(* CODESYS project ScaraRobot2Hand

Project tree, tasks and I/O mapping:
  Just_Motion_Control_x86_64_Linux_SM_WV : Just Motion Control Cortex-Linux SM WV, Shenzhen Just Motion Control Electromechanics Co., version 3.5.19.50
    application Application
      libraries: CommFB, * (3S - Smart Software Solutions GmbH); JMC COMMON, 3.5.17.0 (JMC); ModbusFB, 4.3.0.0 (3S - Smart Software Solutions GmbH); Standard, 3.5.18.0 (System); SysFile, * (System); SysTimeCore, * (System); SysTimeRtc, * (System)
      task EtherCAT_Task (cyclic, interval 8 ms, priority 1) calls POU_MOTION, POU_JOG_ROBOT, POU_CONTROL_ROBOT, POU_MONITOR_ROBOT, POU_COORDINATE_, POU_HOMING, PRG_TrackingObjectSource_A, PRG_TrackingQueue_A, PRG_MultiToolTracking_A, PRG_TrackingObjectSource_B, PRG_TrackingQueue_B, PRG_MultiToolTracking_B
      task SoftMotion_PlanningTask_1 (freewheeling, priority 15) calls nothing
      task SoftMotion_PlanningTask (freewheeling, priority 15) calls nothing
      task Task_Communication (cyclic, interval 15 ms, priority 1) calls POU_MODBUS, PRG_VisionConfigInit, POU_CAM, PRG_VisionModbus, PRG_VisionManager
      task Task_Program (cyclic, interval 8 ms, priority 20) calls Monitor_Production, POU_Alarm, POU_TransFormOXYR, POU_Main, POU_HMI_CONTROL_ROBOT, POU_SAFETY_CHECK
      ENUM/
        Application/
          data type E_ApplicationID
          data type E_ApplicationManagerState
          data type E_ApplicationSimulationMode
        Conveyor Tracking/
          data type E_ConveyorState
          data type E_MultiTrackState
          data type E_ObjectSourceType
          data type E_TrackingObjectState
          data type E_TrackingSelectMode
          data type E_TrackingState
        data type E_AppCoordSystem
        data type E_ApplicationState
        data type E_MoveState
        data type E_ObjectSelectMode
        data type E_QueueResult
        data type E_SystemTestStage
        GlueBonding/
          data type E_GlueRunMode
          data type E_GlueState
          data type E_PathProcessState
          data type E_PathSegmentType
        Interpreter/
          data type E_CondLink
          data type E_CondOperator
          data type E_CondSource
          data type E_RobotCmd
        TOOL/
          data type E_ToolAction
          data type E_ToolCommandType
          data type E_ToolRuntimeState
          data type E_ToolType
        Vision/
          data type E_AlignState
          data type E_InspectionResult
          data type E_InspectionState
          data type E_PlaceMode
          data type E_VisionApplication
          data type E_VisionDataType
          data type E_VisionResultStatus
          data type E_VisionRobot
          data type E_VisionState
      FB_/
        Application/
        function block Blink_Bit [ST]
        ConveyorTrack/
          function block FB_CONVEYOR_TRACKING_MANAGER [ST]
          function block FB_CONVEYOR_TRACKING_MANAGER_B [ST]
          function block FB_MultiToolTrackingController_A [ST]
          function block FB_MultiToolTrackingController_B [ST]
          function block FB_SensorObjectSource [ST]
          function block FB_TrackingCoreInterface_A [ST]
          function block FB_TrackingCoreInterface_B [ST]
          function block FB_TrackingMotionQueueAdapter [ST]
          function block FB_TrackingMotionQueueAdapter_B [ST]
          function block FB_VisionObjectSource [ST]
          function block FB_VisionTrackingResultAdapter [ST]
        function block FB_CalibRunPoints [ST]
        function block FB_CONVERT_POS [ST]
        function block FB_FileManager [ST]: Load, Save
        function block FB_MotionQueuePop [ST]
        function block FB_MotionQueuePop_B [ST]
        function block FB_MotionQueuePush [ST]
        function block FB_MotionQueuePush_B [ST]
        function block FB_PALLETS [ST]
        function block FB_Real_TO_Word_ [ST]
        function block FB_Run_Point [ST]
        function block FB_RunMoveC [ST]
        function block FB_RunMoveL [ST]
        function block FB_RunMoveP [ST]
        function block FB_RunMoveP_1 [ST]
        function block FB_TorqueDiff [ST]
        function block FB_TriggerVS [ST]
        function block FB_word_TO_real_ [ST]
        function block FB_Write_Log [ST]: Write
        Modbus/
          function block FB_VisionModbusDriver [ST]
        TOOL/
          function block FB_SelectRobotTool [ST]
          function block FB_SelectRobotTool_B [ST]
          function block FB_ToolManager [ST]
          function block FB_ToolManager_B [ST]
          function block FB_ToolObjectScheduler [ST]
        Vision/
          function block FB_VisionAlign_1 [ST]
          function block FB_VisionAlign [ST]
          function block FB_VisionGetResult [ST]
          function block FB_VisionTrackingTrigger [ST]
          function block FB_VisionWaitResult [ST]
      FC_/
        function ApplyTransformOnePointDeg [ST]
        function CalcScaraTransformDeg [ST]
        Conveyor/
          function F_AngleDifferenceDeg [ST]
          function F_IsTrackingObjectSelectable [ST]
          function F_IsVisionTrackingDuplicate [ST]
          function F_VisionTrackingRawToMM [ST]
        Coordinate_TF/
          function F_MapAppCoordSystem [ST]
        function F_BuildMotionItem [ST]
        function F_BuildMotionItem_B [ST]
        function F_CheckPositionReached [ST]
        function F_GetFreeMoveSlot [ST]
        function F_GetFreeMoveSlot_B [ST]
        function F_IsMotionCmd [ST]
        function FC_CalcCalibPoint [ST]
        function FC_Deg_To_Rad [ST]
        function FC_NormalizeAngleDeg [ST]
        function FC_Rad_To_Deg [ST]
        Geometry/
          function F_AngleBetweenPoints [ST]
          function F_DegToRad [ST]
          function F_Distance2D [ST]
          function F_Distance3D [ST]
          function F_NormalizeAngleDeg [ST]
          function F_NormalizeVector2D [ST]
          function F_RadToDeg [ST]
          function F_RotateAroundCenter2D [ST]
          function F_RotatePos2D [ST]
          function F_VectorLength2D [ST]
        function MyATAN2 [ST]
        Path/
          function F_CalculateBlendRadius [ST]
          function F_CalculatePathLength [ST]
          function F_InterpolatePosLinear [ST]
          function F_IsDuplicatePathPoint [ST]
          function F_PathPointDistance [ST]
        RBA/
          function F_CalcReg_A [ST]
          function F_CalcVar_A [ST]
          function F_CompareDINT_A [ST]
          function F_EvalCondition_A [ST]
          function F_EvalCondRow_A [ST]
          function F_EvalCondRowFromEdit_A [ST]
          function F_FindElseOrEndIf_A [ST]
          function F_FindEndIf_A [ST]
          function F_FindEndWhile_A [ST]
          function F_FindWhileStart_A [ST]
          function F_GetCondValue_A [ST]
          function F_GetPointSMC_A [ST]
        RBB/
          function F_CalcReg_B [ST]
          function F_CalcVar_B [ST]
          function F_CompareDINT_B [ST]
          function F_EvalCondition_B [ST]
          function F_EvalCondRow_B [ST]
          function F_EvalCondRowFromEdit_B [ST]
          function F_FindElseOrEndIf_B [ST]
          function F_FindEndIf_B [ST]
          function F_FindEndWhile_B [ST]
          function F_FindWhileStart_B [ST]
          function F_GetCondValue_B [ST]
          function F_GetPointSMC_B [ST]
        Tool/
          function F_ConvertToolTCP [ST]
        TrackingQueue/
          function F_SelectTrackingObject [ST]
        Vision/
          function F_CalcTraySlotTarget [ST]
          function F_CheckAlignResult [ST]
          function F_CheckPosRange [ST]
          function F_CheckRangeReal [ST]
          function F_CheckVisionHeader [ST]
          function F_CheckVisionScore [ST]
          function F_CountInspectionFail [ST]
          function F_VisionDINTHighWord [ST]
          function F_VisionDINTLowWord [ST]
          function F_VisionRealToRawDINT [ST]
          function F_VisionUDINTHighWord [ST]
          function F_VisionUDINTLowWord [ST]
          function F_VisionWordsToDINT_LH [ST]
          function F_VisionWordsToUDINT_LH [ST]
      GLOBAL_/
        global variables GVL_2
        global variables GVL
      global variables GVL_1
      PRG_MACHINE/
        program Monitor_Production [ST]: Qty_Production, Tactime_Input, Tactime_MC1, Tactime_MC2, Tactime_output
        program POU_Alarm [ST]: Alarm_Project_4, Alarm_Robot
        program POU_CAM [ST]: ACT_CHECKCONNECT, ACT_Total, ACT_TRIGGER_TOP
        program POU_MODBUS [ST]: ACT_TCP_Sever
        program PRG_VisionConfigInit [ST]
        program PRG_VisionModbus [ST]
        program PRG_VisionTest [ST]
      PRG_ROBOT/
        program POU_CONTROL_ROBOT [ST]: ACT_LOGIC, ACT_POWER, ACT_Reset, ACT_SET_DYNAMICLIMITS
        program POU_COORDINATE_ [ST]: ACT_CFC, ACT_Conver_Pos, ACT_LOGIC
        program POU_HMI_CONTROL_ROBOT [ST]: ACT_ControlPanel, ACT_HMI_A_ConditionEditor, ACT_HMI_A_Vision_Tracking_Config, ACT_HMI_B_ConditionEditor, ACT_HMI_B_Vision_Tracking_Config, ACT_HMI_Recipe_Config, ACT_HMI_Recipe_Config_B, ACT_HMI_SensorSource_Config_B, ACT_HMI_SensorSource_Config, ACT_HMIToolConfigEditor_A, ACT_HMIToolConfigEditor_B, ACT_JOG_LOGIC, ACT_MANORAUTO, ACT_MENU, ACT_select_rb, ACT_View_Edit_Cmd, ACT_View_Edit_Cmd_B, ACT_View_Edit_Point_A, ACT_View_Edit_Point_B
        program POU_HOMING [ST]: ACT_ERROR, ACT_Home_Z, ACT_HOMING, ACT_SETLIMIT, ACT_STOP
        program POU_JOG_ROBOT [ST]: ACT_JOG, ACT_LOGIC_A, ACT_LOGIC_B, ACT_LOGIC_R
        program POU_Main [ST]: ACT_IN, ACT_Manual_MC, ACT_Out, ACT_SAVE_FILE, ACT_SelectProjectRun, ACT_StatusMode, TimeTable
        program POU_MONITOR_ROBOT [ST]: ACT_LOGIC, ACT_READ, ACT_Teaching
        program POU_MOTION [ST]: MOVC, MOVL, MOVP, ACT_GO_Pos_Auto, Main_Base_Program_RB_A, PRG_A_MotionManager, Main_Base_Program_RB_B, PRG_B_MotionManager, _Main_Process_Test, A_Test_Motion, B1_Test_Motion, _Main_Process_Test_VS, A_Test_Motion_VS, B1_Test_Motion_VS, _Main_Process_4, A0_Wait_4, A1_Pick_T1_4, A2_Place_T1_OK_4, A3_Place_T1_NG_4, A4_Pick_T2_4, A5_Place_T2_OK_4, A6_Place_T2_NG_4, A7_Barcode_T1_4, A8_Place_T2_NG_TS_4, B0_wait_4, B1_Pick_T1_4, B2_PLace_T1_4, B3_Barcode_4, B_Trigger_4, CNV_NG, Pro_MC1_4_, Pro_MC2_4_, ACT_GO_Pos_Manual, B_Auto_Calib_4, Robot_Calib_Vision, M_CACULATOR_Z, M_CHOOSE_POS, M_CHOOSE_POS_Calib, M_CHOOSE_POS_Man, M_CHOOSE_POS_VS, M_CHOOSE_POS_XY, M_CHOOSE_POS_Z_BF, M_initProcess, M_R_Mov, M_reset, ACT_Excute_Run
        program POU_SAFETY_CHECK [ST]: ACT_RB_A, ACT_RB_B
        program POU_TransFormOXYR [ST]
        program PRG_MultiToolTracking_A [ST]
        program PRG_MultiToolTracking_B [ST]
        program PRG_TestVisionAlign [ST]
        program PRG_TestVisionTriggerResult [ST]
        program PRG_TrackingObjectSource_A [ST]
        program PRG_TrackingObjectSource_B [ST]
        program PRG_TrackingQueue_A [ST]
        program PRG_TrackingQueue_B [ST]
        program PRG_VisionManager [ST]
        program PRG_VisionTrackingTest_A [ST]
      axis group SCARA_A: TRAFO.Kin_Scara2_Z, axes A0, A1, A2
      axis group SCARA_B: TRAFO.Kin_Scara2_Z, axes B0, B1, B2
      STRUCT_/
        Alarm/
          data type Alarm_Robot
        Application/
          data type ST_APPLICATION_COMMAND
          data type ST_APPLICATION_RESPONSE
        Array/
          data type Pallets_In
          data type Pallets_Out
        CAM/
          data type Calib_Cam
          data type Calib_Cam_Input_Model
          data type ModbusCam
          data type VS_Control
        COMMON/
          data type ST_ERROR_INFO
          data type ST_MODULE_REQUEST
          data type ST_MODULE_RESPONSE
          data type ST_MotionProfile
          data type ST_POS
          data type ST_RANGE_REAL
          data type ST_Transform2D
          data type ST_VECTOR_2D
        ConveyorTracking/
          data type ST_CONVEYOR_CONFIG
          data type ST_CONVEYOR_RUNTIME
          data type ST_CONVEYOR_STATUS
          data type ST_HMIToolConfigEditor
          data type ST_PCS_INFO
          data type ST_SensorObjectSourceConfig
          data type ST_TRACKING_CONFIG
          data type ST_TRACKING_IO_CONFIG
          data type ST_TRACKING_MOTION_CONFIG
          data type ST_TRACKING_MOTION_PHASE_CONFIG
          data type ST_TRACKING_OBJECT
          data type ST_TRACKING_QUEUE
          data type ST_TRACKING_RUNTIME
          data type ST_TRACKING_SIMULATION_CONFIG
          data type ST_TRACKING_WORKSPACE_CONFIG
          data type ST_TrackingObjectQueue
          data type ST_VISION_TRACK_OBJECT_ITEM
          data type ST_VISION_TRACK_OBJECT_RESULT
          data type ST_VisionTrackingDetection
          data type ST_VisionTrackingMultiResult
          data type ST_VisionTrackingSourceConfig
        Geometry/
          data type ST_CIRCLE_2D
          data type ST_LINE_2D
          data type ST_PATH_BLOCK
          data type ST_PATH_DATA
          data type ST_PATH_POINT
        Glue/
          data type ST_GLUE_CONFIG
          data type ST_GLUE_RUNTIME
        HMI/
          data type MainMC
          data type MODBUS
          data type Project
          data type TimeRun
        Modbus/
          data type ST_VISION_MODBUS_CONTROL
          data type ST_VISION_MODBUS_STATUS
        MOTOR/
          data type MOTOR_DATA
          data type MOTOR_IN
          data type MOTOR_OUT
        Project/
          data type Data_Point_Calib
          data type Data_Project_3
          data type Data_Project
          Project1/
          data type Project_2
          data type Project_3
          data type Project_3_VISION
          Project_4/
            data type Alarm_P_4
            data type Pro4_auto
            data type Pro4_Input
            data type Pro4_manual
            data type Pro4_Monitor
            data type Pro4_Process
            data type Pro4_RB_Pos
            data type Pro4_setting
            data type Pro4_Setting_Funtion
            data type Project4
        ROBOT/
          data type Model_Data_RB_ALL
          data type Model_Data_RB
          data type Move_Point
          data type Move_Type
          data type PCS_Data
          data type Pos_Coordsystem
          data type Project_And_Model
          data type RB_DATA
          data type RB_IN
          data type RB_IN_Man
          data type RB_OUT
          data type RB_Signal_Input
          data type RB_Speed_Point
          data type ST_Condition
          data type ST_ConditionLine
          data type ST_ConditionRow
          data type ST_ConditionTable
          data type ST_MotionParam
          data type ST_MotionQueueItem
          data type ST_RobotProgram
          data type ST_RobotStep
          data type ST_ScaraTransformDeg
          data type Torque_Axis
        TOOL/
          data type ST_MultiToolTrackingCommand
          data type ST_MultiToolTrackingRecipe
          data type ST_MultiToolTrackingStatus
          data type ST_ToolCommand
          data type ST_ToolConfig
          data type ST_ToolIOConfig
          data type ST_ToolStatus
        Vision/
          data type ST_ALIGN_CONFIG
          data type ST_ALIGN_RESULT
          data type ST_ALIGN_RUNTIME
          data type ST_AlignResult
          data type ST_ControlWord_VS
          data type ST_INSPECTION_CONFIG
          data type ST_INSPECTION_ITEM
          data type ST_INSPECTION_RESULT
          data type ST_INSPECTION_RUNTIME
          data type ST_InspectionItem
          data type ST_PathPoint
          data type ST_StatusWord_VS
          data type ST_TrayConfig
          data type ST_TrayRuntime
          data type ST_VISION_ALIGN_REQUEST
          data type ST_VISION_CHANNEL_STATUS
          data type ST_VISION_COMMAND
          data type ST_VISION_CONFIG
          data type ST_VISION_JOB_CONFIG
          data type ST_VISION_POS_RESULT
          data type ST_VISION_RESULT
          data type ST_VISION_RESULT_HEADER
          data type ST_VisionAlignRecipe
          data type ST_VisionAlignToolConfig
          data type ST_VisionAlignToolRuntime
          data type ST_VisionCommand
      Symbols
      trace Trace (task EtherCAT_Task): B1.fSetVelocity, B1.fActVelocity, B3.fSetVelocity, B3.fActVelocity, A0.diSetVelocity, A0.diActVelocity, A1.diSetVelocity, A1.diActVelocity, POU_CONTROL_ROBOT.J1_PosError, POU_CONTROL_ROBOT.J2_PosError, POU_CONTROL_ROBOT.J1_VelError, POU_CONTROL_ROBOT.J2_VelError, A0.fSetPosition, A0.fActPosition, A0.fActPosition, A0.fActPosition, A1.fActPosition, A1.fSetPosition, A1.fSetVelocity, A1.fActVelocity, GVL.RB_A_.CUR_X, GVL.RB_A_.CUR_Y, GVL.RB_A_.CUR_SP_X, GVL.RB_A_.CUR_SP_Y, SM_Drive_Logical.fActPosition
    EtherCAT_Master_SoftMotion : EtherCAT Master SoftMotion, CODESYS, version 4.6.0.0
        settings: MasterCycleTime = 8000; NetworkName = 'EtherCAT'; NetworkName = "EtherCAT"; SelectNetworkByName = False; SyncOffset = -20; SrcAddress1 = 3830; SrcAddress2 = 3107753849
      TA133 : TA133, Shenzhen Just Motion Control Electromechanics Co,.ltd, order no. TA133, version Revision=16#00010004
          settings: ModularDevice = True; EnableExpertSettings = True; MDP_InputOffsets = [0,736]; MDP_OutputOffsets = [0,984]; StationAlias = 1001; DeviceIdenticationADO = 18; DeviceIdenticationMode = 1; Sync.Length = 127; Sync.Length = 97; FMMU.Length = 127; FMMU.Length = 97; Number of RxPDOs of the Slave = 8; Number of TxPDOs of the Slave = 8; DC sync0 cycletime = 8000; DC enable = 1; DC sync0 enable = 1; DC sync0 shift time = 0; DC sync1 cycletime = 8000; DC sync1 enable = 0; DC sync1 shift time = 0; Number of SDO = 1; download slot cfg.Index = 16#F030; download slot cfg.Subindex = 16#00; download slot cfg.Size = 48; download slot cfg.AbortIfError = FALSE; download slot cfg.JumpToLine = FALSE; download slot cfg.Line = 0; download slot cfg.CompleteAccess = True; download slot cfg = [1,0,230,0,0,0]; RxTxPdo.NumberofExcludes = 0; RxTxPdo.NumberofEntries = 7; RxTxPdo.Index = 16#1700; RxTxPdo.Fixed = False; RxTxPdo.Mandatory = False; RxTxPdo.Virtual = False; RxTxPdo.Sm = 2; RxTxPdo.Su = 2; RxTxPdo.Name = 'Outputs'; RxTxPdo.DependOnSlot = False; RxTxPdo.DependOnSlotGroup = False;
            RxTxPdo.OverwrittenByModule = False; Controlword(axis 1).Index = 16#6040; Controlword(axis 1).SubIndex = 0; Controlword(axis 1).Size = 16; Controlword(axis 1).Offset = 0; Controlword(axis 1).DependOnSlot = False; Controlword(axis 1).DependOnSlotGroup = False; Modes of operation(axis 1).Index = 16#6060; Modes of operation(axis 1).SubIndex = 0; Modes of operation(axis 1).Size = 8; Modes of operation(axis 1).Offset = 0; Modes of operation(axis 1).DependOnSlot = False; Modes of operation(axis 1).DependOnSlotGroup = False; Target position(axis 1).Index = 16#607A; Target position(axis 1).SubIndex = 0; Target position(axis 1).Size = 32; Target position(axis 1).Offset = 0; Target position(axis 1).DependOnSlot = False; Target position(axis 1).DependOnSlotGroup = False; High-speed comparison 1(axis 1).Index = 16#6701; High-speed comparison 1(axis 1).SubIndex = 0; High-speed comparison 1(axis 1).Size = 32; High-speed comparison 1(axis 1).Offset = 0; High-speed comparison 1(axis 1).DependOnSlot = False; High-speed comparison 1(axis 1).DependOnSlotGroup = False; High-speed comparison 2(axis 1).Index = 16#6702; High-speed comparison 2(axis 1).SubIndex = 0; High-speed comparison 2(axis 1).Size = 32; High-speed comparison 2(axis 1).Offset = 0; High-speed comparison 2(axis 1).DependOnSlot = False; High-speed comparison 2(axis 1).DependOnSlotGroup = False; PWM Duty(axis 1).Index = 16#6707; PWM Duty(axis 1).SubIndex = 0; PWM Duty(axis 1).Size = 8; PWM Duty(axis 1).Offset = 0; PWM Duty(axis 1).DependOnSlot = False; PWM Duty(axis 1).DependOnSlotGroup = False; PWM Freq(axis 1).Index = 16#6708; PWM Freq(axis 1).SubIndex = 0; PWM Freq(axis 1).Size = 32;
            PWM Freq(axis 1).Offset = 0; PWM Freq(axis 1).DependOnSlot = False; PWM Freq(axis 1).DependOnSlotGroup = False; RxTxPdo.NumberofExcludes = 0; RxTxPdo.NumberofEntries = 7; RxTxPdo.Index = 16#1710; RxTxPdo.Fixed = False; RxTxPdo.Mandatory = False; RxTxPdo.Virtual = False; RxTxPdo.Sm = 2; RxTxPdo.Su = 2; RxTxPdo.Name = 'Outputs'; RxTxPdo.DependOnSlot = False; RxTxPdo.DependOnSlotGroup = False; RxTxPdo.OverwrittenByModule = False; Controlword(axis 2).Index = 16#6840; Controlword(axis 2).SubIndex = 0; Controlword(axis 2).Size = 16; Controlword(axis 2).Offset = 0; Controlword(axis 2).DependOnSlot = False; Controlword(axis 2).DependOnSlotGroup = False; Modes of operation(axis 2).Index = 16#6860; Modes of operation(axis 2).SubIndex = 0; Modes of operation(axis 2).Size = 8; Modes of operation(axis 2).Offset = 0; Modes of operation(axis 2).DependOnSlot = False; Modes of operation(axis 2).DependOnSlotGroup = False; Target position(axis 2).Index = 16#687A; Target position(axis 2).SubIndex = 0; Target position(axis 2).Size = 32; Target position(axis 2).Offset = 0; Target position(axis 2).DependOnSlot = False; Target position(axis 2).DependOnSlotGroup = False; High-speed comparison 1(axis 2).Index = 16#6F01; High-speed comparison 1(axis 2).SubIndex = 0; High-speed comparison 1(axis 2).Size = 32; High-speed comparison 1(axis 2).Offset = 0; High-speed comparison 1(axis 2).DependOnSlot = False; High-speed comparison 1(axis 2).DependOnSlotGroup = False; High-speed comparison 2(axis 2).Index = 16#6F02;
            High-speed comparison 2(axis 2).SubIndex = 0; High-speed comparison 2(axis 2).Size = 32; High-speed comparison 2(axis 2).Offset = 0; High-speed comparison 2(axis 2).DependOnSlot = False; High-speed comparison 2(axis 2).DependOnSlotGroup = False; PWM Duty(axis 2).Index = 16#6F07; PWM Duty(axis 2).SubIndex = 0; PWM Duty(axis 2).Size = 8; PWM Duty(axis 2).Offset = 0; PWM Duty(axis 2).DependOnSlot = False; PWM Duty(axis 2).DependOnSlotGroup = False; PWM Freq(axis 2).Index = 16#6F08; PWM Freq(axis 2).SubIndex = 0; PWM Freq(axis 2).Size = 32; PWM Freq(axis 2).Offset = 0; PWM Freq(axis 2).DependOnSlot = False; PWM Freq(axis 2).DependOnSlotGroup = False; RxTxPdo.NumberofExcludes = 0; RxTxPdo.NumberofEntries = 7; RxTxPdo.Index = 16#1720; RxTxPdo.Fixed = False; RxTxPdo.Mandatory = False; RxTxPdo.Virtual = False; RxTxPdo.Sm = 2; RxTxPdo.Su = 2; RxTxPdo.Name = 'Outputs'; RxTxPdo.DependOnSlot = False; RxTxPdo.DependOnSlotGroup = False; RxTxPdo.OverwrittenByModule = False; Controlword(axis 3).Index = 16#7040; Controlword(axis 3).SubIndex = 0; Controlword(axis 3).Size = 16; Controlword(axis 3).Offset = 0; Controlword(axis 3).DependOnSlot = False; Controlword(axis 3).DependOnSlotGroup = False; Modes of operation(axis 3).Index = 16#7060; Modes of operation(axis 3).SubIndex = 0; Modes of operation(axis 3).Size = 8; Modes of operation(axis 3).Offset = 0; Modes of operation(axis 3).DependOnSlot = False;
            Modes of operation(axis 3).DependOnSlotGroup = False; Target position(axis 3).Index = 16#707A; Target position(axis 3).SubIndex = 0; Target position(axis 3).Size = 32; Target position(axis 3).Offset = 0; Target position(axis 3).DependOnSlot = False; Target position(axis 3).DependOnSlotGroup = False; High-speed comparison 1(axis 3).Index = 16#7701; High-speed comparison 1(axis 3).SubIndex = 0; High-speed comparison 1(axis 3).Size = 32; High-speed comparison 1(axis 3).Offset = 0; High-speed comparison 1(axis 3).DependOnSlot = False; High-speed comparison 1(axis 3).DependOnSlotGroup = False; High-speed comparison 2(axis 3).Index = 16#7702; High-speed comparison 2(axis 3).SubIndex = 0; High-speed comparison 2(axis 3).Size = 32; High-speed comparison 2(axis 3).Offset = 0; High-speed comparison 2(axis 3).DependOnSlot = False; High-speed comparison 2(axis 3).DependOnSlotGroup = False; PWM Duty(axis 3).Index = 16#7707; PWM Duty(axis 3).SubIndex = 0; PWM Duty(axis 3).Size = 8; PWM Duty(axis 3).Offset = 0; PWM Duty(axis 3).DependOnSlot = False; PWM Duty(axis 3).DependOnSlotGroup = False; PWM Freq(axis 3).Index = 16#7708; PWM Freq(axis 3).SubIndex = 0; PWM Freq(axis 3).Size = 32; PWM Freq(axis 3).Offset = 0; PWM Freq(axis 3).DependOnSlot = False; PWM Freq(axis 3).DependOnSlotGroup = False; RxTxPdo.NumberofExcludes = 0; RxTxPdo.NumberofEntries = 7; RxTxPdo.Index = 16#1730; RxTxPdo.Fixed = False; RxTxPdo.Mandatory = False; RxTxPdo.Virtual = False; RxTxPdo.Sm = 2; RxTxPdo.Su = 2; RxTxPdo.Name = 'Outputs';
            RxTxPdo.DependOnSlot = False; RxTxPdo.DependOnSlotGroup = False; RxTxPdo.OverwrittenByModule = False; Controlword(axis 4).Index = 16#7840; Controlword(axis 4).SubIndex = 0; Controlword(axis 4).Size = 16; Controlword(axis 4).Offset = 0; Controlword(axis 4).DependOnSlot = False; Controlword(axis 4).DependOnSlotGroup = False; Modes of operation(axis 4).Index = 16#7860; Modes of operation(axis 4).SubIndex = 0; Modes of operation(axis 4).Size = 8; Modes of operation(axis 4).Offset = 0; Modes of operation(axis 4).DependOnSlot = False; Modes of operation(axis 4).DependOnSlotGroup = False; Target position(axis 4).Index = 16#787A; Target position(axis 4).SubIndex = 0; Target position(axis 4).Size = 32; Target position(axis 4).Offset = 0; Target position(axis 4).DependOnSlot = False; Target position(axis 4).DependOnSlotGroup = False; High-speed comparison 1(axis 4).Index = 16#7F01; High-speed comparison 1(axis 4).SubIndex = 0; High-speed comparison 1(axis 4).Size = 32; High-speed comparison 1(axis 4).Offset = 0; High-speed comparison 1(axis 4).DependOnSlot = False; High-speed comparison 1(axis 4).DependOnSlotGroup = False; High-speed comparison 2(axis 4).Index = 16#7F02; High-speed comparison 2(axis 4).SubIndex = 0; High-speed comparison 2(axis 4).Size = 32; High-speed comparison 2(axis 4).Offset = 0; High-speed comparison 2(axis 4).DependOnSlot = False; High-speed comparison 2(axis 4).DependOnSlotGroup = False; PWM Duty(axis 4).Index = 16#7F07; PWM Duty(axis 4).SubIndex = 0; PWM Duty(axis 4).Size = 8; PWM Duty(axis 4).Offset = 0; PWM Duty(axis 4).DependOnSlot = False; PWM Duty(axis 4).DependOnSlotGroup = False; PWM Freq(axis 4).Index = 16#7F08;
            PWM Freq(axis 4).SubIndex = 0; PWM Freq(axis 4).Size = 32; PWM Freq(axis 4).Offset = 0; PWM Freq(axis 4).DependOnSlot = False; PWM Freq(axis 4).DependOnSlotGroup = False; RxTxPdo.NumberofExcludes = 0; RxTxPdo.NumberofEntries = 7; RxTxPdo.Index = 16#1740; RxTxPdo.Fixed = False; RxTxPdo.Mandatory = False; RxTxPdo.Virtual = False; RxTxPdo.Sm = 2; RxTxPdo.Su = 2; RxTxPdo.Name = 'Outputs'; RxTxPdo.DependOnSlot = False; RxTxPdo.DependOnSlotGroup = False; RxTxPdo.OverwrittenByModule = False; Controlword(axis 5).Index = 16#8040; Controlword(axis 5).SubIndex = 0; Controlword(axis 5).Size = 16; Controlword(axis 5).Offset = 0; Controlword(axis 5).DependOnSlot = False; Controlword(axis 5).DependOnSlotGroup = False; Modes of operation(axis 5).Index = 16#8060; Modes of operation(axis 5).SubIndex = 0; Modes of operation(axis 5).Size = 8; Modes of operation(axis 5).Offset = 0; Modes of operation(axis 5).DependOnSlot = False; Modes of operation(axis 5).DependOnSlotGroup = False; Target position(axis 5).Index = 16#807A; Target position(axis 5).SubIndex = 0; Target position(axis 5).Size = 32; Target position(axis 5).Offset = 0; Target position(axis 5).DependOnSlot = False; Target position(axis 5).DependOnSlotGroup = False; High-speed comparison 1(axis 5).Index = 16#8701; High-speed comparison 1(axis 5).SubIndex = 0; High-speed comparison 1(axis 5).Size = 32; High-speed comparison 1(axis 5).Offset = 0; High-speed comparison 1(axis 5).DependOnSlot = False;
            High-speed comparison 1(axis 5).DependOnSlotGroup = False; High-speed comparison 2(axis 5).Index = 16#8702; High-speed comparison 2(axis 5).SubIndex = 0; High-speed comparison 2(axis 5).Size = 32; High-speed comparison 2(axis 5).Offset = 0; High-speed comparison 2(axis 5).DependOnSlot = False; High-speed comparison 2(axis 5).DependOnSlotGroup = False; PWM Duty(axis 5).Index = 16#8707; PWM Duty(axis 5).SubIndex = 0; PWM Duty(axis 5).Size = 8; PWM Duty(axis 5).Offset = 0; PWM Duty(axis 5).DependOnSlot = False; PWM Duty(axis 5).DependOnSlotGroup = False; PWM Freq(axis 5).Index = 16#8708; PWM Freq(axis 5).SubIndex = 0; PWM Freq(axis 5).Size = 32; PWM Freq(axis 5).Offset = 0; PWM Freq(axis 5).DependOnSlot = False; PWM Freq(axis 5).DependOnSlotGroup = False; RxTxPdo.NumberofExcludes = 0; RxTxPdo.NumberofEntries = 7; RxTxPdo.Index = 16#1750; RxTxPdo.Fixed = False; RxTxPdo.Mandatory = False; RxTxPdo.Virtual = False; RxTxPdo.Sm = 2; RxTxPdo.Su = 2; RxTxPdo.Name = 'Outputs'; RxTxPdo.DependOnSlot = False; RxTxPdo.DependOnSlotGroup = False; RxTxPdo.OverwrittenByModule = False; Controlword(axis 6).Index = 16#8840; Controlword(axis 6).SubIndex = 0; Controlword(axis 6).Size = 16; Controlword(axis 6).Offset = 0; Controlword(axis 6).DependOnSlot = False; Controlword(axis 6).DependOnSlotGroup = False; Modes of operation(axis 6).Index = 16#8860; Modes of operation(axis 6).SubIndex = 0; Modes of operation(axis 6).Size = 8;
            Modes of operation(axis 6).Offset = 0; Modes of operation(axis 6).DependOnSlot = False; Modes of operation(axis 6).DependOnSlotGroup = False; Target position(axis 6).Index = 16#887A; Target position(axis 6).SubIndex = 0; Target position(axis 6).Size = 32; Target position(axis 6).Offset = 0; Target position(axis 6).DependOnSlot = False; Target position(axis 6).DependOnSlotGroup = False; High-speed comparison 1(axis 6).Index = 16#8F01; High-speed comparison 1(axis 6).SubIndex = 0; High-speed comparison 1(axis 6).Size = 32; High-speed comparison 1(axis 6).Offset = 0; High-speed comparison 1(axis 6).DependOnSlot = False; High-speed comparison 1(axis 6).DependOnSlotGroup = False; High-speed comparison 2(axis 6).Index = 16#8F02; High-speed comparison 2(axis 6).SubIndex = 0; High-speed comparison 2(axis 6).Size = 32; High-speed comparison 2(axis 6).Offset = 0; High-speed comparison 2(axis 6).DependOnSlot = False; High-speed comparison 2(axis 6).DependOnSlotGroup = False; PWM Duty(axis 6).Index = 16#8F07; PWM Duty(axis 6).SubIndex = 0; PWM Duty(axis 6).Size = 8; PWM Duty(axis 6).Offset = 0; PWM Duty(axis 6).DependOnSlot = False; PWM Duty(axis 6).DependOnSlotGroup = False; PWM Freq(axis 6).Index = 16#8F08; PWM Freq(axis 6).SubIndex = 0; PWM Freq(axis 6).Size = 32; PWM Freq(axis 6).Offset = 0; PWM Freq(axis 6).DependOnSlot = False; PWM Freq(axis 6).DependOnSlotGroup = False; RxTxPdo.NumberofExcludes = 0; RxTxPdo.NumberofEntries = 3; RxTxPdo.Index = 16#1760; RxTxPdo.Fixed = False; RxTxPdo.Mandatory = False; RxTxPdo.Virtual = False; RxTxPdo.Sm = 2;
            RxTxPdo.Su = 2; RxTxPdo.Name = 'Outputs'; RxTxPdo.DependOnSlot = False; RxTxPdo.DependOnSlotGroup = False; RxTxPdo.OverwrittenByModule = False; High-speed comparison 1 switch.Index = 16#6703; High-speed comparison 1 switch.SubIndex = 0; High-speed comparison 1 switch.Size = 8; High-speed comparison 1 switch.Offset = 0; High-speed comparison 1 switch.DependOnSlot = False; High-speed comparison 1 switch.DependOnSlotGroup = False; High-speed comparison 2 switch.Index = 16#6704; High-speed comparison 2 switch.SubIndex = 0; High-speed comparison 2 switch.Size = 8; High-speed comparison 2 switch.Offset = 0; High-speed comparison 2 switch.DependOnSlot = False; High-speed comparison 2 switch.DependOnSlotGroup = False; PWM Output Enable.Index = 16#6709; PWM Output Enable.SubIndex = 0; PWM Output Enable.Size = 8; PWM Output Enable.Offset = 0; PWM Output Enable.DependOnSlot = False; PWM Output Enable.DependOnSlotGroup = False; RxTxPdo.NumberofExcludes = 0; RxTxPdo.NumberofEntries = 17; RxTxPdo.Index = 16#1600; RxTxPdo.Fixed = True; RxTxPdo.Mandatory = True; RxTxPdo.Virtual = False; RxTxPdo.Sm = 2; RxTxPdo.Su = 0; RxTxPdo.Name = 'Outputs process data mapping'; RxTxPdo.DependOnSlot = True; RxTxPdo.DependOnSlotGroup = False; RxTxPdo.OverwrittenByModule = True; AO0.Index = 16#7000; AO0.SubIndex = 1; AO0.Size = 16; AO0.Offset = 0; AO0.DependOnSlot = True;
            AO0.DependOnSlotGroup = False; Y0.Index = 16#7000; Y0.SubIndex = 2; Y0.Size = 1; Y0.Offset = 0; Y0.DependOnSlot = True; Y0.DependOnSlotGroup = False; Y1.Index = 16#7000; Y1.SubIndex = 3; Y1.Size = 1; Y1.Offset = 0; Y1.DependOnSlot = True; Y1.DependOnSlotGroup = False; Y2.Index = 16#7000; Y2.SubIndex = 4; Y2.Size = 1; Y2.Offset = 0; Y2.DependOnSlot = True; Y2.DependOnSlotGroup = False; Y3.Index = 16#7000; Y3.SubIndex = 5; Y3.Size = 1; Y3.Offset = 0; Y3.DependOnSlot = True; Y3.DependOnSlotGroup = False; Y4.Index = 16#7000; Y4.SubIndex = 6; Y4.Size = 1; Y4.Offset = 0; Y4.DependOnSlot = True; Y4.DependOnSlotGroup = False; Y5.Index = 16#7000; Y5.SubIndex = 7; Y5.Size = 1; Y5.Offset = 0; Y5.DependOnSlot = True; Y5.DependOnSlotGroup = False; Y6.Index = 16#7000; Y6.SubIndex = 8; Y6.Size = 1;
            Y6.Offset = 0; Y6.DependOnSlot = True; Y6.DependOnSlotGroup = False; Y7.Index = 16#7000; Y7.SubIndex = 9; Y7.Size = 1; Y7.Offset = 0; Y7.DependOnSlot = True; Y7.DependOnSlotGroup = False; Y8.Index = 16#7000; Y8.SubIndex = 10; Y8.Size = 1; Y8.Offset = 0; Y8.DependOnSlot = True; Y8.DependOnSlotGroup = False; Y9.Index = 16#7000; Y9.SubIndex = 11; Y9.Size = 1; Y9.Offset = 0; Y9.DependOnSlot = True; Y9.DependOnSlotGroup = False; Y10.Index = 16#7000; Y10.SubIndex = 12; Y10.Size = 1; Y10.Offset = 0; Y10.DependOnSlot = True; Y10.DependOnSlotGroup = False; Y11.Index = 16#7000; Y11.SubIndex = 13; Y11.Size = 1; Y11.Offset = 0; Y11.DependOnSlot = True; Y11.DependOnSlotGroup = False; Y12.Index = 16#7000; Y12.SubIndex = 14; Y12.Size = 1; Y12.Offset = 0; Y12.DependOnSlot = True; Y12.DependOnSlotGroup = False; Y13.Index = 16#7000;
            Y13.SubIndex = 15; Y13.Size = 1; Y13.Offset = 0; Y13.DependOnSlot = True; Y13.DependOnSlotGroup = False; Y14.Index = 16#7000; Y14.SubIndex = 16; Y14.Size = 1; Y14.Offset = 0; Y14.DependOnSlot = True; Y14.DependOnSlotGroup = False; Y15.Index = 16#7000; Y15.SubIndex = 17; Y15.Size = 1; Y15.Offset = 0; Y15.DependOnSlot = True; Y15.DependOnSlotGroup = False; RxTxPdo.NumberofExcludes = 0; RxTxPdo.NumberofEntries = 6; RxTxPdo.Index = 16#1B00; RxTxPdo.Fixed = False; RxTxPdo.Mandatory = False; RxTxPdo.Virtual = False; RxTxPdo.Sm = 3; RxTxPdo.Su = 3; RxTxPdo.Name = 'Inputs'; RxTxPdo.DependOnSlot = False; RxTxPdo.DependOnSlotGroup = False; RxTxPdo.OverwrittenByModule = False; Error Code(axis 1).Index = 16#603F; Error Code(axis 1).SubIndex = 0; Error Code(axis 1).Size = 16; Error Code(axis 1).Offset = 0; Error Code(axis 1).DependOnSlot = False; Error Code(axis 1).DependOnSlotGroup = False; Statusword(axis 1).Index = 16#6041; Statusword(axis 1).SubIndex = 0; Statusword(axis 1).Size = 16; Statusword(axis 1).Offset = 0; Statusword(axis 1).DependOnSlot = False;
            Statusword(axis 1).DependOnSlotGroup = False; Modes of operation display(axis 1).Index = 16#6061; Modes of operation display(axis 1).SubIndex = 0; Modes of operation display(axis 1).Size = 8; Modes of operation display(axis 1).Offset = 0; Modes of operation display(axis 1).DependOnSlot = False; Modes of operation display(axis 1).DependOnSlotGroup = False; Position actual value(axis 1).Index = 16#6064; Position actual value(axis 1).SubIndex = 0; Position actual value(axis 1).Size = 32; Position actual value(axis 1).Offset = 0; Position actual value(axis 1).DependOnSlot = False; Position actual value(axis 1).DependOnSlotGroup = False; Encoder Z phase(axis 1).Index = 16#6705; Encoder Z phase(axis 1).SubIndex = 0; Encoder Z phase(axis 1).Size = 32; Encoder Z phase(axis 1).Offset = 0; Encoder Z phase(axis 1).DependOnSlot = False; Encoder Z phase(axis 1).DependOnSlotGroup = False; PWM Error Code(axis 1).Index = 16#6711; PWM Error Code(axis 1).SubIndex = 0; PWM Error Code(axis 1).Size = 16; PWM Error Code(axis 1).Offset = 0; PWM Error Code(axis 1).DependOnSlot = False; PWM Error Code(axis 1).DependOnSlotGroup = False; RxTxPdo.NumberofExcludes = 0; RxTxPdo.NumberofEntries = 6; RxTxPdo.Index = 16#1B10; RxTxPdo.Fixed = False; RxTxPdo.Mandatory = False; RxTxPdo.Virtual = False; RxTxPdo.Sm = 3; RxTxPdo.Su = 3; RxTxPdo.Name = 'Inputs'; RxTxPdo.DependOnSlot = False; RxTxPdo.DependOnSlotGroup = False; RxTxPdo.OverwrittenByModule = False; Error Code(axis 2).Index = 16#683F; Error Code(axis 2).SubIndex = 0; Error Code(axis 2).Size = 16;
            Error Code(axis 2).Offset = 0; Error Code(axis 2).DependOnSlot = False; Error Code(axis 2).DependOnSlotGroup = False; Statusword(axis 2).Index = 16#6841; Statusword(axis 2).SubIndex = 0; Statusword(axis 2).Size = 16; Statusword(axis 2).Offset = 0; Statusword(axis 2).DependOnSlot = False; Statusword(axis 2).DependOnSlotGroup = False; Modes of operation display(axis 2).Index = 16#6861; Modes of operation display(axis 2).SubIndex = 0; Modes of operation display(axis 2).Size = 8; Modes of operation display(axis 2).Offset = 0; Modes of operation display(axis 2).DependOnSlot = False; Modes of operation display(axis 2).DependOnSlotGroup = False; Position actual value(axis 2).Index = 16#6864; Position actual value(axis 2).SubIndex = 0; Position actual value(axis 2).Size = 32; Position actual value(axis 2).Offset = 0; Position actual value(axis 2).DependOnSlot = False; Position actual value(axis 2).DependOnSlotGroup = False; Encoder Z phase(axis 2).Index = 16#6F05; Encoder Z phase(axis 2).SubIndex = 0; Encoder Z phase(axis 2).Size = 32; Encoder Z phase(axis 2).Offset = 0; Encoder Z phase(axis 2).DependOnSlot = False; Encoder Z phase(axis 2).DependOnSlotGroup = False; PWM Error Code(axis 2).Index = 16#6F11; PWM Error Code(axis 2).SubIndex = 0; PWM Error Code(axis 2).Size = 16; PWM Error Code(axis 2).Offset = 0; PWM Error Code(axis 2).DependOnSlot = False; PWM Error Code(axis 2).DependOnSlotGroup = False; RxTxPdo.NumberofExcludes = 0; RxTxPdo.NumberofEntries = 6; RxTxPdo.Index = 16#1B20; RxTxPdo.Fixed = False; RxTxPdo.Mandatory = False; RxTxPdo.Virtual = False; RxTxPdo.Sm = 3;
            RxTxPdo.Su = 3; RxTxPdo.Name = 'Inputs'; RxTxPdo.DependOnSlot = False; RxTxPdo.DependOnSlotGroup = False; RxTxPdo.OverwrittenByModule = False; Error Code(axis 3).Index = 16#703F; Error Code(axis 3).SubIndex = 0; Error Code(axis 3).Size = 16; Error Code(axis 3).Offset = 0; Error Code(axis 3).DependOnSlot = False; Error Code(axis 3).DependOnSlotGroup = False; Statusword(axis 3).Index = 16#7041; Statusword(axis 3).SubIndex = 0; Statusword(axis 3).Size = 16; Statusword(axis 3).Offset = 0; Statusword(axis 3).DependOnSlot = False; Statusword(axis 3).DependOnSlotGroup = False; Modes of operation display(axis 3).Index = 16#7061; Modes of operation display(axis 3).SubIndex = 0; Modes of operation display(axis 3).Size = 8; Modes of operation display(axis 3).Offset = 0; Modes of operation display(axis 3).DependOnSlot = False; Modes of operation display(axis 3).DependOnSlotGroup = False; Position actual value(axis 3).Index = 16#7064; Position actual value(axis 3).SubIndex = 0; Position actual value(axis 3).Size = 32; Position actual value(axis 3).Offset = 0; Position actual value(axis 3).DependOnSlot = False; Position actual value(axis 3).DependOnSlotGroup = False; Encoder Z phase(axis 3).Index = 16#7705; Encoder Z phase(axis 3).SubIndex = 0; Encoder Z phase(axis 3).Size = 32; Encoder Z phase(axis 3).Offset = 0; Encoder Z phase(axis 3).DependOnSlot = False; Encoder Z phase(axis 3).DependOnSlotGroup = False; PWM Error Code(axis 3).Index = 16#7711; PWM Error Code(axis 3).SubIndex = 0; PWM Error Code(axis 3).Size = 16; PWM Error Code(axis 3).Offset = 0; PWM Error Code(axis 3).DependOnSlot = False;
            PWM Error Code(axis 3).DependOnSlotGroup = False; RxTxPdo.NumberofExcludes = 0; RxTxPdo.NumberofEntries = 6; RxTxPdo.Index = 16#1B30; RxTxPdo.Fixed = False; RxTxPdo.Mandatory = False; RxTxPdo.Virtual = False; RxTxPdo.Sm = 3; RxTxPdo.Su = 3; RxTxPdo.Name = 'Inputs'; RxTxPdo.DependOnSlot = False; RxTxPdo.DependOnSlotGroup = False; RxTxPdo.OverwrittenByModule = False; Error Code(axis 4).Index = 16#783F; Error Code(axis 4).SubIndex = 0; Error Code(axis 4).Size = 16; Error Code(axis 4).Offset = 0; Error Code(axis 4).DependOnSlot = False; Error Code(axis 4).DependOnSlotGroup = False; Statusword(axis 4).Index = 16#7841; Statusword(axis 4).SubIndex = 0; Statusword(axis 4).Size = 16; Statusword(axis 4).Offset = 0; Statusword(axis 4).DependOnSlot = False; Statusword(axis 4).DependOnSlotGroup = False; Modes of operation display(axis 4).Index = 16#7861; Modes of operation display(axis 4).SubIndex = 0; Modes of operation display(axis 4).Size = 8; Modes of operation display(axis 4).Offset = 0; Modes of operation display(axis 4).DependOnSlot = False; Modes of operation display(axis 4).DependOnSlotGroup = False; Position actual value(axis 4).Index = 16#7864; Position actual value(axis 4).SubIndex = 0; Position actual value(axis 4).Size = 32; Position actual value(axis 4).Offset = 0; Position actual value(axis 4).DependOnSlot = False; Position actual value(axis 4).DependOnSlotGroup = False; Encoder Z phase(axis 4).Index = 16#7F05; Encoder Z phase(axis 4).SubIndex = 0; Encoder Z phase(axis 4).Size = 32;
            Encoder Z phase(axis 4).Offset = 0; Encoder Z phase(axis 4).DependOnSlot = False; Encoder Z phase(axis 4).DependOnSlotGroup = False; PWM Error Code(axis 4).Index = 16#7F11; PWM Error Code(axis 4).SubIndex = 0; PWM Error Code(axis 4).Size = 16; PWM Error Code(axis 4).Offset = 0; PWM Error Code(axis 4).DependOnSlot = False; PWM Error Code(axis 4).DependOnSlotGroup = False; RxTxPdo.NumberofExcludes = 0; RxTxPdo.NumberofEntries = 6; RxTxPdo.Index = 16#1B40; RxTxPdo.Fixed = False; RxTxPdo.Mandatory = False; RxTxPdo.Virtual = False; RxTxPdo.Sm = 3; RxTxPdo.Su = 3; RxTxPdo.Name = 'Inputs'; RxTxPdo.DependOnSlot = False; RxTxPdo.DependOnSlotGroup = False; RxTxPdo.OverwrittenByModule = False; Error Code(axis 5).Index = 16#803F; Error Code(axis 5).SubIndex = 0; Error Code(axis 5).Size = 16; Error Code(axis 5).Offset = 0; Error Code(axis 5).DependOnSlot = False; Error Code(axis 5).DependOnSlotGroup = False; Statusword(axis 5).Index = 16#8041; Statusword(axis 5).SubIndex = 0; Statusword(axis 5).Size = 16; Statusword(axis 5).Offset = 0; Statusword(axis 5).DependOnSlot = False; Statusword(axis 5).DependOnSlotGroup = False; Modes of operation display(axis 5).Index = 16#8061; Modes of operation display(axis 5).SubIndex = 0; Modes of operation display(axis 5).Size = 8; Modes of operation display(axis 5).Offset = 0; Modes of operation display(axis 5).DependOnSlot = False; Modes of operation display(axis 5).DependOnSlotGroup = False; Position actual value(axis 5).Index = 16#8064;
            Position actual value(axis 5).SubIndex = 0; Position actual value(axis 5).Size = 32; Position actual value(axis 5).Offset = 0; Position actual value(axis 5).DependOnSlot = False; Position actual value(axis 5).DependOnSlotGroup = False; Encoder Z phase(axis 5).Index = 16#8705; Encoder Z phase(axis 5).SubIndex = 0; Encoder Z phase(axis 5).Size = 32; Encoder Z phase(axis 5).Offset = 0; Encoder Z phase(axis 5).DependOnSlot = False; Encoder Z phase(axis 5).DependOnSlotGroup = False; PWM Error Code(axis 5).Index = 16#8711; PWM Error Code(axis 5).SubIndex = 0; PWM Error Code(axis 5).Size = 16; PWM Error Code(axis 5).Offset = 0; PWM Error Code(axis 5).DependOnSlot = False; PWM Error Code(axis 5).DependOnSlotGroup = False; RxTxPdo.NumberofExcludes = 0; RxTxPdo.NumberofEntries = 6; RxTxPdo.Index = 16#1B50; RxTxPdo.Fixed = False; RxTxPdo.Mandatory = False; RxTxPdo.Virtual = False; RxTxPdo.Sm = 3; RxTxPdo.Su = 3; RxTxPdo.Name = 'Inputs'; RxTxPdo.DependOnSlot = False; RxTxPdo.DependOnSlotGroup = False; RxTxPdo.OverwrittenByModule = False; Error Code(axis 6).Index = 16#883F; Error Code(axis 6).SubIndex = 0; Error Code(axis 6).Size = 16; Error Code(axis 6).Offset = 0; Error Code(axis 6).DependOnSlot = False; Error Code(axis 6).DependOnSlotGroup = False; Statusword(axis 6).Index = 16#8841; Statusword(axis 6).SubIndex = 0; Statusword(axis 6).Size = 16; Statusword(axis 6).Offset = 0; Statusword(axis 6).DependOnSlot = False;
            Statusword(axis 6).DependOnSlotGroup = False; Modes of operation display(axis 6).Index = 16#8861; Modes of operation display(axis 6).SubIndex = 0; Modes of operation display(axis 6).Size = 8; Modes of operation display(axis 6).Offset = 0; Modes of operation display(axis 6).DependOnSlot = False; Modes of operation display(axis 6).DependOnSlotGroup = False; Position actual value(axis 6).Index = 16#8864; Position actual value(axis 6).SubIndex = 0; Position actual value(axis 6).Size = 32; Position actual value(axis 6).Offset = 0; Position actual value(axis 6).DependOnSlot = False; Position actual value(axis 6).DependOnSlotGroup = False; Encoder Z phase(axis 6).Index = 16#8F05; Encoder Z phase(axis 6).SubIndex = 0; Encoder Z phase(axis 6).Size = 32; Encoder Z phase(axis 6).Offset = 0; Encoder Z phase(axis 6).DependOnSlot = False; Encoder Z phase(axis 6).DependOnSlotGroup = False; PWM Error Code(axis 6).Index = 16#8F11; PWM Error Code(axis 6).SubIndex = 0; PWM Error Code(axis 6).Size = 16; PWM Error Code(axis 6).Offset = 0; PWM Error Code(axis 6).DependOnSlot = False; PWM Error Code(axis 6).DependOnSlotGroup = False; RxTxPdo.NumberofExcludes = 0; RxTxPdo.NumberofEntries = 2; RxTxPdo.Index = 16#1B60; RxTxPdo.Fixed = False; RxTxPdo.Mandatory = False; RxTxPdo.Virtual = False; RxTxPdo.Sm = 3; RxTxPdo.Su = 3; RxTxPdo.Name = 'Inputs'; RxTxPdo.DependOnSlot = False; RxTxPdo.DependOnSlotGroup = False; RxTxPdo.OverwrittenByModule = False; High-speed comparison output status.Index = 16#6706; High-speed comparison output status.SubIndex = 0; High-speed comparison output status.Size = 8;
            High-speed comparison output status.Offset = 0; High-speed comparison output status.DependOnSlot = False; High-speed comparison output status.DependOnSlotGroup = False; PWM Output Enable Status.Index = 16#6710; PWM Output Enable Status.SubIndex = 0; PWM Output Enable Status.Size = 8; PWM Output Enable Status.Offset = 0; PWM Output Enable Status.DependOnSlot = False; PWM Output Enable Status.DependOnSlotGroup = False; RxTxPdo.NumberofExcludes = 0; RxTxPdo.NumberofEntries = 25; RxTxPdo.Index = 16#1A00; RxTxPdo.Fixed = True; RxTxPdo.Mandatory = True; RxTxPdo.Virtual = False; RxTxPdo.Sm = 3; RxTxPdo.Su = 0; RxTxPdo.Name = 'Inputs process data mapping'; RxTxPdo.DependOnSlot = True; RxTxPdo.DependOnSlotGroup = False; RxTxPdo.OverwrittenByModule = True; AI0.Index = 16#6000; AI0.SubIndex = 1; AI0.Size = 16; AI0.Offset = 0; AI0.DependOnSlot = True; AI0.DependOnSlotGroup = False; X0.Index = 16#6000; X0.SubIndex = 2; X0.Size = 1; X0.Offset = 0; X0.DependOnSlot = True; X0.DependOnSlotGroup = False; X1.Index = 16#6000; X1.SubIndex = 3; X1.Size = 1; X1.Offset = 0; X1.DependOnSlot = True; X1.DependOnSlotGroup = False; X2.Index = 16#6000;
            X2.SubIndex = 4; X2.Size = 1; X2.Offset = 0; X2.DependOnSlot = True; X2.DependOnSlotGroup = False; X3.Index = 16#6000; X3.SubIndex = 5; X3.Size = 1; X3.Offset = 0; X3.DependOnSlot = True; X3.DependOnSlotGroup = False; X4.Index = 16#6000; X4.SubIndex = 6; X4.Size = 1; X4.Offset = 0; X4.DependOnSlot = True; X4.DependOnSlotGroup = False; X5.Index = 16#6000; X5.SubIndex = 7; X5.Size = 1; X5.Offset = 0; X5.DependOnSlot = True; X5.DependOnSlotGroup = False; X6.Index = 16#6000; X6.SubIndex = 8; X6.Size = 1; X6.Offset = 0; X6.DependOnSlot = True; X6.DependOnSlotGroup = False; X7.Index = 16#6000; X7.SubIndex = 9; X7.Size = 1; X7.Offset = 0; X7.DependOnSlot = True; X7.DependOnSlotGroup = False; X8.Index = 16#6000; X8.SubIndex = 10; X8.Size = 1; X8.Offset = 0; X8.DependOnSlot = True;
            X8.DependOnSlotGroup = False; X9.Index = 16#6000; X9.SubIndex = 11; X9.Size = 1; X9.Offset = 0; X9.DependOnSlot = True; X9.DependOnSlotGroup = False; X10.Index = 16#6000; X10.SubIndex = 12; X10.Size = 1; X10.Offset = 0; X10.DependOnSlot = True; X10.DependOnSlotGroup = False; X11.Index = 16#6000; X11.SubIndex = 13; X11.Size = 1; X11.Offset = 0; X11.DependOnSlot = True; X11.DependOnSlotGroup = False; X12.Index = 16#6000; X12.SubIndex = 14; X12.Size = 1; X12.Offset = 0; X12.DependOnSlot = True; X12.DependOnSlotGroup = False; X13.Index = 16#6000; X13.SubIndex = 15; X13.Size = 1; X13.Offset = 0; X13.DependOnSlot = True; X13.DependOnSlotGroup = False; X14.Index = 16#6000; X14.SubIndex = 16; X14.Size = 1; X14.Offset = 0; X14.DependOnSlot = True; X14.DependOnSlotGroup = False; X15.Index = 16#6000; X15.SubIndex = 17; X15.Size = 1;
            X15.Offset = 0; X15.DependOnSlot = True; X15.DependOnSlotGroup = False; X16.Index = 16#6000; X16.SubIndex = 18; X16.Size = 1; X16.Offset = 0; X16.DependOnSlot = True; X16.DependOnSlotGroup = False; X17.Index = 16#6000; X17.SubIndex = 19; X17.Size = 1; X17.Offset = 0; X17.DependOnSlot = True; X17.DependOnSlotGroup = False; X18.Index = 16#6000; X18.SubIndex = 20; X18.Size = 1; X18.Offset = 0; X18.DependOnSlot = True; X18.DependOnSlotGroup = False; X19.Index = 16#6000; X19.SubIndex = 21; X19.Size = 1; X19.Offset = 0; X19.DependOnSlot = True; X19.DependOnSlotGroup = False; X20.Index = 16#6000; X20.SubIndex = 22; X20.Size = 1; X20.Offset = 0; X20.DependOnSlot = True; X20.DependOnSlotGroup = False; X21.Index = 16#6000; X21.SubIndex = 23; X21.Size = 1; X21.Offset = 0; X21.DependOnSlot = True; X21.DependOnSlotGroup = False; X22.Index = 16#6000;
            X22.SubIndex = 24; X22.Size = 1; X22.Offset = 0; X22.DependOnSlot = True; X22.DependOnSlotGroup = False; X23.Index = 16#6000; X23.SubIndex = 25; X23.Size = 1; X23.Offset = 0; X23.DependOnSlot = True; X23.DependOnSlotGroup = False; Controlword(axis 1).Name = 'Controlword(axis 1)'; Controlword(axis 1).DataType = 'UINT'; Controlword(axis 1).Default = ''; Controlword(axis 1).Comment = ''; Modes of operation(axis 1).Name = 'Modes of operation(axis 1)'; Modes of operation(axis 1).DataType = 'SINT'; Modes of operation(axis 1).Default = ''; Modes of operation(axis 1).Comment = ''; Target position(axis 1).Name = 'Target position(axis 1)'; Target position(axis 1).DataType = 'DINT'; Target position(axis 1).Default = ''; Target position(axis 1).Comment = ''; High-speed comparison 1(axis 1).Name = 'High-speed comparison 1(axis 1)'; High-speed comparison 1(axis 1).DataType = 'DINT'; High-speed comparison 1(axis 1).Default = ''; High-speed comparison 1(axis 1).Comment = ''; High-speed comparison 2(axis 1).Name = 'High-speed comparison 2(axis 1)'; High-speed comparison 2(axis 1).DataType = 'DINT'; High-speed comparison 2(axis 1).Default = ''; High-speed comparison 2(axis 1).Comment = ''; PWM Duty(axis 1).Name = 'PWM Duty(axis 1)'; PWM Duty(axis 1).DataType = 'USINT'; PWM Duty(axis 1).Default = ''; PWM Duty(axis 1).Comment = ''; PWM Freq(axis 1).Name = 'PWM Freq(axis 1)'; PWM Freq(axis 1).DataType = 'UDINT'; PWM Freq(axis 1).Default = ''; PWM Freq(axis 1).Comment = ''; Controlword(axis 2).Name = 'Controlword(axis 2)';
            Controlword(axis 2).DataType = 'UINT'; Controlword(axis 2).Default = ''; Controlword(axis 2).Comment = ''; Modes of operation(axis 2).Name = 'Modes of operation(axis 2)'; Modes of operation(axis 2).DataType = 'SINT'; Modes of operation(axis 2).Default = ''; Modes of operation(axis 2).Comment = ''; Target position(axis 2).Name = 'Target position(axis 2)'; Target position(axis 2).DataType = 'DINT'; Target position(axis 2).Default = ''; Target position(axis 2).Comment = ''; High-speed comparison 1(axis 2).Name = 'High-speed comparison 1(axis 2)'; High-speed comparison 1(axis 2).DataType = 'DINT'; High-speed comparison 1(axis 2).Default = ''; High-speed comparison 1(axis 2).Comment = ''; High-speed comparison 2(axis 2).Name = 'High-speed comparison 2(axis 2)'; High-speed comparison 2(axis 2).DataType = 'DINT'; High-speed comparison 2(axis 2).Default = ''; High-speed comparison 2(axis 2).Comment = ''; PWM Duty(axis 2).Name = 'PWM Duty(axis 2)'; PWM Duty(axis 2).DataType = 'USINT'; PWM Duty(axis 2).Default = ''; PWM Duty(axis 2).Comment = ''; PWM Freq(axis 2).Name = 'PWM Freq(axis 2)'; PWM Freq(axis 2).DataType = 'UDINT'; PWM Freq(axis 2).Default = ''; PWM Freq(axis 2).Comment = ''; Controlword(axis 3).Name = 'Controlword(axis 3)'; Controlword(axis 3).DataType = 'UINT'; Controlword(axis 3).Default = ''; Controlword(axis 3).Comment = ''; Modes of operation(axis 3).Name = 'Modes of operation(axis 3)'; Modes of operation(axis 3).DataType = 'SINT'; Modes of operation(axis 3).Default = ''; Modes of operation(axis 3).Comment = ''; Target position(axis 3).Name = 'Target position(axis 3)'; Target position(axis 3).DataType = 'DINT'; Target position(axis 3).Default = ''; Target position(axis 3).Comment = ''; High-speed comparison 1(axis 3).Name = 'High-speed comparison 1(axis 3)';
            High-speed comparison 1(axis 3).DataType = 'DINT'; High-speed comparison 1(axis 3).Default = ''; High-speed comparison 1(axis 3).Comment = ''; High-speed comparison 2(axis 3).Name = 'High-speed comparison 2(axis 3)'; High-speed comparison 2(axis 3).DataType = 'DINT'; High-speed comparison 2(axis 3).Default = ''; High-speed comparison 2(axis 3).Comment = ''; PWM Duty(axis 3).Name = 'PWM Duty(axis 3)'; PWM Duty(axis 3).DataType = 'USINT'; PWM Duty(axis 3).Default = ''; PWM Duty(axis 3).Comment = ''; PWM Freq(axis 3).Name = 'PWM Freq(axis 3)'; PWM Freq(axis 3).DataType = 'UDINT'; PWM Freq(axis 3).Default = ''; PWM Freq(axis 3).Comment = ''; Controlword(axis 4).Name = 'Controlword(axis 4)'; Controlword(axis 4).DataType = 'UINT'; Controlword(axis 4).Default = ''; Controlword(axis 4).Comment = ''; Modes of operation(axis 4).Name = 'Modes of operation(axis 4)'; Modes of operation(axis 4).DataType = 'SINT'; Modes of operation(axis 4).Default = ''; Modes of operation(axis 4).Comment = ''; Target position(axis 4).Name = 'Target position(axis 4)'; Target position(axis 4).DataType = 'DINT'; Target position(axis 4).Default = ''; Target position(axis 4).Comment = ''; High-speed comparison 1(axis 4).Name = 'High-speed comparison 1(axis 4)'; High-speed comparison 1(axis 4).DataType = 'DINT'; High-speed comparison 1(axis 4).Default = ''; High-speed comparison 1(axis 4).Comment = ''; High-speed comparison 2(axis 4).Name = 'High-speed comparison 2(axis 4)'; High-speed comparison 2(axis 4).DataType = 'DINT'; High-speed comparison 2(axis 4).Default = ''; High-speed comparison 2(axis 4).Comment = ''; PWM Duty(axis 4).Name = 'PWM Duty(axis 4)'; PWM Duty(axis 4).DataType = 'USINT'; PWM Duty(axis 4).Default = ''; PWM Duty(axis 4).Comment = ''; PWM Freq(axis 4).Name = 'PWM Freq(axis 4)';
            PWM Freq(axis 4).DataType = 'UDINT'; PWM Freq(axis 4).Default = ''; PWM Freq(axis 4).Comment = ''; Controlword(axis 5).Name = 'Controlword(axis 5)'; Controlword(axis 5).DataType = 'UINT'; Controlword(axis 5).Default = ''; Controlword(axis 5).Comment = ''; Modes of operation(axis 5).Name = 'Modes of operation(axis 5)'; Modes of operation(axis 5).DataType = 'SINT'; Modes of operation(axis 5).Default = ''; Modes of operation(axis 5).Comment = ''; Target position(axis 5).Name = 'Target position(axis 5)'; Target position(axis 5).DataType = 'DINT'; Target position(axis 5).Default = ''; Target position(axis 5).Comment = ''; High-speed comparison 1(axis 5).Name = 'High-speed comparison 1(axis 5)'; High-speed comparison 1(axis 5).DataType = 'DINT'; High-speed comparison 1(axis 5).Default = ''; High-speed comparison 1(axis 5).Comment = ''; High-speed comparison 2(axis 5).Name = 'High-speed comparison 2(axis 5)'; High-speed comparison 2(axis 5).DataType = 'DINT'; High-speed comparison 2(axis 5).Default = ''; High-speed comparison 2(axis 5).Comment = ''; PWM Duty(axis 5).Name = 'PWM Duty(axis 5)'; PWM Duty(axis 5).DataType = 'USINT'; PWM Duty(axis 5).Default = ''; PWM Duty(axis 5).Comment = ''; PWM Freq(axis 5).Name = 'PWM Freq(axis 5)'; PWM Freq(axis 5).DataType = 'UDINT'; PWM Freq(axis 5).Default = ''; PWM Freq(axis 5).Comment = ''; Controlword(axis 6).Name = 'Controlword(axis 6)'; Controlword(axis 6).DataType = 'UINT'; Controlword(axis 6).Default = ''; Controlword(axis 6).Comment = ''; Modes of operation(axis 6).Name = 'Modes of operation(axis 6)'; Modes of operation(axis 6).DataType = 'SINT'; Modes of operation(axis 6).Default = ''; Modes of operation(axis 6).Comment = ''; Target position(axis 6).Name = 'Target position(axis 6)';
            Target position(axis 6).DataType = 'DINT'; Target position(axis 6).Default = ''; Target position(axis 6).Comment = ''; High-speed comparison 1(axis 6).Name = 'High-speed comparison 1(axis 6)'; High-speed comparison 1(axis 6).DataType = 'DINT'; High-speed comparison 1(axis 6).Default = ''; High-speed comparison 1(axis 6).Comment = ''; High-speed comparison 2(axis 6).Name = 'High-speed comparison 2(axis 6)'; High-speed comparison 2(axis 6).DataType = 'DINT'; High-speed comparison 2(axis 6).Default = ''; High-speed comparison 2(axis 6).Comment = ''; PWM Duty(axis 6).Name = 'PWM Duty(axis 6)'; PWM Duty(axis 6).DataType = 'USINT'; PWM Duty(axis 6).Default = ''; PWM Duty(axis 6).Comment = ''; PWM Freq(axis 6).Name = 'PWM Freq(axis 6)'; PWM Freq(axis 6).DataType = 'UDINT'; PWM Freq(axis 6).Default = ''; PWM Freq(axis 6).Comment = ''; High-speed comparison 1 switch.Name = 'High-speed comparison 1 switch'; High-speed comparison 1 switch.DataType = 'USINT'; High-speed comparison 1 switch.Default = ''; High-speed comparison 1 switch.Comment = ''; High-speed comparison 2 switch.Name = 'High-speed comparison 2 switch'; High-speed comparison 2 switch.DataType = 'USINT'; High-speed comparison 2 switch.Default = ''; High-speed comparison 2 switch.Comment = ''; PWM Output Enable.Name = 'PWM Output Enable'; PWM Output Enable.DataType = 'USINT'; PWM Output Enable.Default = ''; PWM Output Enable.Comment = ''; AO0.Name = 'AO0'; AO0.DataType = 'UINT'; AO0.Default = ''; AO0.Comment = ''; Y0.Name = 'Y0'; Y0.DataType = 'BOOL'; Y0.Default = ''; Y0.Comment = ''; Y1.Name = 'Y1';
            Y1.DataType = 'BOOL'; Y1.Default = ''; Y1.Comment = ''; Y2.Name = 'Y2'; Y2.DataType = 'BOOL'; Y2.Default = ''; Y2.Comment = ''; Y3.Name = 'Y3'; Y3.DataType = 'BOOL'; Y3.Default = ''; Y3.Comment = ''; Y4.Name = 'Y4'; Y4.DataType = 'BOOL'; Y4.Default = ''; Y4.Comment = ''; Y5.Name = 'Y5'; Y5.DataType = 'BOOL'; Y5.Default = ''; Y5.Comment = ''; Y6.Name = 'Y6'; Y6.DataType = 'BOOL'; Y6.Default = ''; Y6.Comment = ''; Y7.Name = 'Y7'; Y7.DataType = 'BOOL'; Y7.Default = ''; Y7.Comment = ''; Y8.Name = 'Y8'; Y8.DataType = 'BOOL'; Y8.Default = ''; Y8.Comment = ''; Y9.Name = 'Y9'; Y9.DataType = 'BOOL'; Y9.Default = ''; Y9.Comment = ''; Y10.Name = 'Y10'; Y10.DataType = 'BOOL'; Y10.Default = ''; Y10.Comment = ''; Y11.Name = 'Y11';
            Y11.DataType = 'BOOL'; Y11.Default = ''; Y11.Comment = ''; Y12.Name = 'Y12'; Y12.DataType = 'BOOL'; Y12.Default = ''; Y12.Comment = ''; Y13.Name = 'Y13'; Y13.DataType = 'BOOL'; Y13.Default = ''; Y13.Comment = ''; Y14.Name = 'Y14'; Y14.DataType = 'BOOL'; Y14.Default = ''; Y14.Comment = ''; Y15.Name = 'Y15'; Y15.DataType = 'BOOL'; Y15.Default = ''; Y15.Comment = ''; Error Code(axis 1).Name = 'Error Code(axis 1)'; Error Code(axis 1).DataType = 'UINT'; Error Code(axis 1).Default = ''; Error Code(axis 1).Comment = ''; Statusword(axis 1).Name = 'Statusword(axis 1)'; Statusword(axis 1).DataType = 'UINT'; Statusword(axis 1).Default = ''; Statusword(axis 1).Comment = ''; Modes of operation display(axis 1).Name = 'Modes of operation display(axis 1)'; Modes of operation display(axis 1).DataType = 'SINT'; Modes of operation display(axis 1).Default = ''; Modes of operation display(axis 1).Comment = ''; Position actual value(axis 1).Name = 'Position actual value(axis 1)'; Position actual value(axis 1).DataType = 'DINT'; Position actual value(axis 1).Default = ''; Position actual value(axis 1).Comment = ''; Encoder Z phase(axis 1).Name = 'Encoder Z phase(axis 1)'; Encoder Z phase(axis 1).DataType = 'DINT'; Encoder Z phase(axis 1).Default = ''; Encoder Z phase(axis 1).Comment = ''; PWM Error Code(axis 1).Name = 'PWM Error Code(axis 1)';
            PWM Error Code(axis 1).DataType = 'UINT'; PWM Error Code(axis 1).Default = ''; PWM Error Code(axis 1).Comment = ''; Error Code(axis 2).Name = 'Error Code(axis 2)'; Error Code(axis 2).DataType = 'UINT'; Error Code(axis 2).Default = ''; Error Code(axis 2).Comment = ''; Statusword(axis 2).Name = 'Statusword(axis 2)'; Statusword(axis 2).DataType = 'UINT'; Statusword(axis 2).Default = ''; Statusword(axis 2).Comment = ''; Modes of operation display(axis 2).Name = 'Modes of operation display(axis 2)'; Modes of operation display(axis 2).DataType = 'SINT'; Modes of operation display(axis 2).Default = ''; Modes of operation display(axis 2).Comment = ''; Position actual value(axis 2).Name = 'Position actual value(axis 2)'; Position actual value(axis 2).DataType = 'DINT'; Position actual value(axis 2).Default = ''; Position actual value(axis 2).Comment = ''; Encoder Z phase(axis 2).Name = 'Encoder Z phase(axis 2)'; Encoder Z phase(axis 2).DataType = 'DINT'; Encoder Z phase(axis 2).Default = ''; Encoder Z phase(axis 2).Comment = ''; PWM Error Code(axis 2).Name = 'PWM Error Code(axis 2)'; PWM Error Code(axis 2).DataType = 'UINT'; PWM Error Code(axis 2).Default = ''; PWM Error Code(axis 2).Comment = ''; Error Code(axis 3).Name = 'Error Code(axis 3)'; Error Code(axis 3).DataType = 'UINT'; Error Code(axis 3).Default = ''; Error Code(axis 3).Comment = ''; Statusword(axis 3).Name = 'Statusword(axis 3)'; Statusword(axis 3).DataType = 'UINT'; Statusword(axis 3).Default = ''; Statusword(axis 3).Comment = ''; Modes of operation display(axis 3).Name = 'Modes of operation display(axis 3)'; Modes of operation display(axis 3).DataType = 'SINT'; Modes of operation display(axis 3).Default = ''; Modes of operation display(axis 3).Comment = ''; Position actual value(axis 3).Name = 'Position actual value(axis 3)';
            Position actual value(axis 3).DataType = 'DINT'; Position actual value(axis 3).Default = ''; Position actual value(axis 3).Comment = ''; Encoder Z phase(axis 3).Name = 'Encoder Z phase(axis 3)'; Encoder Z phase(axis 3).DataType = 'DINT'; Encoder Z phase(axis 3).Default = ''; Encoder Z phase(axis 3).Comment = ''; PWM Error Code(axis 3).Name = 'PWM Error Code(axis 3)'; PWM Error Code(axis 3).DataType = 'UINT'; PWM Error Code(axis 3).Default = ''; PWM Error Code(axis 3).Comment = ''; Error Code(axis 4).Name = 'Error Code(axis 4)'; Error Code(axis 4).DataType = 'UINT'; Error Code(axis 4).Default = ''; Error Code(axis 4).Comment = ''; Statusword(axis 4).Name = 'Statusword(axis 4)'; Statusword(axis 4).DataType = 'UINT'; Statusword(axis 4).Default = ''; Statusword(axis 4).Comment = ''; Modes of operation display(axis 4).Name = 'Modes of operation display(axis 4)'; Modes of operation display(axis 4).DataType = 'SINT'; Modes of operation display(axis 4).Default = ''; Modes of operation display(axis 4).Comment = ''; Position actual value(axis 4).Name = 'Position actual value(axis 4)'; Position actual value(axis 4).DataType = 'DINT'; Position actual value(axis 4).Default = ''; Position actual value(axis 4).Comment = ''; Encoder Z phase(axis 4).Name = 'Encoder Z phase(axis 4)'; Encoder Z phase(axis 4).DataType = 'DINT'; Encoder Z phase(axis 4).Default = ''; Encoder Z phase(axis 4).Comment = ''; PWM Error Code(axis 4).Name = 'PWM Error Code(axis 4)'; PWM Error Code(axis 4).DataType = 'UINT'; PWM Error Code(axis 4).Default = ''; PWM Error Code(axis 4).Comment = ''; Error Code(axis 5).Name = 'Error Code(axis 5)'; Error Code(axis 5).DataType = 'UINT'; Error Code(axis 5).Default = ''; Error Code(axis 5).Comment = ''; Statusword(axis 5).Name = 'Statusword(axis 5)';
            Statusword(axis 5).DataType = 'UINT'; Statusword(axis 5).Default = ''; Statusword(axis 5).Comment = ''; Modes of operation display(axis 5).Name = 'Modes of operation display(axis 5)'; Modes of operation display(axis 5).DataType = 'SINT'; Modes of operation display(axis 5).Default = ''; Modes of operation display(axis 5).Comment = ''; Position actual value(axis 5).Name = 'Position actual value(axis 5)'; Position actual value(axis 5).DataType = 'DINT'; Position actual value(axis 5).Default = ''; Position actual value(axis 5).Comment = ''; Encoder Z phase(axis 5).Name = 'Encoder Z phase(axis 5)'; Encoder Z phase(axis 5).DataType = 'DINT'; Encoder Z phase(axis 5).Default = ''; Encoder Z phase(axis 5).Comment = ''; PWM Error Code(axis 5).Name = 'PWM Error Code(axis 5)'; PWM Error Code(axis 5).DataType = 'UINT'; PWM Error Code(axis 5).Default = ''; PWM Error Code(axis 5).Comment = ''; Error Code(axis 6).Name = 'Error Code(axis 6)'; Error Code(axis 6).DataType = 'UINT'; Error Code(axis 6).Default = ''; Error Code(axis 6).Comment = ''; Statusword(axis 6).Name = 'Statusword(axis 6)'; Statusword(axis 6).DataType = 'UINT'; Statusword(axis 6).Default = ''; Statusword(axis 6).Comment = ''; Modes of operation display(axis 6).Name = 'Modes of operation display(axis 6)'; Modes of operation display(axis 6).DataType = 'SINT'; Modes of operation display(axis 6).Default = ''; Modes of operation display(axis 6).Comment = ''; Position actual value(axis 6).Name = 'Position actual value(axis 6)'; Position actual value(axis 6).DataType = 'DINT'; Position actual value(axis 6).Default = ''; Position actual value(axis 6).Comment = ''; Encoder Z phase(axis 6).Name = 'Encoder Z phase(axis 6)'; Encoder Z phase(axis 6).DataType = 'DINT'; Encoder Z phase(axis 6).Default = ''; Encoder Z phase(axis 6).Comment = ''; PWM Error Code(axis 6).Name = 'PWM Error Code(axis 6)';
            PWM Error Code(axis 6).DataType = 'UINT'; PWM Error Code(axis 6).Default = ''; PWM Error Code(axis 6).Comment = ''; High-speed comparison output status.Name = 'High-speed comparison output status'; High-speed comparison output status.DataType = 'USINT'; High-speed comparison output status.Default = ''; High-speed comparison output status.Comment = ''; PWM Output Enable Status.Name = 'PWM Output Enable Status'; PWM Output Enable Status.DataType = 'USINT'; PWM Output Enable Status.Default = ''; PWM Output Enable Status.Comment = ''; AI0.Name = 'AI0'; AI0.DataType = 'UINT'; AI0.Default = ''; AI0.Comment = ''; X0.Name = 'X0'; X0.DataType = 'BOOL'; X0.Default = ''; X0.Comment = ''; X1.Name = 'X1'; X1.DataType = 'BOOL'; X1.Default = ''; X1.Comment = ''; X2.Name = 'X2'; X2.DataType = 'BOOL'; X2.Default = ''; X2.Comment = ''; X3.Name = 'X3'; X3.DataType = 'BOOL'; X3.Default = ''; X3.Comment = ''; X4.Name = 'X4'; X4.DataType = 'BOOL'; X4.Default = ''; X4.Comment = ''; X5.Name = 'X5'; X5.DataType = 'BOOL'; X5.Default = ''; X5.Comment = ''; X6.Name = 'X6';
            X6.DataType = 'BOOL'; X6.Default = ''; X6.Comment = ''; X7.Name = 'X7'; X7.DataType = 'BOOL'; X7.Default = ''; X7.Comment = ''; X8.Name = 'X8'; X8.DataType = 'BOOL'; X8.Default = ''; X8.Comment = ''; X9.Name = 'X9'; X9.DataType = 'BOOL'; X9.Default = ''; X9.Comment = ''; X10.Name = 'X10'; X10.DataType = 'BOOL'; X10.Default = ''; X10.Comment = ''; X11.Name = 'X11'; X11.DataType = 'BOOL'; X11.Default = ''; X11.Comment = ''; X12.Name = 'X12'; X12.DataType = 'BOOL'; X12.Default = ''; X12.Comment = ''; X13.Name = 'X13'; X13.DataType = 'BOOL'; X13.Default = ''; X13.Comment = ''; X14.Name = 'X14'; X14.DataType = 'BOOL'; X14.Default = ''; X14.Comment = ''; X15.Name = 'X15'; X15.DataType = 'BOOL'; X15.Default = ''; X15.Comment = ''; X16.Name = 'X16';
            X16.DataType = 'BOOL'; X16.Default = ''; X16.Comment = ''; X17.Name = 'X17'; X17.DataType = 'BOOL'; X17.Default = ''; X17.Comment = ''; X18.Name = 'X18'; X18.DataType = 'BOOL'; X18.Default = ''; X18.Comment = ''; X19.Name = 'X19'; X19.DataType = 'BOOL'; X19.Default = ''; X19.Comment = ''; X20.Name = 'X20'; X20.DataType = 'BOOL'; X20.Default = ''; X20.Comment = ''; X21.Name = 'X21'; X21.DataType = 'BOOL'; X21.Default = ''; X21.Comment = ''; X22.Name = 'X22'; X22.DataType = 'BOOL'; X22.Default = ''; X22.Comment = ''; X23.Name = 'X23'; X23.DataType = 'BOOL'; X23.Default = ''; X23.Comment = ''
          unmapped channels: Controlword(axis 1), Modes of operation(axis 1), Target position(axis 1), High-speed comparison 1(axis 1), High-speed comparison 2(axis 1), PWM Duty(axis 1), PWM Freq(axis 1), Controlword(axis 2), Modes of operation(axis 2), Target position(axis 2), High-speed comparison 1(axis 2), High-speed comparison 2(axis 2), PWM Duty(axis 2), PWM Freq(axis 2), Controlword(axis 3), Modes of operation(axis 3), Target position(axis 3), High-speed comparison 1(axis 3), High-speed comparison 2(axis 3), PWM Duty(axis 3), PWM Freq(axis 3), Controlword(axis 4), Modes of operation(axis 4), Target position(axis 4), High-speed comparison 1(axis 4), High-speed comparison 2(axis 4), PWM Duty(axis 4), PWM Freq(axis 4), Controlword(axis 5), Modes of operation(axis 5), Target position(axis 5), High-speed comparison 1(axis 5), High-speed comparison 2(axis 5), PWM Duty(axis 5), PWM Freq(axis 5), Controlword(axis 6), Modes of operation(axis 6), Target position(axis 6), High-speed comparison 1(axis 6), High-speed comparison 2(axis 6),
            PWM Duty(axis 6), PWM Freq(axis 6), High-speed comparison 1 switch, High-speed comparison 2 switch, PWM Output Enable, Error Code(axis 1), Statusword(axis 1), Modes of operation display(axis 1), Position actual value(axis 1), Encoder Z phase(axis 1), PWM Error Code(axis 1), Error Code(axis 2), Statusword(axis 2), Modes of operation display(axis 2), Position actual value(axis 2), Encoder Z phase(axis 2), PWM Error Code(axis 2), Error Code(axis 3), Statusword(axis 3), Modes of operation display(axis 3), Position actual value(axis 3), Encoder Z phase(axis 3), PWM Error Code(axis 3), Error Code(axis 4), Statusword(axis 4), Modes of operation display(axis 4), Position actual value(axis 4), Encoder Z phase(axis 4), PWM Error Code(axis 4), Error Code(axis 5), Statusword(axis 5), Modes of operation display(axis 5), Position actual value(axis 5), Encoder Z phase(axis 5), PWM Error Code(axis 5), Error Code(axis 6), Statusword(axis 6), Modes of operation display(axis 6), Position actual value(axis 6), Encoder Z phase(axis 6),
            PWM Error Code(axis 6), High-speed comparison output status, PWM Output Enable Status
        AXIS_1 : SM_Drive_EtherCAT_JMC, 3S - Smart Software Solutions GmbH, order no. 0, version 4.6.1.0
            settings: wDriveID = 16; AdrOffset_8010 = 304; BitOffset_8010 = 0; BitLength_8010 = 16; Address_8010 = '%QW152'; Type_8010 = 'UINT'; AddressPointer_8010 = ADR(%QW152); AdrOffset_8020 = 308; BitOffset_8020 = 0; BitLength_8020 = 32; Address_8020 = '%QD77'; Type_8020 = 'DINT'; AddressPointer_8020 = ADR(%QD77); AdrOffset_8030 = 4294967295; BitOffset_8030 = 0; BitLength_8030 = 0; Address_8030 = ''; Type_8030 = ''; AddressPointer_8030 = 0; AdrOffset_8040 = 4294967295; BitOffset_8040 = 0; BitLength_8040 = 0; Address_8040 = ''; Type_8040 = ''; AddressPointer_8040 = 0; AdrOffset_8050 = 306; BitOffset_8050 = 0; BitLength_8050 = 8; Address_8050 = '%QB306'; Type_8050 = 'SINT'; AddressPointer_8050 = ADR(%QB306); AdrOffset_8060 = 4294967295; BitOffset_8060 = 0; BitLength_8060 = 0; Address_8060 = ''; Type_8060 = ''; AddressPointer_8060 = 0; AdrOffset_8070 = 4294967295; BitOffset_8070 = 0; BitLength_8070 = 0;
              Address_8070 = ''; Type_8070 = ''; AddressPointer_8070 = 0; AdrOffset_8080 = 4294967295; BitOffset_8080 = 0; BitLength_8080 = 0; Address_8080 = ''; Type_8080 = ''; AddressPointer_8080 = 0; AdrOffset_8090 = 4294967295; BitOffset_8090 = 0; BitLength_8090 = 0; Address_8090 = ''; Type_8090 = ''; AddressPointer_8090 = 0; AdrOffset_8510 = 2; BitOffset_8510 = 0; BitLength_8510 = 16; Address_8510 = '%IW1'; Type_8510 = 'UINT'; AddressPointer_8510 = ADR(%IW1); AdrOffset_8520 = 8; BitOffset_8520 = 0; BitLength_8520 = 32; Address_8520 = '%ID2'; Type_8520 = 'DINT'; AddressPointer_8520 = ADR(%ID2); AdrOffset_8530 = 4294967295; BitOffset_8530 = 0; BitLength_8530 = 0; Address_8530 = ''; Type_8530 = ''; AddressPointer_8530 = 0; AdrOffset_8540 = 4294967295; BitOffset_8540 = 0; BitLength_8540 = 0; Address_8540 = ''; Type_8540 = ''; AddressPointer_8540 = 0; AdrOffset_8550 = 4;
              BitOffset_8550 = 0; BitLength_8550 = 8; Address_8550 = '%IB4'; Type_8550 = 'SINT'; AddressPointer_8550 = ADR(%IB4); AdrOffset_8560 = 4294967295; BitOffset_8560 = 0; BitLength_8560 = 0; Address_8560 = ''; Type_8560 = ''; AddressPointer_8560 = 0; AdrOffset_8570 = 4294967295; BitOffset_8570 = 0; BitLength_8570 = 0; Address_8570 = ''; Type_8570 = ''; AddressPointer_8570 = 0; AdrOffset_8580 = 4294967295; BitOffset_8580 = 0; BitLength_8580 = 0; Address_8580 = ''; Type_8580 = ''; AddressPointer_8580 = 0; AdrOffset_8590 = 4294967295; BitOffset_8590 = 0; BitLength_8590 = 0; Address_8590 = ''; Type_8590 = ''; AddressPointer_8590 = 0; AdrOffset_8600 = 4294967295; BitOffset_8600 = 0; BitLength_8600 = 0; Address_8600 = ''; Type_8600 = ''; AddressPointer_8600 = 0; AdrOffset_8600 = 4294967295; BitOffset_8600 = 0; BitLength_8600 = 0; Address_8610 = ''; Type_8610 = '';
              AddressPointer_8610 = 0; AdrOffset_8620 = 4294967295; BitOffset_8620 = 0; BitLength_8620 = 0; Address_8620 = ''; Type_8620 = ''; AddressPointer_8620 = 0
        AXIS_2 : SM_Drive_EtherCAT_JMC, 3S - Smart Software Solutions GmbH, order no. 0, version 4.6.1.0
            settings: wDriveID = 17; AdrOffset_8010 = 328; BitOffset_8010 = 0; BitLength_8010 = 16; Address_8010 = '%QW164'; Type_8010 = 'UINT'; AddressPointer_8010 = ADR(%QW164); AdrOffset_8020 = 332; BitOffset_8020 = 0; BitLength_8020 = 32; Address_8020 = '%QD83'; Type_8020 = 'DINT'; AddressPointer_8020 = ADR(%QD83); AdrOffset_8030 = 4294967295; BitOffset_8030 = 0; BitLength_8030 = 0; Address_8030 = ''; Type_8030 = ''; AddressPointer_8030 = 0; AdrOffset_8040 = 4294967295; BitOffset_8040 = 0; BitLength_8040 = 0; Address_8040 = ''; Type_8040 = ''; AddressPointer_8040 = 0; AdrOffset_8050 = 330; BitOffset_8050 = 0; BitLength_8050 = 8; Address_8050 = '%QB330'; Type_8050 = 'SINT'; AddressPointer_8050 = ADR(%QB330); AdrOffset_8060 = 4294967295; BitOffset_8060 = 0; BitLength_8060 = 0; Address_8060 = ''; Type_8060 = ''; AddressPointer_8060 = 0; AdrOffset_8070 = 4294967295; BitOffset_8070 = 0; BitLength_8070 = 0;
              Address_8070 = ''; Type_8070 = ''; AddressPointer_8070 = 0; AdrOffset_8080 = 4294967295; BitOffset_8080 = 0; BitLength_8080 = 0; Address_8080 = ''; Type_8080 = ''; AddressPointer_8080 = 0; AdrOffset_8090 = 4294967295; BitOffset_8090 = 0; BitLength_8090 = 0; Address_8090 = ''; Type_8090 = ''; AddressPointer_8090 = 0; AdrOffset_8510 = 20; BitOffset_8510 = 0; BitLength_8510 = 16; Address_8510 = '%IW10'; Type_8510 = 'UINT'; AddressPointer_8510 = ADR(%IW10); AdrOffset_8520 = 24; BitOffset_8520 = 0; BitLength_8520 = 32; Address_8520 = '%ID6'; Type_8520 = 'DINT'; AddressPointer_8520 = ADR(%ID6); AdrOffset_8530 = 4294967295; BitOffset_8530 = 0; BitLength_8530 = 0; Address_8530 = ''; Type_8530 = ''; AddressPointer_8530 = 0; AdrOffset_8540 = 4294967295; BitOffset_8540 = 0; BitLength_8540 = 0; Address_8540 = ''; Type_8540 = ''; AddressPointer_8540 = 0; AdrOffset_8550 = 22;
              BitOffset_8550 = 0; BitLength_8550 = 8; Address_8550 = '%IB22'; Type_8550 = 'SINT'; AddressPointer_8550 = ADR(%IB22); AdrOffset_8560 = 4294967295; BitOffset_8560 = 0; BitLength_8560 = 0; Address_8560 = ''; Type_8560 = ''; AddressPointer_8560 = 0; AdrOffset_8570 = 4294967295; BitOffset_8570 = 0; BitLength_8570 = 0; Address_8570 = ''; Type_8570 = ''; AddressPointer_8570 = 0; AdrOffset_8580 = 4294967295; BitOffset_8580 = 0; BitLength_8580 = 0; Address_8580 = ''; Type_8580 = ''; AddressPointer_8580 = 0; AdrOffset_8590 = 4294967295; BitOffset_8590 = 0; BitLength_8590 = 0; Address_8590 = ''; Type_8590 = ''; AddressPointer_8590 = 0; AdrOffset_8600 = 4294967295; BitOffset_8600 = 0; BitLength_8600 = 0; Address_8600 = ''; Type_8600 = ''; AddressPointer_8600 = 0; AdrOffset_8600 = 4294967295; BitOffset_8600 = 0; BitLength_8600 = 0; Address_8610 = ''; Type_8610 = '';
              AddressPointer_8610 = 0; AdrOffset_8620 = 4294967295; BitOffset_8620 = 0; BitLength_8620 = 0; Address_8620 = ''; Type_8620 = ''; AddressPointer_8620 = 0
        AXIS_3 : SM_Drive_EtherCAT_JMC, 3S - Smart Software Solutions GmbH, order no. 0, version 4.6.1.0
            settings: wDriveID = 18; AdrOffset_8010 = 352; BitOffset_8010 = 0; BitLength_8010 = 16; Address_8010 = '%QW176'; Type_8010 = 'UINT'; AddressPointer_8010 = ADR(%QW176); AdrOffset_8020 = 356; BitOffset_8020 = 0; BitLength_8020 = 32; Address_8020 = '%QD89'; Type_8020 = 'DINT'; AddressPointer_8020 = ADR(%QD89); AdrOffset_8030 = 4294967295; BitOffset_8030 = 0; BitLength_8030 = 0; Address_8030 = ''; Type_8030 = ''; AddressPointer_8030 = 0; AdrOffset_8040 = 4294967295; BitOffset_8040 = 0; BitLength_8040 = 0; Address_8040 = ''; Type_8040 = ''; AddressPointer_8040 = 0; AdrOffset_8050 = 354; BitOffset_8050 = 0; BitLength_8050 = 8; Address_8050 = '%QB354'; Type_8050 = 'SINT'; AddressPointer_8050 = ADR(%QB354); AdrOffset_8060 = 4294967295; BitOffset_8060 = 0; BitLength_8060 = 0; Address_8060 = ''; Type_8060 = ''; AddressPointer_8060 = 0; AdrOffset_8070 = 4294967295; BitOffset_8070 = 0; BitLength_8070 = 0;
              Address_8070 = ''; Type_8070 = ''; AddressPointer_8070 = 0; AdrOffset_8080 = 4294967295; BitOffset_8080 = 0; BitLength_8080 = 0; Address_8080 = ''; Type_8080 = ''; AddressPointer_8080 = 0; AdrOffset_8090 = 4294967295; BitOffset_8090 = 0; BitLength_8090 = 0; Address_8090 = ''; Type_8090 = ''; AddressPointer_8090 = 0; AdrOffset_8510 = 36; BitOffset_8510 = 0; BitLength_8510 = 16; Address_8510 = '%IW18'; Type_8510 = 'UINT'; AddressPointer_8510 = ADR(%IW18); AdrOffset_8520 = 40; BitOffset_8520 = 0; BitLength_8520 = 32; Address_8520 = '%ID10'; Type_8520 = 'DINT'; AddressPointer_8520 = ADR(%ID10); AdrOffset_8530 = 4294967295; BitOffset_8530 = 0; BitLength_8530 = 0; Address_8530 = ''; Type_8530 = ''; AddressPointer_8530 = 0; AdrOffset_8540 = 4294967295; BitOffset_8540 = 0; BitLength_8540 = 0; Address_8540 = ''; Type_8540 = ''; AddressPointer_8540 = 0; AdrOffset_8550 = 38;
              BitOffset_8550 = 0; BitLength_8550 = 8; Address_8550 = '%IB38'; Type_8550 = 'SINT'; AddressPointer_8550 = ADR(%IB38); AdrOffset_8560 = 4294967295; BitOffset_8560 = 0; BitLength_8560 = 0; Address_8560 = ''; Type_8560 = ''; AddressPointer_8560 = 0; AdrOffset_8570 = 4294967295; BitOffset_8570 = 0; BitLength_8570 = 0; Address_8570 = ''; Type_8570 = ''; AddressPointer_8570 = 0; AdrOffset_8580 = 4294967295; BitOffset_8580 = 0; BitLength_8580 = 0; Address_8580 = ''; Type_8580 = ''; AddressPointer_8580 = 0; AdrOffset_8590 = 4294967295; BitOffset_8590 = 0; BitLength_8590 = 0; Address_8590 = ''; Type_8590 = ''; AddressPointer_8590 = 0; AdrOffset_8600 = 4294967295; BitOffset_8600 = 0; BitLength_8600 = 0; Address_8600 = ''; Type_8600 = ''; AddressPointer_8600 = 0; AdrOffset_8600 = 4294967295; BitOffset_8600 = 0; BitLength_8600 = 0; Address_8610 = ''; Type_8610 = '';
              AddressPointer_8610 = 0; AdrOffset_8620 = 4294967295; BitOffset_8620 = 0; BitLength_8620 = 0; Address_8620 = ''; Type_8620 = ''; AddressPointer_8620 = 0
        AXIS_4 : SM_Drive_EtherCAT_JMC, 3S - Smart Software Solutions GmbH, order no. 0, version 4.6.1.0
            settings: wDriveID = 19; AdrOffset_8010 = 376; BitOffset_8010 = 0; BitLength_8010 = 16; Address_8010 = '%QW188'; Type_8010 = 'UINT'; AddressPointer_8010 = ADR(%QW188); AdrOffset_8020 = 380; BitOffset_8020 = 0; BitLength_8020 = 32; Address_8020 = '%QD95'; Type_8020 = 'DINT'; AddressPointer_8020 = ADR(%QD95); AdrOffset_8030 = 4294967295; BitOffset_8030 = 0; BitLength_8030 = 0; Address_8030 = ''; Type_8030 = ''; AddressPointer_8030 = 0; AdrOffset_8040 = 4294967295; BitOffset_8040 = 0; BitLength_8040 = 0; Address_8040 = ''; Type_8040 = ''; AddressPointer_8040 = 0; AdrOffset_8050 = 378; BitOffset_8050 = 0; BitLength_8050 = 8; Address_8050 = '%QB378'; Type_8050 = 'SINT'; AddressPointer_8050 = ADR(%QB378); AdrOffset_8060 = 4294967295; BitOffset_8060 = 0; BitLength_8060 = 0; Address_8060 = ''; Type_8060 = ''; AddressPointer_8060 = 0; AdrOffset_8070 = 4294967295; BitOffset_8070 = 0; BitLength_8070 = 0;
              Address_8070 = ''; Type_8070 = ''; AddressPointer_8070 = 0; AdrOffset_8080 = 4294967295; BitOffset_8080 = 0; BitLength_8080 = 0; Address_8080 = ''; Type_8080 = ''; AddressPointer_8080 = 0; AdrOffset_8090 = 4294967295; BitOffset_8090 = 0; BitLength_8090 = 0; Address_8090 = ''; Type_8090 = ''; AddressPointer_8090 = 0; AdrOffset_8510 = 52; BitOffset_8510 = 0; BitLength_8510 = 16; Address_8510 = '%IW26'; Type_8510 = 'UINT'; AddressPointer_8510 = ADR(%IW26); AdrOffset_8520 = 56; BitOffset_8520 = 0; BitLength_8520 = 32; Address_8520 = '%ID14'; Type_8520 = 'DINT'; AddressPointer_8520 = ADR(%ID14); AdrOffset_8530 = 4294967295; BitOffset_8530 = 0; BitLength_8530 = 0; Address_8530 = ''; Type_8530 = ''; AddressPointer_8530 = 0; AdrOffset_8540 = 4294967295; BitOffset_8540 = 0; BitLength_8540 = 0; Address_8540 = ''; Type_8540 = ''; AddressPointer_8540 = 0; AdrOffset_8550 = 54;
              BitOffset_8550 = 0; BitLength_8550 = 8; Address_8550 = '%IB54'; Type_8550 = 'SINT'; AddressPointer_8550 = ADR(%IB54); AdrOffset_8560 = 4294967295; BitOffset_8560 = 0; BitLength_8560 = 0; Address_8560 = ''; Type_8560 = ''; AddressPointer_8560 = 0; AdrOffset_8570 = 4294967295; BitOffset_8570 = 0; BitLength_8570 = 0; Address_8570 = ''; Type_8570 = ''; AddressPointer_8570 = 0; AdrOffset_8580 = 4294967295; BitOffset_8580 = 0; BitLength_8580 = 0; Address_8580 = ''; Type_8580 = ''; AddressPointer_8580 = 0; AdrOffset_8590 = 4294967295; BitOffset_8590 = 0; BitLength_8590 = 0; Address_8590 = ''; Type_8590 = ''; AddressPointer_8590 = 0; AdrOffset_8600 = 4294967295; BitOffset_8600 = 0; BitLength_8600 = 0; Address_8600 = ''; Type_8600 = ''; AddressPointer_8600 = 0; AdrOffset_8600 = 4294967295; BitOffset_8600 = 0; BitLength_8600 = 0; Address_8610 = ''; Type_8610 = '';
              AddressPointer_8610 = 0; AdrOffset_8620 = 4294967295; BitOffset_8620 = 0; BitLength_8620 = 0; Address_8620 = ''; Type_8620 = ''; AddressPointer_8620 = 0
        AXIS_5 : SM_Drive_EtherCAT_JMC, 3S - Smart Software Solutions GmbH, order no. 0, version 4.6.1.0
            settings: wDriveID = 20; AdrOffset_8010 = 400; BitOffset_8010 = 0; BitLength_8010 = 16; Address_8010 = '%QW200'; Type_8010 = 'UINT'; AddressPointer_8010 = ADR(%QW200); AdrOffset_8020 = 404; BitOffset_8020 = 0; BitLength_8020 = 32; Address_8020 = '%QD101'; Type_8020 = 'DINT'; AddressPointer_8020 = ADR(%QD101); AdrOffset_8030 = 4294967295; BitOffset_8030 = 0; BitLength_8030 = 0; Address_8030 = ''; Type_8030 = ''; AddressPointer_8030 = 0; AdrOffset_8040 = 4294967295; BitOffset_8040 = 0; BitLength_8040 = 0; Address_8040 = ''; Type_8040 = ''; AddressPointer_8040 = 0; AdrOffset_8050 = 402; BitOffset_8050 = 0; BitLength_8050 = 8; Address_8050 = '%QB402'; Type_8050 = 'SINT'; AddressPointer_8050 = ADR(%QB402); AdrOffset_8060 = 4294967295; BitOffset_8060 = 0; BitLength_8060 = 0; Address_8060 = ''; Type_8060 = ''; AddressPointer_8060 = 0; AdrOffset_8070 = 4294967295; BitOffset_8070 = 0; BitLength_8070 = 0;
              Address_8070 = ''; Type_8070 = ''; AddressPointer_8070 = 0; AdrOffset_8080 = 4294967295; BitOffset_8080 = 0; BitLength_8080 = 0; Address_8080 = ''; Type_8080 = ''; AddressPointer_8080 = 0; AdrOffset_8090 = 4294967295; BitOffset_8090 = 0; BitLength_8090 = 0; Address_8090 = ''; Type_8090 = ''; AddressPointer_8090 = 0; AdrOffset_8510 = 68; BitOffset_8510 = 0; BitLength_8510 = 16; Address_8510 = '%IW34'; Type_8510 = 'UINT'; AddressPointer_8510 = ADR(%IW34); AdrOffset_8520 = 72; BitOffset_8520 = 0; BitLength_8520 = 32; Address_8520 = '%ID18'; Type_8520 = 'DINT'; AddressPointer_8520 = ADR(%ID18); AdrOffset_8530 = 4294967295; BitOffset_8530 = 0; BitLength_8530 = 0; Address_8530 = ''; Type_8530 = ''; AddressPointer_8530 = 0; AdrOffset_8540 = 4294967295; BitOffset_8540 = 0; BitLength_8540 = 0; Address_8540 = ''; Type_8540 = ''; AddressPointer_8540 = 0; AdrOffset_8550 = 70;
              BitOffset_8550 = 0; BitLength_8550 = 8; Address_8550 = '%IB70'; Type_8550 = 'SINT'; AddressPointer_8550 = ADR(%IB70); AdrOffset_8560 = 4294967295; BitOffset_8560 = 0; BitLength_8560 = 0; Address_8560 = ''; Type_8560 = ''; AddressPointer_8560 = 0; AdrOffset_8570 = 4294967295; BitOffset_8570 = 0; BitLength_8570 = 0; Address_8570 = ''; Type_8570 = ''; AddressPointer_8570 = 0; AdrOffset_8580 = 4294967295; BitOffset_8580 = 0; BitLength_8580 = 0; Address_8580 = ''; Type_8580 = ''; AddressPointer_8580 = 0; AdrOffset_8590 = 4294967295; BitOffset_8590 = 0; BitLength_8590 = 0; Address_8590 = ''; Type_8590 = ''; AddressPointer_8590 = 0; AdrOffset_8600 = 4294967295; BitOffset_8600 = 0; BitLength_8600 = 0; Address_8600 = ''; Type_8600 = ''; AddressPointer_8600 = 0; AdrOffset_8600 = 4294967295; BitOffset_8600 = 0; BitLength_8600 = 0; Address_8610 = ''; Type_8610 = '';
              AddressPointer_8610 = 0; AdrOffset_8620 = 4294967295; BitOffset_8620 = 0; BitLength_8620 = 0; Address_8620 = ''; Type_8620 = ''; AddressPointer_8620 = 0
        AXIS_6 : SM_Drive_EtherCAT_JMC, 3S - Smart Software Solutions GmbH, order no. 0, version 4.6.1.0
            settings: wDriveID = 21; dwRatioTechUnitsDenom = 800; eRampType = 3; ScalingIncs = 800; AdrOffset_8010 = 424; BitOffset_8010 = 0; BitLength_8010 = 16; Address_8010 = '%QW212'; Type_8010 = 'UINT'; AddressPointer_8010 = ADR(%QW212); AdrOffset_8020 = 428; BitOffset_8020 = 0; BitLength_8020 = 32; Address_8020 = '%QD107'; Type_8020 = 'DINT'; AddressPointer_8020 = ADR(%QD107); AdrOffset_8030 = 4294967295; BitOffset_8030 = 0; BitLength_8030 = 0; Address_8030 = ''; Type_8030 = ''; AddressPointer_8030 = 0; AdrOffset_8040 = 4294967295; BitOffset_8040 = 0; BitLength_8040 = 0; Address_8040 = ''; Type_8040 = ''; AddressPointer_8040 = 0; AdrOffset_8050 = 426; BitOffset_8050 = 0; BitLength_8050 = 8; Address_8050 = '%QB426'; Type_8050 = 'SINT'; AddressPointer_8050 = ADR(%QB426); AdrOffset_8060 = 4294967295; BitOffset_8060 = 0; BitLength_8060 = 0; Address_8060 = ''; Type_8060 = ''; AddressPointer_8060 = 0;
              AdrOffset_8070 = 4294967295; BitOffset_8070 = 0; BitLength_8070 = 0; Address_8070 = ''; Type_8070 = ''; AddressPointer_8070 = 0; AdrOffset_8080 = 4294967295; BitOffset_8080 = 0; BitLength_8080 = 0; Address_8080 = ''; Type_8080 = ''; AddressPointer_8080 = 0; AdrOffset_8090 = 4294967295; BitOffset_8090 = 0; BitLength_8090 = 0; Address_8090 = ''; Type_8090 = ''; AddressPointer_8090 = 0; AdrOffset_8510 = 84; BitOffset_8510 = 0; BitLength_8510 = 16; Address_8510 = '%IW42'; Type_8510 = 'UINT'; AddressPointer_8510 = ADR(%IW42); AdrOffset_8520 = 88; BitOffset_8520 = 0; BitLength_8520 = 32; Address_8520 = '%ID22'; Type_8520 = 'DINT'; AddressPointer_8520 = ADR(%ID22); AdrOffset_8530 = 4294967295; BitOffset_8530 = 0; BitLength_8530 = 0; Address_8530 = ''; Type_8530 = ''; AddressPointer_8530 = 0; AdrOffset_8540 = 4294967295; BitOffset_8540 = 0; BitLength_8540 = 0; Address_8540 = '';
              Type_8540 = ''; AddressPointer_8540 = 0; AdrOffset_8550 = 86; BitOffset_8550 = 0; BitLength_8550 = 8; Address_8550 = '%IB86'; Type_8550 = 'SINT'; AddressPointer_8550 = ADR(%IB86); AdrOffset_8560 = 4294967295; BitOffset_8560 = 0; BitLength_8560 = 0; Address_8560 = ''; Type_8560 = ''; AddressPointer_8560 = 0; AdrOffset_8570 = 4294967295; BitOffset_8570 = 0; BitLength_8570 = 0; Address_8570 = ''; Type_8570 = ''; AddressPointer_8570 = 0; AdrOffset_8580 = 4294967295; BitOffset_8580 = 0; BitLength_8580 = 0; Address_8580 = ''; Type_8580 = ''; AddressPointer_8580 = 0; AdrOffset_8590 = 4294967295; BitOffset_8590 = 0; BitLength_8590 = 0; Address_8590 = ''; Type_8590 = ''; AddressPointer_8590 = 0; AdrOffset_8600 = 4294967295; BitOffset_8600 = 0; BitLength_8600 = 0; Address_8600 = ''; Type_8600 = ''; AddressPointer_8600 = 0; AdrOffset_8600 = 4294967295; BitOffset_8600 = 0;
              BitLength_8600 = 0; Address_8610 = ''; Type_8610 = ''; AddressPointer_8610 = 0; AdrOffset_8620 = 4294967295; BitOffset_8620 = 0; BitLength_8620 = 0; Address_8620 = ''; Type_8620 = ''; AddressPointer_8620 = 0
        local : local, Shenzhen Just Motion Control Electromechanics Co,.ltd, order no. local, version 0
            settings: Number of Outputs = 17; Number of Inputs = 25; Number of Infos about Outputs = 17; Number of Infos about Inputs = 25; RxTxPdo.Virtual = False; RxTxPdo.DependOnSlot = True; RxTxPdo.DependOnSlotGroup = False; RxTxPdo.OverwrittenByModule = True; AO0.Offset = 0; AO0.DependOnSlot = True; AO0.DependOnSlotGroup = False; Y0.Offset = 0; Y0.DependOnSlot = True; Y0.DependOnSlotGroup = False; Y1.Offset = 0; Y1.DependOnSlot = True; Y1.DependOnSlotGroup = False; Y2.Offset = 0; Y2.DependOnSlot = True; Y2.DependOnSlotGroup = False; Y3.Offset = 0; Y3.DependOnSlot = True; Y3.DependOnSlotGroup = False; Y4.Offset = 0; Y4.DependOnSlot = True; Y4.DependOnSlotGroup = False; Y5.Offset = 0; Y5.DependOnSlot = True; Y5.DependOnSlotGroup = False; Y6.Offset = 0; Y6.DependOnSlot = True; Y6.DependOnSlotGroup = False; Y7.Offset = 0; Y7.DependOnSlot = True; Y7.DependOnSlotGroup = False; Y8.Offset = 0; Y8.DependOnSlot = True; Y8.DependOnSlotGroup = False; Y9.Offset = 0; Y9.DependOnSlot = True;
              Y9.DependOnSlotGroup = False; Y10.Offset = 0; Y10.DependOnSlot = True; Y10.DependOnSlotGroup = False; Y11.Offset = 0; Y11.DependOnSlot = True; Y11.DependOnSlotGroup = False; Y12.Offset = 0; Y12.DependOnSlot = True; Y12.DependOnSlotGroup = False; Y13.Offset = 0; Y13.DependOnSlot = True; Y13.DependOnSlotGroup = False; Y14.Offset = 0; Y14.DependOnSlot = True; Y14.DependOnSlotGroup = False; Y15.Offset = 0; Y15.DependOnSlot = True; Y15.DependOnSlotGroup = False; RxTxPdo.Virtual = False; RxTxPdo.DependOnSlot = True; RxTxPdo.DependOnSlotGroup = False; RxTxPdo.OverwrittenByModule = True; AI0.Offset = 0; AI0.DependOnSlot = True; AI0.DependOnSlotGroup = False; X0.Offset = 0; X0.DependOnSlot = True; X0.DependOnSlotGroup = False; X1.Offset = 0; X1.DependOnSlot = True; X1.DependOnSlotGroup = False; X2.Offset = 0; X2.DependOnSlot = True; X2.DependOnSlotGroup = False; X3.Offset = 0; X3.DependOnSlot = True; X3.DependOnSlotGroup = False; X4.Offset = 0; X4.DependOnSlot = True;
              X4.DependOnSlotGroup = False; X5.Offset = 0; X5.DependOnSlot = True; X5.DependOnSlotGroup = False; X6.Offset = 0; X6.DependOnSlot = True; X6.DependOnSlotGroup = False; X7.Offset = 0; X7.DependOnSlot = True; X7.DependOnSlotGroup = False; X8.Offset = 0; X8.DependOnSlot = True; X8.DependOnSlotGroup = False; X9.Offset = 0; X9.DependOnSlot = True; X9.DependOnSlotGroup = False; X10.Offset = 0; X10.DependOnSlot = True; X10.DependOnSlotGroup = False; X11.Offset = 0; X11.DependOnSlot = True; X11.DependOnSlotGroup = False; X12.Offset = 0; X12.DependOnSlot = True; X12.DependOnSlotGroup = False; X13.Offset = 0; X13.DependOnSlot = True; X13.DependOnSlotGroup = False; X14.Offset = 0; X14.DependOnSlot = True; X14.DependOnSlotGroup = False; X15.Offset = 0; X15.DependOnSlot = True; X15.DependOnSlotGroup = False; X16.Offset = 0; X16.DependOnSlot = True; X16.DependOnSlotGroup = False; X17.Offset = 0; X17.DependOnSlot = True; X17.DependOnSlotGroup = False;
              X18.Offset = 0; X18.DependOnSlot = True; X18.DependOnSlotGroup = False; X19.Offset = 0; X19.DependOnSlot = True; X19.DependOnSlotGroup = False; X20.Offset = 0; X20.DependOnSlot = True; X20.DependOnSlotGroup = False; X21.Offset = 0; X21.DependOnSlot = True; X21.DependOnSlotGroup = False; X22.Offset = 0; X22.DependOnSlot = True; X22.DependOnSlotGroup = False; X23.Offset = 0; X23.DependOnSlot = True; X23.DependOnSlotGroup = False; AO0.Default = ''; Y0.Default = ''; Y1.Default = ''; Y2.Default = ''; Y3.Default = ''; Y4.Default = ''; Y5.Default = ''; Y6.Default = ''; Y7.Default = ''; Y8.Default = ''; Y9.Default = ''; Y10.Default = ''; Y11.Default = ''; Y12.Default = ''; Y13.Default = ''; Y14.Default = ''; Y15.Default = ''; AI0.Default = ''; X0.Default = ''; X1.Default = ''; X2.Default = ''; X3.Default = '';
              X4.Default = ''; X5.Default = ''; X6.Default = ''; X7.Default = ''; X8.Default = ''; X9.Default = ''; X10.Default = ''; X11.Default = ''; X12.Default = ''; X13.Default = ''; X14.Default = ''; X15.Default = ''; X16.Default = ''; X17.Default = ''; X18.Default = ''; X19.Default = ''; X20.Default = ''; X21.Default = ''; X22.Default = ''; X23.Default = ''
            output Application.GVL.Y[0] : BIT  // Y0
            output Application.GVL.Y[1] : BIT  // Y1
            output Application.GVL.Y[2] : BIT  // Y2
            output Application.GVL.Y[3] : BIT  // Y3
            output Application.GVL.Y[4] : BIT  // Y4
            output Application.GVL.Y[5] : BIT  // Y5
            output Application.GVL.Y[6] : BIT  // Y6
            output Application.GVL.Y[7] : BIT  // Y7
            output Application.GVL.Y[8] : BIT  // Y8
            output Application.GVL.Y[9] : BIT  // Y9
            output Application.GVL.Y[10] : BIT  // Y10
            output Application.GVL.Y[11] : BIT  // Y11
            output Application.GVL.Y[12] : BIT  // Y12
            output Application.GVL.Y[13] : BIT  // Y13
            output Application.GVL.Y[14] : BIT  // Y14
            output Application.GVL.Y[15] : BIT  // Y15
            input  Application.GVL.X[0] : BIT  // X0
            input  Application.GVL.X[1] : BIT  // X1
            input  Application.GVL.X[2] : BIT  // X2
            input  Application.GVL.X[3] : BIT  // X3
            input  Application.GVL.X[4] : BIT  // X4
            input  Application.GVL.X[5] : BIT  // X5
            input  Application.GVL.X[6] : BIT  // X6
            input  Application.GVL.X[7] : BIT  // X7
            input  Application.GVL.X[8] : BIT  // X8
            input  Application.GVL.X[9] : BIT  // X9
            input  Application.GVL.X[10] : BIT  // X10
            input  Application.GVL.X[11] : BIT  // X11
            input  Application.GVL.X[12] : BIT  // X12
            input  Application.GVL.X[13] : BIT  // X13
            input  Application.GVL.X[14] : BIT  // X14
            input  Application.GVL.X[15] : BIT  // X15
            input  Application.GVL.X[16] : BIT  // X16
            input  Application.GVL.X[17] : BIT  // X17
            input  Application.GVL.X[18] : BIT  // X18
            input  Application.GVL.X[19] : BIT  // X19
            input  Application.GVL.X[20] : BIT  // X20
            input  Application.GVL.X[21] : BIT  // X21
            input  Application.GVL.X[22] : BIT  // X22
            input  Application.GVL.X[23] : BIT  // X23
            unmapped channels: AO0, AI0
      XINJE_DS5C1_CoE_Drive_Rev4_0_A0 : XINJE-DS5C1 EtherCAT(CoE) Drive Rev4.0 v3.7.70, Xinje Electronics, Inc., order no. XINJE-DS5C1 CoE Drive Rev4.0, version Revision=16#20201207
          settings: EnableExpertSettings = True; StationAlias = 1002; Optional = False; DeviceIdenticationADO = 18; DeviceIdenticationMode = 1; DC sync0 cycletime = 8000; DC enable = 1; DC sync0 enable = 1; DC sync0 shift time = 0; DC sync1 cycletime = 8000; DC sync1 enable = 0; DC sync1 factor = 'x 1'; DC sync1 shift time = 0; Number of SDO = 4; Interpolation time period.Value = 8; Homing method.Index = 16#6098; Homing method.Subindex = 16#00; Homing method.Value = 35; Homing method.Size = 8; Homing method.AbortIfError = FALSE; Homing method.JumpToLine = FALSE; Homing method.Line = 0; Homing method.CompleteAccess = False; Interpolation time index.Index = 16#60C2; Interpolation time index.Subindex = 16#02; Interpolation time index.Value = 253; Interpolation time index.Size = 8; Interpolation time index.AbortIfError = FALSE; Interpolation time index.JumpToLine = FALSE; Interpolation time index.Line = 0; Interpolation time index.CompleteAccess = False
          unmapped channels: Control Word, TargetPosition, TargetVelocity, TargetTorque, ModeOfOperation, Status Word, ActualPosition, Velocity actual value, ActualTorque, ModeOfOperationDisplay
        A0 : SM_Drive_GenericDSP402, 3S - Smart Software Solutions GmbH, order no. 0, version 4.6.1.0
            settings: wDriveID = 3; dwRatioTechUnitsDenom = 327680; iRatioTechUnitsNum = -9; eRampType = 2; fSWMaxVelocity = 225; fSWMaxAcceleration = 500; fSWMaxDeceleration = 500; fSWMaxJerk = 500; ScalingIncs = 131072; ScalingMotorTurns2 = 100; ScalingUnits = 360; InvertDirection = TRUE; IsLinearMotor = FALSE; AdrOffset_8010 = 456; BitOffset_8010 = 0; BitLength_8010 = 16; Address_8010 = '%QW228'; Type_8010 = 'UINT'; AddressPointer_8010 = ADR(%QW228); AdrOffset_8020 = 460; BitOffset_8020 = 0; BitLength_8020 = 32; Address_8020 = '%QD115'; Type_8020 = 'DINT'; AddressPointer_8020 = ADR(%QD115); AdrOffset_8030 = 464; BitOffset_8030 = 0; BitLength_8030 = 32; Address_8030 = '%QD116'; Type_8030 = 'DINT'; AddressPointer_8030 = ADR(%QD116); AdrOffset_8040 = 468; BitOffset_8040 = 0; BitLength_8040 = 16; Address_8040 = '%QW234'; Type_8040 = 'INT'; AddressPointer_8040 = ADR(%QW234); AdrOffset_8050 = 470; BitOffset_8050 = 0; BitLength_8050 = 8;
              Address_8050 = '%QB470'; Type_8050 = 'SINT'; AddressPointer_8050 = ADR(%QB470); AdrOffset_8060 = 4294967295; BitOffset_8060 = 0; BitLength_8060 = 0; Address_8060 = ''; Type_8060 = ''; AddressPointer_8060 = 0; AdrOffset_8070 = 4294967295; BitOffset_8070 = 0; BitLength_8070 = 0; Address_8070 = ''; Type_8070 = ''; AddressPointer_8070 = 0; AdrOffset_8080 = 4294967295; BitOffset_8080 = 0; BitLength_8080 = 0; Address_8080 = ''; Type_8080 = ''; AddressPointer_8080 = 0; AdrOffset_8090 = 4294967295; BitOffset_8090 = 0; BitLength_8090 = 0; Address_8090 = ''; Type_8090 = ''; AddressPointer_8090 = 0; AdrOffset_8510 = 108; BitOffset_8510 = 0; BitLength_8510 = 16; Address_8510 = '%IW54'; Type_8510 = 'UINT'; AddressPointer_8510 = ADR(%IW54); AdrOffset_8520 = 112; BitOffset_8520 = 0; BitLength_8520 = 32; Address_8520 = '%ID28'; Type_8520 = 'DINT'; AddressPointer_8520 = ADR(%ID28); AdrOffset_8530 = 116;
              BitOffset_8530 = 0; BitLength_8530 = 32; Address_8530 = '%ID29'; Type_8530 = 'DINT'; AddressPointer_8530 = ADR(%ID29); AdrOffset_8540 = 120; BitOffset_8540 = 0; BitLength_8540 = 16; Address_8540 = '%IW60'; Type_8540 = 'INT'; AddressPointer_8540 = ADR(%IW60); AdrOffset_8550 = 122; BitOffset_8550 = 0; BitLength_8550 = 8; Address_8550 = '%IB122'; Type_8550 = 'SINT'; AddressPointer_8550 = ADR(%IB122); AdrOffset_8560 = 4294967295; BitOffset_8560 = 0; BitLength_8560 = 0; Address_8560 = ''; Type_8560 = ''; AddressPointer_8560 = 0; AdrOffset_8570 = 4294967295; BitOffset_8570 = 0; BitLength_8570 = 0; Address_8570 = ''; Type_8570 = ''; AddressPointer_8570 = 0; AdrOffset_8580 = 4294967295; BitOffset_8580 = 0; BitLength_8580 = 0; Address_8580 = ''; Type_8580 = ''; AddressPointer_8580 = 0; AdrOffset_8590 = 4294967295; BitOffset_8590 = 0; BitLength_8590 = 0; Address_8590 = ''; Type_8590 = '';
              AddressPointer_8590 = 0; AdrOffset_8600 = 4294967295; BitOffset_8600 = 0; BitLength_8600 = 0; Address_8600 = ''; Type_8600 = ''; AddressPointer_8600 = 0; AdrOffset_8600 = 4294967295; BitOffset_8600 = 0; BitLength_8600 = 0; Address_8610 = ''; Type_8610 = ''; AddressPointer_8610 = 0; AdrOffset_8620 = 4294967295; BitOffset_8620 = 0; BitLength_8620 = 0; Address_8620 = ''; Type_8620 = ''; AddressPointer_8620 = 0
      XINJE_DS5C1_CoE_Drive_Rev4_0_A1 : XINJE-DS5C1 EtherCAT(CoE) Drive Rev4.0 v3.7.70, Xinje Electronics, Inc., order no. XINJE-DS5C1 CoE Drive Rev4.0, version Revision=16#20201207
          settings: EnableExpertSettings = True; StationAlias = 1003; DeviceIdenticationADO = 18; DeviceIdenticationMode = 1; DC sync0 cycletime = 8000; DC sync1 cycletime = 8000; Number of SDO = 4; Homing method.Index = 16#6098; Homing method.Subindex = 16#00; Homing method.Value = 35; Homing method.Size = 8; Homing method.AbortIfError = FALSE; Homing method.JumpToLine = FALSE; Homing method.Line = 0; Homing method.CompleteAccess = False; Op mode.Index = 16#6060; Op mode.Subindex = 16#00; Op mode.Value = 8; Op mode.Size = 8; Op mode.AbortIfError = FALSE; Op mode.JumpToLine = FALSE; Op mode.Line = 0; Op mode.CompleteAccess = False; Interpolation time period.Index = 16#60C2; Interpolation time period.Subindex = 16#01; Interpolation time period.Value = 8; Interpolation time period.Size = 8; Interpolation time period.AbortIfError = FALSE; Interpolation time period.JumpToLine = FALSE; Interpolation time period.Line = 0; Interpolation time period.CompleteAccess = False; Interpolation time index.Index = 16#60C2; Interpolation time index.Subindex = 16#02; Interpolation time index.Value = 253; Interpolation time index.Size = 8; Interpolation time index.AbortIfError = FALSE; Interpolation time index.JumpToLine = FALSE; Interpolation time index.Line = 0; Interpolation time index.CompleteAccess = False
          unmapped channels: Control Word, TargetPosition, TargetVelocity, TargetTorque, ModeOfOperation, Status Word, ActualPosition, Velocity actual value, ActualTorque, ModeOfOperationDisplay
        A1 : SM_Drive_GenericDSP402, 3S - Smart Software Solutions GmbH, order no. 0, version 4.6.1.0
            settings: wDriveID = 4; dwRatioTechUnitsDenom = 327680; iRatioTechUnitsNum = -9; eRampType = 2; fSWMaxVelocity = 140; fSWMaxAcceleration = 400; fSWMaxDeceleration = 400; fSWMaxJerk = 400; ScalingIncs = 131072; ScalingMotorTurns2 = 100; ScalingUnits = 360; InvertDirection = TRUE; AdrOffset_8010 = 472; BitOffset_8010 = 0; BitLength_8010 = 16; Address_8010 = '%QW236'; Type_8010 = 'UINT'; AddressPointer_8010 = ADR(%QW236); AdrOffset_8020 = 476; BitOffset_8020 = 0; BitLength_8020 = 32; Address_8020 = '%QD119'; Type_8020 = 'DINT'; AddressPointer_8020 = ADR(%QD119); AdrOffset_8030 = 480; BitOffset_8030 = 0; BitLength_8030 = 32; Address_8030 = '%QD120'; Type_8030 = 'DINT'; AddressPointer_8030 = ADR(%QD120); AdrOffset_8040 = 484; BitOffset_8040 = 0; BitLength_8040 = 16; Address_8040 = '%QW242'; Type_8040 = 'INT'; AddressPointer_8040 = ADR(%QW242); AdrOffset_8050 = 486; BitOffset_8050 = 0; BitLength_8050 = 8; Address_8050 = '%QB486';
              Type_8050 = 'SINT'; AddressPointer_8050 = ADR(%QB486); AdrOffset_8060 = 4294967295; BitOffset_8060 = 0; BitLength_8060 = 0; Address_8060 = ''; Type_8060 = ''; AddressPointer_8060 = 0; AdrOffset_8070 = 4294967295; BitOffset_8070 = 0; BitLength_8070 = 0; Address_8070 = ''; Type_8070 = ''; AddressPointer_8070 = 0; AdrOffset_8080 = 4294967295; BitOffset_8080 = 0; BitLength_8080 = 0; Address_8080 = ''; Type_8080 = ''; AddressPointer_8080 = 0; AdrOffset_8090 = 4294967295; BitOffset_8090 = 0; BitLength_8090 = 0; Address_8090 = ''; Type_8090 = ''; AddressPointer_8090 = 0; AdrOffset_8510 = 124; BitOffset_8510 = 0; BitLength_8510 = 16; Address_8510 = '%IW62'; Type_8510 = 'UINT'; AddressPointer_8510 = ADR(%IW62); AdrOffset_8520 = 128; BitOffset_8520 = 0; BitLength_8520 = 32; Address_8520 = '%ID32'; Type_8520 = 'DINT'; AddressPointer_8520 = ADR(%ID32); AdrOffset_8530 = 132; BitOffset_8530 = 0;
              BitLength_8530 = 32; Address_8530 = '%ID33'; Type_8530 = 'DINT'; AddressPointer_8530 = ADR(%ID33); AdrOffset_8540 = 136; BitOffset_8540 = 0; BitLength_8540 = 16; Address_8540 = '%IW68'; Type_8540 = 'INT'; AddressPointer_8540 = ADR(%IW68); AdrOffset_8550 = 138; BitOffset_8550 = 0; BitLength_8550 = 8; Address_8550 = '%IB138'; Type_8550 = 'SINT'; AddressPointer_8550 = ADR(%IB138); AdrOffset_8560 = 4294967295; BitOffset_8560 = 0; BitLength_8560 = 0; Address_8560 = ''; Type_8560 = ''; AddressPointer_8560 = 0; AdrOffset_8570 = 4294967295; BitOffset_8570 = 0; BitLength_8570 = 0; Address_8570 = ''; Type_8570 = ''; AddressPointer_8570 = 0; AdrOffset_8580 = 4294967295; BitOffset_8580 = 0; BitLength_8580 = 0; Address_8580 = ''; Type_8580 = ''; AddressPointer_8580 = 0; AdrOffset_8590 = 4294967295; BitOffset_8590 = 0; BitLength_8590 = 0; Address_8590 = ''; Type_8590 = ''; AddressPointer_8590 = 0;
              AdrOffset_8600 = 4294967295; BitOffset_8600 = 0; BitLength_8600 = 0; Address_8600 = ''; Type_8600 = ''; AddressPointer_8600 = 0; AdrOffset_8600 = 4294967295; BitOffset_8600 = 0; BitLength_8600 = 0; Address_8610 = ''; Type_8610 = ''; AddressPointer_8610 = 0; AdrOffset_8620 = 4294967295; BitOffset_8620 = 0; BitLength_8620 = 0; Address_8620 = ''; Type_8620 = ''; AddressPointer_8620 = 0
      XINJE_DS5C1_CoE_Drive_Rev4_0_A2 : XINJE-DS5C1 EtherCAT(CoE) Drive Rev4.0 v3.7.70, Xinje Electronics, Inc., order no. XINJE-DS5C1 CoE Drive Rev4.0, version Revision=16#20201207
          settings: EnableExpertSettings = True; StationAlias = 1004; DeviceIdenticationADO = 18; DeviceIdenticationMode = 1; DC sync0 cycletime = 8000; DC sync1 cycletime = 8000; Number of SDO = 4; Homing method.Index = 16#6098; Homing method.Subindex = 16#00; Homing method.Value = 35; Homing method.Size = 8; Homing method.AbortIfError = FALSE; Homing method.JumpToLine = FALSE; Homing method.Line = 0; Homing method.CompleteAccess = False; Op mode.Index = 16#6060; Op mode.Subindex = 16#00; Op mode.Value = 8; Op mode.Size = 8; Op mode.AbortIfError = FALSE; Op mode.JumpToLine = FALSE; Op mode.Line = 0; Op mode.CompleteAccess = False; Interpolation time period.Index = 16#60C2; Interpolation time period.Subindex = 16#01; Interpolation time period.Value = 8; Interpolation time period.Size = 8; Interpolation time period.AbortIfError = FALSE; Interpolation time period.JumpToLine = FALSE; Interpolation time period.Line = 0; Interpolation time period.CompleteAccess = False; Interpolation time index.Index = 16#60C2; Interpolation time index.Subindex = 16#02; Interpolation time index.Value = 253; Interpolation time index.Size = 8; Interpolation time index.AbortIfError = FALSE; Interpolation time index.JumpToLine = FALSE; Interpolation time index.Line = 0; Interpolation time index.CompleteAccess = False
          unmapped channels: Control Word, TargetPosition, TargetVelocity, TargetTorque, ModeOfOperation, Status Word, ActualPosition, Velocity actual value, ActualTorque, ModeOfOperationDisplay
        A2 : SM_Drive_GenericDSP402, 3S - Smart Software Solutions GmbH, order no. 0, version 4.6.1.0
            settings: wDriveID = 5; dwRatioTechUnitsDenom = 32768; iRatioTechUnitsNum = 5; eRampType = 2; fSWMaxVelocity = 500; fSWMaxAcceleration = 2000; fSWMaxDeceleration = 2000; ScalingIncs = 131072; ScalingUnits = 20; AdrOffset_8010 = 488; BitOffset_8010 = 0; BitLength_8010 = 16; Address_8010 = '%QW244'; Type_8010 = 'UINT'; AddressPointer_8010 = ADR(%QW244); AdrOffset_8020 = 492; BitOffset_8020 = 0; BitLength_8020 = 32; Address_8020 = '%QD123'; Type_8020 = 'DINT'; AddressPointer_8020 = ADR(%QD123); AdrOffset_8030 = 496; BitOffset_8030 = 0; BitLength_8030 = 32; Address_8030 = '%QD124'; Type_8030 = 'DINT'; AddressPointer_8030 = ADR(%QD124); AdrOffset_8040 = 500; BitOffset_8040 = 0; BitLength_8040 = 16; Address_8040 = '%QW250'; Type_8040 = 'INT'; AddressPointer_8040 = ADR(%QW250); AdrOffset_8050 = 502; BitOffset_8050 = 0; BitLength_8050 = 8; Address_8050 = '%QB502'; Type_8050 = 'SINT'; AddressPointer_8050 = ADR(%QB502); AdrOffset_8060 = 4294967295;
              BitOffset_8060 = 0; BitLength_8060 = 0; Address_8060 = ''; Type_8060 = ''; AddressPointer_8060 = 0; AdrOffset_8070 = 4294967295; BitOffset_8070 = 0; BitLength_8070 = 0; Address_8070 = ''; Type_8070 = ''; AddressPointer_8070 = 0; AdrOffset_8080 = 4294967295; BitOffset_8080 = 0; BitLength_8080 = 0; Address_8080 = ''; Type_8080 = ''; AddressPointer_8080 = 0; AdrOffset_8090 = 4294967295; BitOffset_8090 = 0; BitLength_8090 = 0; Address_8090 = ''; Type_8090 = ''; AddressPointer_8090 = 0; AdrOffset_8510 = 140; BitOffset_8510 = 0; BitLength_8510 = 16; Address_8510 = '%IW70'; Type_8510 = 'UINT'; AddressPointer_8510 = ADR(%IW70); AdrOffset_8520 = 144; BitOffset_8520 = 0; BitLength_8520 = 32; Address_8520 = '%ID36'; Type_8520 = 'DINT'; AddressPointer_8520 = ADR(%ID36); AdrOffset_8530 = 148; BitOffset_8530 = 0; BitLength_8530 = 32; Address_8530 = '%ID37'; Type_8530 = 'DINT';
              AddressPointer_8530 = ADR(%ID37); AdrOffset_8540 = 152; BitOffset_8540 = 0; BitLength_8540 = 16; Address_8540 = '%IW76'; Type_8540 = 'INT'; AddressPointer_8540 = ADR(%IW76); AdrOffset_8550 = 154; BitOffset_8550 = 0; BitLength_8550 = 8; Address_8550 = '%IB154'; Type_8550 = 'SINT'; AddressPointer_8550 = ADR(%IB154); AdrOffset_8560 = 4294967295; BitOffset_8560 = 0; BitLength_8560 = 0; Address_8560 = ''; Type_8560 = ''; AddressPointer_8560 = 0; AdrOffset_8570 = 4294967295; BitOffset_8570 = 0; BitLength_8570 = 0; Address_8570 = ''; Type_8570 = ''; AddressPointer_8570 = 0; AdrOffset_8580 = 4294967295; BitOffset_8580 = 0; BitLength_8580 = 0; Address_8580 = ''; Type_8580 = ''; AddressPointer_8580 = 0; AdrOffset_8590 = 4294967295; BitOffset_8590 = 0; BitLength_8590 = 0; Address_8590 = ''; Type_8590 = ''; AddressPointer_8590 = 0; AdrOffset_8600 = 4294967295; BitOffset_8600 = 0; BitLength_8600 = 0;
              Address_8600 = ''; Type_8600 = ''; AddressPointer_8600 = 0; AdrOffset_8600 = 4294967295; BitOffset_8600 = 0; BitLength_8600 = 0; Address_8610 = ''; Type_8610 = ''; AddressPointer_8610 = 0; AdrOffset_8620 = 4294967295; BitOffset_8620 = 0; BitLength_8620 = 0; Address_8620 = ''; Type_8620 = ''; AddressPointer_8620 = 0
      XINJE_DS5C1_CoE_Drive_Rev4_0_A3 : XINJE-DS5C1 EtherCAT(CoE) Drive Rev4.0 v3.7.70, Xinje Electronics, Inc., order no. XINJE-DS5C1 CoE Drive Rev4.0, version Revision=16#20201207
          settings: EnableExpertSettings = True; StationAlias = 1005; DeviceIdenticationADO = 18; DeviceIdenticationMode = 1; DC sync0 cycletime = 8000; DC sync1 cycletime = 8000; Number of SDO = 4; Homing method.Index = 16#6098; Homing method.Subindex = 16#00; Homing method.Value = 35; Homing method.Size = 8; Homing method.AbortIfError = FALSE; Homing method.JumpToLine = FALSE; Homing method.Line = 0; Homing method.CompleteAccess = False; Op mode.Index = 16#6060; Op mode.Subindex = 16#00; Op mode.Value = 8; Op mode.Size = 8; Op mode.AbortIfError = FALSE; Op mode.JumpToLine = FALSE; Op mode.Line = 0; Op mode.CompleteAccess = False; Interpolation time period.Index = 16#60C2; Interpolation time period.Subindex = 16#01; Interpolation time period.Value = 8; Interpolation time period.Size = 8; Interpolation time period.AbortIfError = FALSE; Interpolation time period.JumpToLine = FALSE; Interpolation time period.Line = 0; Interpolation time period.CompleteAccess = False; Interpolation time index.Index = 16#60C2; Interpolation time index.Subindex = 16#02; Interpolation time index.Value = 253; Interpolation time index.Size = 8; Interpolation time index.AbortIfError = FALSE; Interpolation time index.JumpToLine = FALSE; Interpolation time index.Line = 0; Interpolation time index.CompleteAccess = False
          unmapped channels: Control Word, TargetPosition, TargetVelocity, TargetTorque, ModeOfOperation, Status Word, ActualPosition, Velocity actual value, ActualTorque, ModeOfOperationDisplay
        A3 : SM_Drive_GenericDSP402, 3S - Smart Software Solutions GmbH, order no. 0, version 4.6.1.0
            settings: wDriveID = 6; dwRatioTechUnitsDenom = 65536; iRatioTechUnitsNum = 45; eRampType = 2; fSWMaxVelocity = 2000; fSWMaxAcceleration = 4000; fSWMaxDeceleration = 4000; fSWMaxJerk = 4000; ScalingIncs = 131072; ScalingMotorTurns2 = 4; ScalingUnits = 360; AdrOffset_8010 = 504; BitOffset_8010 = 0; BitLength_8010 = 16; Address_8010 = '%QW252'; Type_8010 = 'UINT'; AddressPointer_8010 = ADR(%QW252); AdrOffset_8020 = 508; BitOffset_8020 = 0; BitLength_8020 = 32; Address_8020 = '%QD127'; Type_8020 = 'DINT'; AddressPointer_8020 = ADR(%QD127); AdrOffset_8030 = 512; BitOffset_8030 = 0; BitLength_8030 = 32; Address_8030 = '%QD128'; Type_8030 = 'DINT'; AddressPointer_8030 = ADR(%QD128); AdrOffset_8040 = 516; BitOffset_8040 = 0; BitLength_8040 = 16; Address_8040 = '%QW258'; Type_8040 = 'INT'; AddressPointer_8040 = ADR(%QW258); AdrOffset_8050 = 518; BitOffset_8050 = 0; BitLength_8050 = 8; Address_8050 = '%QB518'; Type_8050 = 'SINT';
              AddressPointer_8050 = ADR(%QB518); AdrOffset_8060 = 4294967295; BitOffset_8060 = 0; BitLength_8060 = 0; Address_8060 = ''; Type_8060 = ''; AddressPointer_8060 = 0; AdrOffset_8070 = 4294967295; BitOffset_8070 = 0; BitLength_8070 = 0; Address_8070 = ''; Type_8070 = ''; AddressPointer_8070 = 0; AdrOffset_8080 = 4294967295; BitOffset_8080 = 0; BitLength_8080 = 0; Address_8080 = ''; Type_8080 = ''; AddressPointer_8080 = 0; AdrOffset_8090 = 4294967295; BitOffset_8090 = 0; BitLength_8090 = 0; Address_8090 = ''; Type_8090 = ''; AddressPointer_8090 = 0; AdrOffset_8510 = 156; BitOffset_8510 = 0; BitLength_8510 = 16; Address_8510 = '%IW78'; Type_8510 = 'UINT'; AddressPointer_8510 = ADR(%IW78); AdrOffset_8520 = 160; BitOffset_8520 = 0; BitLength_8520 = 32; Address_8520 = '%ID40'; Type_8520 = 'DINT'; AddressPointer_8520 = ADR(%ID40); AdrOffset_8530 = 164; BitOffset_8530 = 0; BitLength_8530 = 32;
              Address_8530 = '%ID41'; Type_8530 = 'DINT'; AddressPointer_8530 = ADR(%ID41); AdrOffset_8540 = 168; BitOffset_8540 = 0; BitLength_8540 = 16; Address_8540 = '%IW84'; Type_8540 = 'INT'; AddressPointer_8540 = ADR(%IW84); AdrOffset_8550 = 170; BitOffset_8550 = 0; BitLength_8550 = 8; Address_8550 = '%IB170'; Type_8550 = 'SINT'; AddressPointer_8550 = ADR(%IB170); AdrOffset_8560 = 4294967295; BitOffset_8560 = 0; BitLength_8560 = 0; Address_8560 = ''; Type_8560 = ''; AddressPointer_8560 = 0; AdrOffset_8570 = 4294967295; BitOffset_8570 = 0; BitLength_8570 = 0; Address_8570 = ''; Type_8570 = ''; AddressPointer_8570 = 0; AdrOffset_8580 = 4294967295; BitOffset_8580 = 0; BitLength_8580 = 0; Address_8580 = ''; Type_8580 = ''; AddressPointer_8580 = 0; AdrOffset_8590 = 4294967295; BitOffset_8590 = 0; BitLength_8590 = 0; Address_8590 = ''; Type_8590 = ''; AddressPointer_8590 = 0; AdrOffset_8600 = 4294967295;
              BitOffset_8600 = 0; BitLength_8600 = 0; Address_8600 = ''; Type_8600 = ''; AddressPointer_8600 = 0; AdrOffset_8600 = 4294967295; BitOffset_8600 = 0; BitLength_8600 = 0; Address_8610 = ''; Type_8610 = ''; AddressPointer_8610 = 0; AdrOffset_8620 = 4294967295; BitOffset_8620 = 0; BitLength_8620 = 0; Address_8620 = ''; Type_8620 = ''; AddressPointer_8620 = 0; Automatic Mapping = FALSE
      XINJE_DS5C1_CoE_Drive_Rev4_0_B0 : XINJE-DS5C1 EtherCAT(CoE) Drive Rev4.0 v3.7.70, Xinje Electronics, Inc., order no. XINJE-DS5C1 CoE Drive Rev4.0, version Revision=16#20201207
          settings: EnableExpertSettings = True; StationAlias = 1006; DeviceIdenticationADO = 18; DeviceIdenticationMode = 1; DC sync0 cycletime = 8000; DC sync1 cycletime = 8000; Number of SDO = 4; Homing method.Index = 16#6098; Homing method.Subindex = 16#00; Homing method.Value = 35; Homing method.Size = 8; Homing method.AbortIfError = FALSE; Homing method.JumpToLine = FALSE; Homing method.Line = 0; Homing method.CompleteAccess = False; Op mode.Index = 16#6060; Op mode.Subindex = 16#00; Op mode.Value = 8; Op mode.Size = 8; Op mode.AbortIfError = FALSE; Op mode.JumpToLine = FALSE; Op mode.Line = 0; Op mode.CompleteAccess = False; Interpolation time period.Index = 16#60C2; Interpolation time period.Subindex = 16#01; Interpolation time period.Value = 8; Interpolation time period.Size = 8; Interpolation time period.AbortIfError = FALSE; Interpolation time period.JumpToLine = FALSE; Interpolation time period.Line = 0; Interpolation time period.CompleteAccess = False; Interpolation time index.Index = 16#60C2; Interpolation time index.Subindex = 16#02; Interpolation time index.Value = 253; Interpolation time index.Size = 8; Interpolation time index.AbortIfError = FALSE; Interpolation time index.JumpToLine = FALSE; Interpolation time index.Line = 0; Interpolation time index.CompleteAccess = False
          unmapped channels: Control Word, TargetPosition, TargetVelocity, TargetTorque, ModeOfOperation, Status Word, ActualPosition, Velocity actual value, ActualTorque, ModeOfOperationDisplay
        B0 : SM_Drive_GenericDSP402, 3S - Smart Software Solutions GmbH, order no. 0, version 4.6.1.0
            settings: wDriveID = 7; dwRatioTechUnitsDenom = 327680; iRatioTechUnitsNum = -9; eRampType = 2; fSWMaxVelocity = 225; fSWMaxAcceleration = 500; fSWMaxDeceleration = 500; fSWMaxJerk = 500; ScalingIncs = 131072; ScalingMotorTurns2 = 100; ScalingUnits = 360; InvertDirection = TRUE; AdrOffset_8010 = 520; BitOffset_8010 = 0; BitLength_8010 = 16; Address_8010 = '%QW260'; Type_8010 = 'UINT'; AddressPointer_8010 = ADR(%QW260); AdrOffset_8020 = 524; BitOffset_8020 = 0; BitLength_8020 = 32; Address_8020 = '%QD131'; Type_8020 = 'DINT'; AddressPointer_8020 = ADR(%QD131); AdrOffset_8030 = 528; BitOffset_8030 = 0; BitLength_8030 = 32; Address_8030 = '%QD132'; Type_8030 = 'DINT'; AddressPointer_8030 = ADR(%QD132); AdrOffset_8040 = 532; BitOffset_8040 = 0; BitLength_8040 = 16; Address_8040 = '%QW266'; Type_8040 = 'INT'; AddressPointer_8040 = ADR(%QW266); AdrOffset_8050 = 534; BitOffset_8050 = 0; BitLength_8050 = 8; Address_8050 = '%QB534';
              Type_8050 = 'SINT'; AddressPointer_8050 = ADR(%QB534); AdrOffset_8060 = 4294967295; BitOffset_8060 = 0; BitLength_8060 = 0; Address_8060 = ''; Type_8060 = ''; AddressPointer_8060 = 0; AdrOffset_8070 = 4294967295; BitOffset_8070 = 0; BitLength_8070 = 0; Address_8070 = ''; Type_8070 = ''; AddressPointer_8070 = 0; AdrOffset_8080 = 4294967295; BitOffset_8080 = 0; BitLength_8080 = 0; Address_8080 = ''; Type_8080 = ''; AddressPointer_8080 = 0; AdrOffset_8090 = 4294967295; BitOffset_8090 = 0; BitLength_8090 = 0; Address_8090 = ''; Type_8090 = ''; AddressPointer_8090 = 0; AdrOffset_8510 = 172; BitOffset_8510 = 0; BitLength_8510 = 16; Address_8510 = '%IW86'; Type_8510 = 'UINT'; AddressPointer_8510 = ADR(%IW86); AdrOffset_8520 = 176; BitOffset_8520 = 0; BitLength_8520 = 32; Address_8520 = '%ID44'; Type_8520 = 'DINT'; AddressPointer_8520 = ADR(%ID44); AdrOffset_8530 = 180; BitOffset_8530 = 0;
              BitLength_8530 = 32; Address_8530 = '%ID45'; Type_8530 = 'DINT'; AddressPointer_8530 = ADR(%ID45); AdrOffset_8540 = 184; BitOffset_8540 = 0; BitLength_8540 = 16; Address_8540 = '%IW92'; Type_8540 = 'INT'; AddressPointer_8540 = ADR(%IW92); AdrOffset_8550 = 186; BitOffset_8550 = 0; BitLength_8550 = 8; Address_8550 = '%IB186'; Type_8550 = 'SINT'; AddressPointer_8550 = ADR(%IB186); AdrOffset_8560 = 4294967295; BitOffset_8560 = 0; BitLength_8560 = 0; Address_8560 = ''; Type_8560 = ''; AddressPointer_8560 = 0; AdrOffset_8570 = 4294967295; BitOffset_8570 = 0; BitLength_8570 = 0; Address_8570 = ''; Type_8570 = ''; AddressPointer_8570 = 0; AdrOffset_8580 = 4294967295; BitOffset_8580 = 0; BitLength_8580 = 0; Address_8580 = ''; Type_8580 = ''; AddressPointer_8580 = 0; AdrOffset_8590 = 4294967295; BitOffset_8590 = 0; BitLength_8590 = 0; Address_8590 = ''; Type_8590 = ''; AddressPointer_8590 = 0;
              AdrOffset_8600 = 4294967295; BitOffset_8600 = 0; BitLength_8600 = 0; Address_8600 = ''; Type_8600 = ''; AddressPointer_8600 = 0; AdrOffset_8600 = 4294967295; BitOffset_8600 = 0; BitLength_8600 = 0; Address_8610 = ''; Type_8610 = ''; AddressPointer_8610 = 0; AdrOffset_8620 = 4294967295; BitOffset_8620 = 0; BitLength_8620 = 0; Address_8620 = ''; Type_8620 = ''; AddressPointer_8620 = 0
      XINJE_DS5C1_CoE_Drive_Rev4_0_B1 : XINJE-DS5C1 EtherCAT(CoE) Drive Rev4.0 v3.7.70, Xinje Electronics, Inc., order no. XINJE-DS5C1 CoE Drive Rev4.0, version Revision=16#20201207
          settings: EnableExpertSettings = True; StationAlias = 1007; DeviceIdenticationADO = 18; DeviceIdenticationMode = 1; DC sync0 cycletime = 8000; DC sync1 cycletime = 8000; Number of SDO = 4; Homing method.Index = 16#6098; Homing method.Subindex = 16#00; Homing method.Value = 35; Homing method.Size = 8; Homing method.AbortIfError = FALSE; Homing method.JumpToLine = FALSE; Homing method.Line = 0; Homing method.CompleteAccess = False; Op mode.Index = 16#6060; Op mode.Subindex = 16#00; Op mode.Value = 8; Op mode.Size = 8; Op mode.AbortIfError = FALSE; Op mode.JumpToLine = FALSE; Op mode.Line = 0; Op mode.CompleteAccess = False; Interpolation time period.Index = 16#60C2; Interpolation time period.Subindex = 16#01; Interpolation time period.Value = 8; Interpolation time period.Size = 8; Interpolation time period.AbortIfError = FALSE; Interpolation time period.JumpToLine = FALSE; Interpolation time period.Line = 0; Interpolation time period.CompleteAccess = False; Interpolation time index.Index = 16#60C2; Interpolation time index.Subindex = 16#02; Interpolation time index.Value = 253; Interpolation time index.Size = 8; Interpolation time index.AbortIfError = FALSE; Interpolation time index.JumpToLine = FALSE; Interpolation time index.Line = 0; Interpolation time index.CompleteAccess = False
          unmapped channels: Control Word, TargetPosition, TargetVelocity, TargetTorque, ModeOfOperation, Status Word, ActualPosition, Velocity actual value, ActualTorque, ModeOfOperationDisplay
        B1 : SM_Drive_GenericDSP402, 3S - Smart Software Solutions GmbH, order no. 0, version 4.6.1.0
            settings: wDriveID = 8; dwRatioTechUnitsDenom = 327680; iRatioTechUnitsNum = 9; eRampType = 2; fSWMaxVelocity = 140; fSWMaxAcceleration = 400; fSWMaxDeceleration = 400; fSWMaxJerk = 400; ScalingIncs = 131072; ScalingMotorTurns2 = 100; ScalingUnits = 360; AdrOffset_8010 = 536; BitOffset_8010 = 0; BitLength_8010 = 16; Address_8010 = '%QW268'; Type_8010 = 'UINT'; AddressPointer_8010 = ADR(%QW268); AdrOffset_8020 = 540; BitOffset_8020 = 0; BitLength_8020 = 32; Address_8020 = '%QD135'; Type_8020 = 'DINT'; AddressPointer_8020 = ADR(%QD135); AdrOffset_8030 = 544; BitOffset_8030 = 0; BitLength_8030 = 32; Address_8030 = '%QD136'; Type_8030 = 'DINT'; AddressPointer_8030 = ADR(%QD136); AdrOffset_8040 = 548; BitOffset_8040 = 0; BitLength_8040 = 16; Address_8040 = '%QW274'; Type_8040 = 'INT'; AddressPointer_8040 = ADR(%QW274); AdrOffset_8050 = 550; BitOffset_8050 = 0; BitLength_8050 = 8; Address_8050 = '%QB550'; Type_8050 = 'SINT';
              AddressPointer_8050 = ADR(%QB550); AdrOffset_8060 = 4294967295; BitOffset_8060 = 0; BitLength_8060 = 0; Address_8060 = ''; Type_8060 = ''; AddressPointer_8060 = 0; AdrOffset_8070 = 4294967295; BitOffset_8070 = 0; BitLength_8070 = 0; Address_8070 = ''; Type_8070 = ''; AddressPointer_8070 = 0; AdrOffset_8080 = 4294967295; BitOffset_8080 = 0; BitLength_8080 = 0; Address_8080 = ''; Type_8080 = ''; AddressPointer_8080 = 0; AdrOffset_8090 = 4294967295; BitOffset_8090 = 0; BitLength_8090 = 0; Address_8090 = ''; Type_8090 = ''; AddressPointer_8090 = 0; AdrOffset_8510 = 188; BitOffset_8510 = 0; BitLength_8510 = 16; Address_8510 = '%IW94'; Type_8510 = 'UINT'; AddressPointer_8510 = ADR(%IW94); AdrOffset_8520 = 192; BitOffset_8520 = 0; BitLength_8520 = 32; Address_8520 = '%ID48'; Type_8520 = 'DINT'; AddressPointer_8520 = ADR(%ID48); AdrOffset_8530 = 196; BitOffset_8530 = 0; BitLength_8530 = 32;
              Address_8530 = '%ID49'; Type_8530 = 'DINT'; AddressPointer_8530 = ADR(%ID49); AdrOffset_8540 = 200; BitOffset_8540 = 0; BitLength_8540 = 16; Address_8540 = '%IW100'; Type_8540 = 'INT'; AddressPointer_8540 = ADR(%IW100); AdrOffset_8550 = 202; BitOffset_8550 = 0; BitLength_8550 = 8; Address_8550 = '%IB202'; Type_8550 = 'SINT'; AddressPointer_8550 = ADR(%IB202); AdrOffset_8560 = 4294967295; BitOffset_8560 = 0; BitLength_8560 = 0; Address_8560 = ''; Type_8560 = ''; AddressPointer_8560 = 0; AdrOffset_8570 = 4294967295; BitOffset_8570 = 0; BitLength_8570 = 0; Address_8570 = ''; Type_8570 = ''; AddressPointer_8570 = 0; AdrOffset_8580 = 4294967295; BitOffset_8580 = 0; BitLength_8580 = 0; Address_8580 = ''; Type_8580 = ''; AddressPointer_8580 = 0; AdrOffset_8590 = 4294967295; BitOffset_8590 = 0; BitLength_8590 = 0; Address_8590 = ''; Type_8590 = ''; AddressPointer_8590 = 0; AdrOffset_8600 = 4294967295;
              BitOffset_8600 = 0; BitLength_8600 = 0; Address_8600 = ''; Type_8600 = ''; AddressPointer_8600 = 0; AdrOffset_8600 = 4294967295; BitOffset_8600 = 0; BitLength_8600 = 0; Address_8610 = ''; Type_8610 = ''; AddressPointer_8610 = 0; AdrOffset_8620 = 4294967295; BitOffset_8620 = 0; BitLength_8620 = 0; Address_8620 = ''; Type_8620 = ''; AddressPointer_8620 = 0
      XINJE_DS5C1_CoE_Drive_Rev4_0_B2 : XINJE-DS5C1 EtherCAT(CoE) Drive Rev4.0 v3.7.70, Xinje Electronics, Inc., order no. XINJE-DS5C1 CoE Drive Rev4.0, version Revision=16#20201207
          settings: EnableExpertSettings = True; StationAlias = 1008; DeviceIdenticationADO = 18; DeviceIdenticationMode = 1; DC sync0 cycletime = 8000; DC sync1 cycletime = 8000; Number of SDO = 4; Homing method.Index = 16#6098; Homing method.Subindex = 16#00; Homing method.Value = 35; Homing method.Size = 8; Homing method.AbortIfError = FALSE; Homing method.JumpToLine = FALSE; Homing method.Line = 0; Homing method.CompleteAccess = False; Op mode.Index = 16#6060; Op mode.Subindex = 16#00; Op mode.Value = 8; Op mode.Size = 8; Op mode.AbortIfError = FALSE; Op mode.JumpToLine = FALSE; Op mode.Line = 0; Op mode.CompleteAccess = False; Interpolation time period.Index = 16#60C2; Interpolation time period.Subindex = 16#01; Interpolation time period.Value = 8; Interpolation time period.Size = 8; Interpolation time period.AbortIfError = FALSE; Interpolation time period.JumpToLine = FALSE; Interpolation time period.Line = 0; Interpolation time period.CompleteAccess = False; Interpolation time index.Index = 16#60C2; Interpolation time index.Subindex = 16#02; Interpolation time index.Value = 253; Interpolation time index.Size = 8; Interpolation time index.AbortIfError = FALSE; Interpolation time index.JumpToLine = FALSE; Interpolation time index.Line = 0; Interpolation time index.CompleteAccess = False
          unmapped channels: Control Word, TargetPosition, TargetVelocity, TargetTorque, ModeOfOperation, Status Word, ActualPosition, Velocity actual value, ActualTorque, ModeOfOperationDisplay
        B2 : SM_Drive_GenericDSP402, 3S - Smart Software Solutions GmbH, order no. 0, version 4.6.1.0
            settings: wDriveID = 9; dwRatioTechUnitsDenom = 32768; iRatioTechUnitsNum = 5; eRampType = 2; fSWMaxVelocity = 500; fSWMaxAcceleration = 2000; fSWMaxDeceleration = 2000; ScalingIncs = 131072; ScalingUnits = 20; AdrOffset_8010 = 552; BitOffset_8010 = 0; BitLength_8010 = 16; Address_8010 = '%QW276'; Type_8010 = 'UINT'; AddressPointer_8010 = ADR(%QW276); AdrOffset_8020 = 556; BitOffset_8020 = 0; BitLength_8020 = 32; Address_8020 = '%QD139'; Type_8020 = 'DINT'; AddressPointer_8020 = ADR(%QD139); AdrOffset_8030 = 560; BitOffset_8030 = 0; BitLength_8030 = 32; Address_8030 = '%QD140'; Type_8030 = 'DINT'; AddressPointer_8030 = ADR(%QD140); AdrOffset_8040 = 564; BitOffset_8040 = 0; BitLength_8040 = 16; Address_8040 = '%QW282'; Type_8040 = 'INT'; AddressPointer_8040 = ADR(%QW282); AdrOffset_8050 = 566; BitOffset_8050 = 0; BitLength_8050 = 8; Address_8050 = '%QB566'; Type_8050 = 'SINT'; AddressPointer_8050 = ADR(%QB566); AdrOffset_8060 = 4294967295;
              BitOffset_8060 = 0; BitLength_8060 = 0; Address_8060 = ''; Type_8060 = ''; AddressPointer_8060 = 0; AdrOffset_8070 = 4294967295; BitOffset_8070 = 0; BitLength_8070 = 0; Address_8070 = ''; Type_8070 = ''; AddressPointer_8070 = 0; AdrOffset_8080 = 4294967295; BitOffset_8080 = 0; BitLength_8080 = 0; Address_8080 = ''; Type_8080 = ''; AddressPointer_8080 = 0; AdrOffset_8090 = 4294967295; BitOffset_8090 = 0; BitLength_8090 = 0; Address_8090 = ''; Type_8090 = ''; AddressPointer_8090 = 0; AdrOffset_8510 = 204; BitOffset_8510 = 0; BitLength_8510 = 16; Address_8510 = '%IW102'; Type_8510 = 'UINT'; AddressPointer_8510 = ADR(%IW102); AdrOffset_8520 = 208; BitOffset_8520 = 0; BitLength_8520 = 32; Address_8520 = '%ID52'; Type_8520 = 'DINT'; AddressPointer_8520 = ADR(%ID52); AdrOffset_8530 = 212; BitOffset_8530 = 0; BitLength_8530 = 32; Address_8530 = '%ID53'; Type_8530 = 'DINT';
              AddressPointer_8530 = ADR(%ID53); AdrOffset_8540 = 216; BitOffset_8540 = 0; BitLength_8540 = 16; Address_8540 = '%IW108'; Type_8540 = 'INT'; AddressPointer_8540 = ADR(%IW108); AdrOffset_8550 = 218; BitOffset_8550 = 0; BitLength_8550 = 8; Address_8550 = '%IB218'; Type_8550 = 'SINT'; AddressPointer_8550 = ADR(%IB218); AdrOffset_8560 = 4294967295; BitOffset_8560 = 0; BitLength_8560 = 0; Address_8560 = ''; Type_8560 = ''; AddressPointer_8560 = 0; AdrOffset_8570 = 4294967295; BitOffset_8570 = 0; BitLength_8570 = 0; Address_8570 = ''; Type_8570 = ''; AddressPointer_8570 = 0; AdrOffset_8580 = 4294967295; BitOffset_8580 = 0; BitLength_8580 = 0; Address_8580 = ''; Type_8580 = ''; AddressPointer_8580 = 0; AdrOffset_8590 = 4294967295; BitOffset_8590 = 0; BitLength_8590 = 0; Address_8590 = ''; Type_8590 = ''; AddressPointer_8590 = 0; AdrOffset_8600 = 4294967295; BitOffset_8600 = 0; BitLength_8600 = 0;
              Address_8600 = ''; Type_8600 = ''; AddressPointer_8600 = 0; AdrOffset_8600 = 4294967295; BitOffset_8600 = 0; BitLength_8600 = 0; Address_8610 = ''; Type_8610 = ''; AddressPointer_8610 = 0; AdrOffset_8620 = 4294967295; BitOffset_8620 = 0; BitLength_8620 = 0; Address_8620 = ''; Type_8620 = ''; AddressPointer_8620 = 0
      XINJE_DS5C1_CoE_Drive_Rev4_0_B3 : XINJE-DS5C1 EtherCAT(CoE) Drive Rev4.0 v3.7.70, Xinje Electronics, Inc., order no. XINJE-DS5C1 CoE Drive Rev4.0, version Revision=16#20201207
          settings: EnableExpertSettings = True; StationAlias = 1009; DeviceIdenticationADO = 18; DeviceIdenticationMode = 1; DC sync0 cycletime = 8000; DC sync1 cycletime = 8000; Number of SDO = 4; Homing method.Index = 16#6098; Homing method.Subindex = 16#00; Homing method.Value = 35; Homing method.Size = 8; Homing method.AbortIfError = FALSE; Homing method.JumpToLine = FALSE; Homing method.Line = 0; Homing method.CompleteAccess = False; Op mode.Index = 16#6060; Op mode.Subindex = 16#00; Op mode.Value = 8; Op mode.Size = 8; Op mode.AbortIfError = FALSE; Op mode.JumpToLine = FALSE; Op mode.Line = 0; Op mode.CompleteAccess = False; Interpolation time period.Index = 16#60C2; Interpolation time period.Subindex = 16#01; Interpolation time period.Value = 8; Interpolation time period.Size = 8; Interpolation time period.AbortIfError = FALSE; Interpolation time period.JumpToLine = FALSE; Interpolation time period.Line = 0; Interpolation time period.CompleteAccess = False; Interpolation time index.Index = 16#60C2; Interpolation time index.Subindex = 16#02; Interpolation time index.Value = 253; Interpolation time index.Size = 8; Interpolation time index.AbortIfError = FALSE; Interpolation time index.JumpToLine = FALSE; Interpolation time index.Line = 0; Interpolation time index.CompleteAccess = False
          unmapped channels: Control Word, TargetPosition, TargetVelocity, TargetTorque, ModeOfOperation, Status Word, ActualPosition, Velocity actual value, ActualTorque, ModeOfOperationDisplay
        B3 : SM_Drive_GenericDSP402, 3S - Smart Software Solutions GmbH, order no. 0, version 4.6.1.0
            settings: wDriveID = 10; dwRatioTechUnitsDenom = 65536; iRatioTechUnitsNum = 45; eRampType = 2; fSWMaxVelocity = 2000; fSWMaxAcceleration = 4000; fSWMaxDeceleration = 4000; fSWMaxJerk = 4000; ScalingIncs = 131072; ScalingMotorTurns2 = 4; ScalingUnits = 360; AdrOffset_8010 = 568; BitOffset_8010 = 0; BitLength_8010 = 16; Address_8010 = '%QW284'; Type_8010 = 'UINT'; AddressPointer_8010 = ADR(%QW284); AdrOffset_8020 = 572; BitOffset_8020 = 0; BitLength_8020 = 32; Address_8020 = '%QD143'; Type_8020 = 'DINT'; AddressPointer_8020 = ADR(%QD143); AdrOffset_8030 = 576; BitOffset_8030 = 0; BitLength_8030 = 32; Address_8030 = '%QD144'; Type_8030 = 'DINT'; AddressPointer_8030 = ADR(%QD144); AdrOffset_8040 = 580; BitOffset_8040 = 0; BitLength_8040 = 16; Address_8040 = '%QW290'; Type_8040 = 'INT'; AddressPointer_8040 = ADR(%QW290); AdrOffset_8050 = 582; BitOffset_8050 = 0; BitLength_8050 = 8; Address_8050 = '%QB582'; Type_8050 = 'SINT';
              AddressPointer_8050 = ADR(%QB582); AdrOffset_8060 = 4294967295; BitOffset_8060 = 0; BitLength_8060 = 0; Address_8060 = ''; Type_8060 = ''; AddressPointer_8060 = 0; AdrOffset_8070 = 4294967295; BitOffset_8070 = 0; BitLength_8070 = 0; Address_8070 = ''; Type_8070 = ''; AddressPointer_8070 = 0; AdrOffset_8080 = 4294967295; BitOffset_8080 = 0; BitLength_8080 = 0; Address_8080 = ''; Type_8080 = ''; AddressPointer_8080 = 0; AdrOffset_8090 = 4294967295; BitOffset_8090 = 0; BitLength_8090 = 0; Address_8090 = ''; Type_8090 = ''; AddressPointer_8090 = 0; AdrOffset_8510 = 220; BitOffset_8510 = 0; BitLength_8510 = 16; Address_8510 = '%IW110'; Type_8510 = 'UINT'; AddressPointer_8510 = ADR(%IW110); AdrOffset_8520 = 224; BitOffset_8520 = 0; BitLength_8520 = 32; Address_8520 = '%ID56'; Type_8520 = 'DINT'; AddressPointer_8520 = ADR(%ID56); AdrOffset_8530 = 228; BitOffset_8530 = 0; BitLength_8530 = 32;
              Address_8530 = '%ID57'; Type_8530 = 'DINT'; AddressPointer_8530 = ADR(%ID57); AdrOffset_8540 = 232; BitOffset_8540 = 0; BitLength_8540 = 16; Address_8540 = '%IW116'; Type_8540 = 'INT'; AddressPointer_8540 = ADR(%IW116); AdrOffset_8550 = 234; BitOffset_8550 = 0; BitLength_8550 = 8; Address_8550 = '%IB234'; Type_8550 = 'SINT'; AddressPointer_8550 = ADR(%IB234); AdrOffset_8560 = 4294967295; BitOffset_8560 = 0; BitLength_8560 = 0; Address_8560 = ''; Type_8560 = ''; AddressPointer_8560 = 0; AdrOffset_8570 = 4294967295; BitOffset_8570 = 0; BitLength_8570 = 0; Address_8570 = ''; Type_8570 = ''; AddressPointer_8570 = 0; AdrOffset_8580 = 4294967295; BitOffset_8580 = 0; BitLength_8580 = 0; Address_8580 = ''; Type_8580 = ''; AddressPointer_8580 = 0; AdrOffset_8590 = 4294967295; BitOffset_8590 = 0; BitLength_8590 = 0; Address_8590 = ''; Type_8590 = ''; AddressPointer_8590 = 0; AdrOffset_8600 = 4294967295;
              BitOffset_8600 = 0; BitLength_8600 = 0; Address_8600 = ''; Type_8600 = ''; AddressPointer_8600 = 0; AdrOffset_8600 = 4294967295; BitOffset_8600 = 0; BitLength_8600 = 0; Address_8610 = ''; Type_8610 = ''; AddressPointer_8610 = 0; AdrOffset_8620 = 4294967295; BitOffset_8620 = 0; BitLength_8620 = 0; Address_8620 = ''; Type_8620 = ''; AddressPointer_8620 = 0
    Ethernet : Ethernet, CODESYS, version 4.2.0.0
        settings: IPAddress = [192,168,3,6]; SubnetMask = [255,255,255,0]; GatewayAddress = [0,0,0,0]; MACAddress = [16#00,16#00,16#00,16#00,16#00,16#00]; SaveCommunicationSettings = FALSE
      Modbus_TCP_Master : Modbus TCP Master, 3S - Smart Software Solutions GmbH, version 4.3.0.0
      ModbusTCP_Slave_Device : ModbusTCP Slave Device, 3S - Smart Software Solutions GmbH, version 4.3.0.0
          settings: UpdateableHolding = TRUE
          unmapped channels: Holding Registers, Input Registers
    SoftMotion General Axis Pool
      SMC_FreeEncoder : SMC_FreeEncoder, 3S - Smart Software Solutions GmbH, order no. 1805, version 4.14.0.0
          settings: wDriveID = 22; dwRatioTechUnitsDenom = 800000; iRatioTechUnitsNum = -19007; ScalingIncs = 800000; ScalingUnits = 19007; InvertDirection = TRUE
        SM_Drive_Logical : SM_Drive_Logical, 3S - Smart Software Solutions GmbH, order no. 1805, version 4.14.0.0
            settings: wDriveID = 23; iMovementType = 1; fTimeShiftCycles = 0
      SMC_FreeEncoder_B : SMC_FreeEncoder, 3S - Smart Software Solutions GmbH, order no. 1805, version 4.14.0.0
          settings: wDriveID = 24; dwRatioTechUnitsDenom = 800000; iRatioTechUnitsNum = -19007; ScalingIncs = 800000; ScalingUnits = 19007; InvertDirection = TRUE
        SM_Drive_Logical_B : SM_Drive_Logical, 3S - Smart Software Solutions GmbH, order no. 1805, version 4.14.0.0
            settings: wDriveID = 25; iMovementType = 1; fTimeShiftCycles = 0
  global_bonus/
*)

// Just_Motion_Control_x86_64_Linux_SM_WV/Application/ENUM/E_AppCoordSystem
{attribute 'qualified_only'}
{attribute 'strict'}
TYPE E_AppCoordSystem :
(
    APP_COORD_NONE := 0,             // Chưa xác định hệ tọa độ.

    APP_COORD_ROBOT_BASE := 10,       // Hệ tọa độ gốc robot.
    APP_COORD_WORK := 20,             // Hệ tọa độ làm việc.
    APP_COORD_TOOL := 30,             // Hệ tọa độ tool.
    APP_COORD_CAMERA := 40,           // Hệ tọa độ camera.
    APP_COORD_CONVEYOR := 50,         // Hệ tọa độ tĩnh của conveyor.
    APP_COORD_PCS1 := 60,             // Dynamic PCS số 1.
    APP_COORD_PCS2 := 70              // Dynamic PCS số 2.
);
END_TYPE

// Just_Motion_Control_x86_64_Linux_SM_WV/Application/ENUM/E_ApplicationState
{attribute 'qualified_only'}
{attribute 'strict'}
TYPE E_ApplicationState :
(
    APP_IDLE := 0,                    // Application Manager đang rảnh.

    APP_ACCEPT_REQUEST := 10,          // Tiếp nhận yêu cầu từ Interpreter.
    APP_PREPARE := 20,                 // Chuẩn bị camera, job và dữ liệu capture.
    APP_START_VISION := 30,            // Phát yêu cầu tới Vision Manager.
    APP_WAIT_VISION := 40,             // Chờ Vision Manager hoàn thành.
    APP_PROCESS_RESULT := 50,          // Phân loại và xử lý kết quả vision.
    APP_PREPARE_MOTION := 60,          // Chuẩn bị offset, path hoặc object.
    APP_EXECUTE := 70,                 // Thực hiện ứng dụng tương ứng.
    APP_WAIT_COMPLETE := 80,           // Chờ module con hoàn thành.
    APP_COMPLETE := 90,                // Toàn bộ yêu cầu hoàn thành.
    APP_ABORTING := 100,               // Đang hủy ứng dụng.
    APP_RESETTING := 110,              // Đang reset các module liên quan.

    APP_ERROR := 900                   // Application Manager gặp lỗi.
);
END_TYPE

// Just_Motion_Control_x86_64_Linux_SM_WV/Application/ENUM/E_MoveState
{attribute 'qualified_only'}
{attribute 'strict'}
TYPE E_MoveState :
(
	MOVE_IDLE := 0,
    MOVE_LOAD := 10,
    MOVE_SEND := 20,
    MOVE_WAIT_ACCEPT := 30,
    MOVE_WAIT_DONE := 40,
    MOVE_CHECK_POS := 50,
    MOVE_DONE := 60,
    MOVE_ERROR := 90,
    MOVE_TIMEOUT := 91,
    MOVE_ABORTED := 92
);
END_TYPE

// Just_Motion_Control_x86_64_Linux_SM_WV/Application/ENUM/E_ObjectSelectMode
{attribute 'qualified_only'}
{attribute 'strict'}
TYPE E_ObjectSelectMode :
(
    SELECT_NONE := 0,                  // Chưa chọn phương pháp.

    SELECT_FIRST_IN_QUEUE := 10,       // Chọn object vào queue sớm nhất.
    SELECT_NEAREST_PICK_ZONE := 20,    // Chọn object gần vùng gắp nhất.
    SELECT_HIGHEST_SCORE := 30,        // Chọn object có vision score cao nhất.
    SELECT_LOWEST_OBJECT_ID := 40,     // Chọn ObjectID nhỏ nhất.
    SELECT_SPECIFIC_ID := 50           // Chọn theo ObjectID được chỉ định.
);
END_TYPE

// Just_Motion_Control_x86_64_Linux_SM_WV/Application/ENUM/E_QueueResult
{attribute 'qualified_only'}
{attribute 'strict'}
TYPE E_QueueResult :
(
    QUEUE_RESULT_NONE := 0,          // Chưa thực hiện thao tác queue.

    QUEUE_RESULT_OK := 10,            // Thao tác thành công.
    QUEUE_RESULT_FULL := 20,          // Queue không còn slot trống.
    QUEUE_RESULT_EMPTY := 30,         // Queue không có object.
    QUEUE_RESULT_NOT_FOUND := 40,     // Không tìm thấy object yêu cầu.
    QUEUE_RESULT_ALREADY_RESERVED := 50, // Object đã được module khác giữ.
    QUEUE_RESULT_INVALID_ID := 60,    // ObjectID hoặc TriggerID không hợp lệ.

    QUEUE_RESULT_ERROR := 900         // Lỗi queue không xác định.
);
END_TYPE

// Just_Motion_Control_x86_64_Linux_SM_WV/Application/ENUM/E_SystemTestStage
{attribute 'qualified_only'}
{attribute 'strict'}
TYPE E_SystemTestStage :
(
    TEST_NONE := 0,                    // Không chạy kiểm thử module.

    TEST_VISION_COMM := 10,             // Kiểm tra handshake vision.
    TEST_VISION_ALIGN := 20,            // Kiểm tra kết quả align.
    TEST_VISION_INSPECTION := 30,       // Kiểm tra PASS/FAIL.
    TEST_GLUE_PATH_RECEIVE := 40,       // Kiểm tra nhận dữ liệu path.
    TEST_GLUE_STATIC_DRY_RUN := 50,     // Chạy path tĩnh, không bật keo.
    TEST_CONVEYOR_AXIS := 60,           // Kiểm tra AXIS_6 và encoder.
    TEST_TRACK_SINGLE_DRY_RUN := 70,    // Tracking một object, không gắp thật.
    TEST_TRACK_SINGLE_PICK := 80,       // Tracking và gắp một object.
    TEST_TRACK_QUEUE := 90,             // Tracking nhiều object.
    TEST_CONVEYOR_INSPECTION := 100,    // Inspection trên conveyor.
    TEST_CONVEYOR_GLUE_DRY_RUN := 110,  // Bôi keo tracking nhưng chưa bật keo.
    TEST_CONVEYOR_GLUE := 120            // Chạy đầy đủ bôi keo trên conveyor.
);
END_TYPE

// Just_Motion_Control_x86_64_Linux_SM_WV/Application/ENUM/Application/E_ApplicationID
{attribute 'qualified_only'}
{attribute 'strict'}
TYPE E_ApplicationID :
(
	APP_NONE := 0,
    APP_VISION_ALIGN := 10,
    APP_INSPECTION := 20,
    APP_CONVEYOR_PICK := 30,
    APP_GLUE := 40

);
END_TYPE

// Just_Motion_Control_x86_64_Linux_SM_WV/Application/ENUM/Application/E_ApplicationManagerState
{attribute 'qualified_only'}
{attribute 'strict'}
TYPE E_ApplicationManagerState :
(
	APPM_IDLE := 0,
    APPM_START := 10,
    APPM_RUNNING := 20,
    APPM_COMPLETE := 30,
    APPM_ABORTING := 40,
    APPM_ERROR := 900

);
END_TYPE

// Just_Motion_Control_x86_64_Linux_SM_WV/Application/ENUM/Application/E_ApplicationSimulationMode
{attribute 'qualified_only'}
{attribute 'strict'}
TYPE E_ApplicationSimulationMode :
(
	SIM_OFF := 0,          // Robot, encoder, vision và IO thật.
    SIM_LOGIC_ONLY := 10,  // Không chạy robot; motion tự Accepted/Done.
    SIM_ROBOT_REAL := 20   // Robot thật; encoder, object và vacuum giả.

);
END_TYPE

// Just_Motion_Control_x86_64_Linux_SM_WV/Application/ENUM/Conveyor Tracking/E_ConveyorState
{attribute 'qualified_only'}
{attribute 'strict'}
TYPE E_ConveyorState :
(
    CONV_DISABLED := 0,             // Conveyor chưa được bật trong phần mềm.

    CONV_INITIALIZING := 10,         // Đang kiểm tra AXIS encoder.
    CONV_STANDSTILL := 20,           // Conveyor đang đứng yên.
    CONV_RUNNING_FORWARD := 30,      // Conveyor chạy thuận.
    CONV_RUNNING_REVERSE := 40,      // Conveyor chạy ngược.
    CONV_TRACKING_ACTIVE := 50,      // Có robot đang tracking.
    CONV_STOPPING := 60,             // Conveyor đang giảm tốc hoặc dừng.
    CONV_SIMULATION := 70,           // Đang chạy chế độ mô phỏng.

    CONV_ERROR := 900                // Encoder hoặc conveyor axis lỗi.
);
END_TYPE

// Just_Motion_Control_x86_64_Linux_SM_WV/Application/ENUM/Conveyor Tracking/E_MultiTrackState
//=============================================================================
// ENUM: MULTI-TOOL TRACKING STATE
//-----------------------------------------------------------------------------
// State machine của FB_MultiToolTrackingApplication.
//=============================================================================
{attribute 'qualified_only'}
{attribute 'strict'}
TYPE E_MultiTrackState :
(
    // Chờ lệnh mới.
    IDLE := 0,

    // Đọc Tracking Recipe.
    LOAD_RECIPE := 10,

    // Kiểm tra Tool/Recipe.
    VALIDATE_TOOLS := 20,

    // Chờ Object có trong Queue.
    WAIT_OBJECT := 40,

    // Chọn cặp Tool - Object.
    SELECT_ASSIGNMENT := 50,

    // Chọn TCP của Tool cho Robot.
    SELECT_ROBOT_TOOL := 60,

    // Phát lệnh cho Tracking Core.
    START_TRACKING := 70,

    // Chờ Tracking Core báo đồng bộ.
    WAIT_SYNC := 80,

    // Phát lệnh hạ Tool.
    TOOL_DOWN := 90,

    // Chờ Tool hạ xong.
    WAIT_TOOL_DOWN := 100,

    // Phát lệnh hút/kẹp.
    TOOL_GRIP := 110,

    // Chờ Grip OK.
    WAIT_TOOL_GRIP := 120,

    // Phát lệnh nâng Tool.
    TOOL_UP := 130,

    // Chờ Tool lên an toàn.
    WAIT_TOOL_UP := 140,

    // Yêu cầu Tracking Core thoát PCS.
    RELEASE_TRACKING := 150,

    // Lưu kết quả gắp.
    STORE_RESULT := 160,

    // Kiểm tra đã đủ số lượng chưa.
    CHECK_COUNT := 170,

    // Chu trình hoàn thành.
    COMPLETE := 800,

    // Đang Abort.
    ABORTING := 850,

    // Chu trình lỗi.
    ERROR := 900
);
END_TYPE

// Just_Motion_Control_x86_64_Linux_SM_WV/Application/ENUM/Conveyor Tracking/E_ObjectSourceType
{attribute 'qualified_only'}
{attribute 'strict'}
TYPE E_ObjectSourceType :
(
	// Không sử dụng nguồn Object.
    NONE := 0,

    // Object được phát hiện từ hệ thống Vision.
    VISION := 10,

    // Object được tạo từ Sensor phát hiện sản phẩm.
    SENSOR := 20

);
END_TYPE

// Just_Motion_Control_x86_64_Linux_SM_WV/Application/ENUM/Conveyor Tracking/E_TrackingObjectState
//=============================================================================
// ENUM: TRACKING OBJECT STATE
//-----------------------------------------------------------------------------
// Trạng thái vòng đời của một Object trong Queue.
//=============================================================================
{attribute 'qualified_only'}
{attribute 'strict'}
TYPE E_TrackingObjectState :
(
    
	OBJ_EMPTY := 0,                   // Slot chưa chứa sản phẩm.

    OBJ_CAPTURED := 10,               // Camera đã được trigger và encoder đã được chốt.
    OBJ_WAIT_VISION := 20,            // Đang chờ vision trả kết quả.
    OBJ_DETECTED := 30,               // Vision đã tìm thấy sản phẩm.
    OBJ_INSPECTION_PASS := 40,         // Sản phẩm đã kiểm tra và đạt.
    OBJ_INSPECTION_FAIL := 50,         // Sản phẩm đã kiểm tra và không đạt.
    OBJ_WAIT_PICK_ZONE := 60,          // Sản phẩm chưa vào vùng gắp.
    OBJ_READY := 70,                   // Sản phẩm đã vào vùng gắp.
    OBJ_RESERVED := 80,                // Robot đã giữ quyền xử lý sản phẩm.
    OBJ_PCS_READY := 90,               // Dynamic PCS của sản phẩm đã được tạo.
    OBJ_TRACKING := 100,               // Robot đang bám theo sản phẩm.
    OBJ_PICKING := 110,                // Robot đang thực hiện thao tác gắp.
    OBJ_PICKED := 120,                 // Sản phẩm đã được gắp thành công.
    OBJ_REJECTED := 130,               // Sản phẩm bị loại.
    OBJ_EXPIRED := 140,                // Sản phẩm đã đi quá vùng robot.
	OBJ_MISSED  := 145,				   // Đã được robot chọn nhưng không còn đủ thời gian/vùng an toàn để gắp.
    OBJ_ABORTED := 150,                // Xử lý sản phẩm bị hủy.

    OBJ_ERROR := 900                   // Object gặp lỗi xử lý.
);
END_TYPE

// Just_Motion_Control_x86_64_Linux_SM_WV/Application/ENUM/Conveyor Tracking/E_TrackingSelectMode
{attribute 'qualified_only'}
{attribute 'strict'}
TYPE E_TrackingSelectMode :
(
	// Không tự động chọn object.
    // Chỉ dùng khi Application chỉ định trực tiếp ObjectID.
    TRACK_SELECT_NONE := 0,

    // Chọn object có CaptureTime nhỏ nhất.
    // Tương đương object được camera ghi nhận sớm nhất.
    TRACK_SELECT_FIFO := 10,

    // Chọn object nằm gần giới hạn thoát/AbortPosition nhất.
    // Phù hợp khi ưu tiên cứu object sắp ra khỏi vùng gắp.
    TRACK_SELECT_NEAREST_EXIT := 20,

    // Chọn object có TimeRemainingSec nhỏ nhất.
    // Đây là kiểu Earliest Deadline First.
    TRACK_SELECT_MIN_TIME_REMAIN := 30,

    // Chọn object có Priority lớn nhất.
    // Nếu Priority bằng nhau thì dùng TimeRemainingSec nhỏ hơn.
    TRACK_SELECT_HIGHEST_PRIORITY := 40,

    // Chọn object có VisionScore lớn nhất.
    // Nếu VisionScore bằng nhau thì dùng TimeRemainingSec nhỏ hơn.
    TRACK_SELECT_HIGHEST_VISION_SCORE := 50,

    // Chọn object có EstimatedPickTimeSec nhỏ nhất.
    // Dùng khi vị trí object khác nhau làm thời gian robot tiếp cận khác nhau.
    TRACK_SELECT_SHORTEST_PICK_TIME := 60,

    // Chọn đúng ObjectID do Application yêu cầu.
    TRACK_SELECT_SPECIFIC_ID := 70
);
END_TYPE

// Just_Motion_Control_x86_64_Linux_SM_WV/Application/ENUM/Conveyor Tracking/E_TrackingState
{attribute 'qualified_only'}
{attribute 'strict'}
TYPE E_TrackingState :
(
    // Manager đang chờ lệnh chạy.
    TRK_IDLE := 0,

    // Tìm object phù hợp trong Queue.
    TRK_FIND_OBJECT := 10,

    // Khóa quyền sở hữu object đã chọn.
    TRK_RESERVE_OBJECT := 20,

    // Chờ object nằm trong vùng gắp an toàn.
    TRK_WAIT_PICK_ZONE := 30,

    // Chuẩn bị dữ liệu PCS và các điểm Approach/Pick/Retract.
    TRK_PREPARE_PCS := 40,

    // Phát Execute cho MC_TrackConveyorBelt.
    TRK_CREATE_PCS := 50,

    // Chờ PCS động được tạo thành công.
    TRK_WAIT_PCS := 60,

    // Di chuyển tới điểm phía trên object trong PCS.
    TRK_MOVE_APPROACH := 70,
	
	// Robot đã tới Approach trong PCS; chờ Tool DOWN/GRIP/UP.
    TRK_SYNCHRONIZED := 75,
	
    // Hạ xuống điểm gắp trong PCS.
    TRK_MOVE_PICK := 80,

    // Bật tool hút hoặc lệnh Grip.
    TRK_GRIP_ON := 90,

    // Chờ xác nhận tool đã giữ được vật.
    TRK_WAIT_GRIP := 100,

    // Nâng vật lên trong PCS sau khi gắp.
    TRK_MOVE_RETRACT := 110,

    // Di chuyển ra khỏi vùng tracking sang hệ robot/base.
    TRK_LEAVE_PCS := 120,

    // Chờ PCS không còn được Motion sử dụng rồi hạ Execute tracking.
    TRK_RELEASE_PCS := 130,
	
	// LEAVE PCS Safe
	TRK_MOVE_SAFE_LEAVE := 135,

    // Di chuyển tới điểm đặt sản phẩm trong hệ robot/base.
    TRK_MOVE_PLACE := 140,

    // Tắt hút hoặc phát lệnh Release tool.
    TRK_RELEASE_PRODUCT := 150,

    // Chờ hoàn tất thời gian thổi hoặc nhả.
    TRK_WAIT_BLOW := 160,

    // Hoàn thành xử lý một object.
    TRK_COMPLETE := 170,

    // Abort object active vì chạy quá vùng an toàn.
    TRK_ABORT_ACTIVE := 180,

    // Di chuyển robot về vị trí an toàn sau khi bỏ object.
    TRK_MOVE_SAFE := 190,

    // Giải phóng object MISSED rồi tìm object tiếp theo.
    TRK_RELEASE_OBJECT := 200,

    // Hủy toàn bộ chu trình do Execute bị hạ hoặc có lệnh Stop.
    TRK_ABORTING := 210,

    // Manager đang ở trạng thái lỗi.
    TRK_ERROR := 900
);
END_TYPE

// Just_Motion_Control_x86_64_Linux_SM_WV/Application/ENUM/GlueBonding/E_GlueRunMode
{attribute 'qualified_only'}
{attribute 'strict'}
TYPE E_GlueRunMode :
(
    GLUE_MODE_NONE := 0,              // Chưa chọn chế độ.

    GLUE_MODE_STATIC := 10,            // Sản phẩm đứng yên.
    GLUE_MODE_WORK_OFFSET := 20,       // Đường keo áp dụng work offset.
    GLUE_MODE_CONVEYOR_PCS1 := 30,     // Bôi keo trong PCS_1.
    GLUE_MODE_CONVEYOR_PCS2 := 40,     // Bôi keo trong PCS_2.
    GLUE_MODE_DRY_RUN := 50            // Robot chạy path nhưng không bật keo.
);
END_TYPE

// Just_Motion_Control_x86_64_Linux_SM_WV/Application/ENUM/GlueBonding/E_GlueState
{attribute 'qualified_only'}
{attribute 'strict'}
TYPE E_GlueState :
(
    GLUE_IDLE := 0,                  // Glue Manager đang rảnh.

    GLUE_LOAD_PATH := 10,             // Nạp đường keo.
    GLUE_VALIDATE_PATH := 20,         // Kiểm tra tính hợp lệ của đường keo.
    GLUE_PROCESS_PATH := 30,          // Lọc và chuẩn hóa đường keo.
    GLUE_PREPARE_QUEUE := 40,         // Chuyển path thành Motion Queue.
    GLUE_MOVE_APPROACH := 50,         // Di chuyển tới vị trí approach.
    GLUE_MOVE_START := 60,            // Di chuyển tới điểm đầu đường keo.
    GLUE_PRE_FLOW := 70,              // Mở keo trước khi chạy.
    GLUE_RUN_PATH := 80,              // Chạy đường keo.
    GLUE_POST_FLOW := 90,             // Xử lý đóng keo tại cuối đường.
    GLUE_MOVE_RETRACT := 100,         // Rút robot khỏi sản phẩm.
    GLUE_COMPLETE := 110,             // Bôi keo hoàn thành.
    GLUE_ABORTING := 120,             // Đang dừng quá trình bôi keo.

    GLUE_ERROR := 900                 // Bôi keo gặp lỗi.
);
END_TYPE

// Just_Motion_Control_x86_64_Linux_SM_WV/Application/ENUM/GlueBonding/E_PathProcessState
{attribute 'qualified_only'}
{attribute 'strict'}
TYPE E_PathProcessState :
(
    PATH_PROC_IDLE := 0,              // Bộ xử lý path đang rảnh.

    PATH_PROC_LOAD := 10,              // Nạp dữ liệu điểm thô.
    PATH_PROC_VALIDATE := 20,          // Kiểm tra số điểm và phạm vi tọa độ.
    PATH_PROC_REMOVE_DUPLICATE := 30,  // Loại bỏ điểm trùng.
    PATH_PROC_FILTER := 40,            // Lọc nhiễu vị trí.
    PATH_PROC_RESAMPLE := 50,          // Chia lại khoảng cách giữa các điểm.
    PATH_PROC_SEGMENT := 60,           // Phân loại line, arc hoặc spline.
    PATH_PROC_PLAN_SPEED := 70,        // Tính tốc độ theo từng đoạn.
    PATH_PROC_COMPLETE := 80,          // Path đã xử lý xong.

    PATH_PROC_ERROR := 900             // Dữ liệu path hoặc xử lý bị lỗi.
);
END_TYPE

// Just_Motion_Control_x86_64_Linux_SM_WV/Application/ENUM/GlueBonding/E_PathSegmentType
{attribute 'qualified_only'}
{attribute 'strict'}
TYPE E_PathSegmentType :
(
    PATH_NONE := 0,               // Chưa xác định kiểu đoạn.

    PATH_POINT := 10,             // Một điểm độc lập.
    PATH_LINE := 20,              // Đoạn thẳng tới điểm tiếp theo.
    PATH_ARC_MID_END := 30,       // Cung tròn xác định bởi điểm giữa và điểm cuối.
    PATH_ARC_CW := 40,            // Cung tròn theo chiều kim đồng hồ.
    PATH_ARC_CCW := 50,           // Cung tròn ngược chiều kim đồng hồ.
    PATH_SPLINE := 60,            // Đường spline qua nhiều điểm.
    PATH_BEZIER := 70,            // Đường Bézier.
    PATH_BREAK := 80              // Ngắt quỹ đạo, không nối với đoạn kế tiếp.
);
END_TYPE

// Just_Motion_Control_x86_64_Linux_SM_WV/Application/ENUM/Interpreter/E_CondLink
{attribute 'qualified_only'}
{attribute 'strict'}
TYPE E_CondLink : // Enum liên kết nhiều dòng điều kiện
(
	COND_LINK_NONE := 0,
    COND_LINK_AND  := 1,
    COND_LINK_OR   := 2
);
END_TYPE

// Just_Motion_Control_x86_64_Linux_SM_WV/Application/ENUM/Interpreter/E_CondOperator
{attribute 'qualified_only'}
{attribute 'strict'}
TYPE E_CondOperator :
(
	COND_OP_NONE := 0,
    COND_OP_EQ   := 1,    // =
    COND_OP_NE   := 2,    // <>
    COND_OP_GT   := 3,    // >
    COND_OP_GE   := 4,    // >=
    COND_OP_LT   := 5,    // <
    COND_OP_LE   := 6     // <=
);
END_TYPE

// Just_Motion_Control_x86_64_Linux_SM_WV/Application/ENUM/Interpreter/E_CondSource
{attribute 'qualified_only'}
{attribute 'strict'}
TYPE E_CondSource  :
(
	COND_SRC_NONE := 0,
    COND_SRC_DI   := 1,   // Input
    COND_SRC_DO   := 2,   // Output
    COND_SRC_REG  := 3,   // Register số
    COND_SRC_VAR  := 4,   // Biến nội bộ
    COND_SRC_TIMER:= 5    // Timer
);
END_TYPE

// Just_Motion_Control_x86_64_Linux_SM_WV/Application/ENUM/Interpreter/E_RobotCmd
{attribute 'qualified_only'}
{attribute 'strict'}
TYPE E_RobotCmd :
(
	CMD_NOP := 0,
    CMD_MovP := 1, // Chay PTP
    CMD_MovL := 2, // Chay Linear
	CMD_MovC := 3, // Chay theo cung tron
	CMD_Set_Speed := 4, // Set Toc do
	CMD_Set_Fac_Speed := 5, // Set HS toc do
    CMD_DO_ON := 10, // Output Digital ON
    CMD_DO_OFF := 11, // Output Digital OFF
	CMD_DO_TOGGLE := 12, // Output Digital Reverse
    CMD_WAIT_IN := 13, // Wait Input Signal
    CMD_WAIT := 14, // Wait Condition
	CMD_Delay := 15, // Delay Time
	CMD_Timer_Start := 16, // Timer No
	CMD_Timer_Wait := 17, // Timer No
    CMD_IF := 20, // If loop with condition No
	CMD_IF_IN := 21, // If loop with Input No
	CMD_IF_VAR := 22, // If loop with Variable No
	CMD_IF_REG := 23, // If loop with Reg No
    CMD_ELSE := 24, // Else cmd
	CMD_END_IF := 25, // End of if loop
    CMD_JUMP := 26, // Jump another step
    CMD_CALL := 27, // Call another program
    CMD_RETURN := 28, // Out off Loop
	CMD_WHILE := 29, // While loop with condition No
	CMD_WHILE_IN := 30, // While loop with Input No
	CMD_WHILE_REG := 31, // While loop with Reg No
	CMD_END_WHILE := 32, // End of While loop
    CMD_VISION_TRIGGER := 35, // Trigger VS System
    CMD_VISION_SET_POINT := 36, // Wait Result VS System
	CMD_VISION_PICK := 37, 
	CMD_VISION_CHECK := 38,
    CMD_TRACK_ON := 45, // On Conveyor Tracking
    CMD_TRACK_OFF := 46, // Off Conveyor Tracking
	CMD_TRACK_PICK := 47, 
	CMD_TRACK_PLACE := 48,
	CMD_TOOL_RELEASE := 49, // Nha tool da gap
	CMD_CONV_PICK := 50,
	CMD_REG_SET := 60,
	CMD_REG_ADD := 61,
	CMD_REG_SUB := 62,
	CMD_REG_MUL := 63,
	CMD_REG_DIV := 64,
	CMD_REG_MOD := 65,
	
	CMD_VAR_SET := 70,
	CMD_VAR_ADD := 71,
	CMD_VAR_SUB := 72,
	CMD_VAR_MUL := 73,
	CMD_VAR_DIV := 74,
	CMD_VAR_MOD := 75,
	
	
	CMD_MB_REG_SET         := 77,   // Ghi 1 thanh ghi MODBUS, INT16 signed
	CMD_MB_BIT_SET         := 78,   // Set/Reset 1 bit của thanh ghi MODBUS
	CMD_MB_REG_READ        := 79,   // Doc 1 thanh ghi MODBUS, INT16 signed
	
	CMD_POINT_COPY         := 82,   // Point đích = Point nguồn
	CMD_POINT_ADD          := 83,   // Point đích = Point gốc + Point offset
	CMD_POINT_SUB          := 84,   // Point đích = Point gốc - Point offset
	CMD_POINT_ADD_VALUE    := 85,   // Point đích = Point gốc + X/Y/Z/R nhập trực tiếp
	CMD_POINT_ADD_REG      := 86,   // Point đích = Point gốc + A_Reg/B_Reg X/Y/Z/R
	CMD_POINT_ADD_MB_REG   := 87,   // Point đích = Point gốc + MODBUS X/Y/Z/R


    CMD_END := 999
);
END_TYPE

// Just_Motion_Control_x86_64_Linux_SM_WV/Application/ENUM/TOOL/E_ToolAction
//=============================================================================
// ENUM: TOOL ACTION
//-----------------------------------------------------------------------------
// Lệnh mức cao gửi tới FB_ToolManager.
//=============================================================================
{attribute 'qualified_only'}
{attribute 'strict'}
TYPE E_ToolAction :
(
    // Không có lệnh.
    NONE := 0,

    // Hạ cơ cấu Tool xuống.
    DOWN := 10,

    // Bật hút hoặc đóng kẹp.
    GRIP := 20,

    // Nâng cơ cấu Tool lên.
    UP := 30,

    // Nhả sản phẩm.
    RELEASE := 40,

    // Reset Tool.
    RESET := 100
);
END_TYPE

// Just_Motion_Control_x86_64_Linux_SM_WV/Application/ENUM/TOOL/E_ToolCommandType
//=============================================================================
// ENUM: TOOL COMMAND TYPE
//-----------------------------------------------------------------------------
// Loại lệnh mức cao gửi tới FB_ToolManager.
//=============================================================================
{attribute 'qualified_only'}
{attribute 'strict'}
TYPE E_ToolCommandType :
(
    // Không có lệnh.
    NONE := 0,

    // Hạ cơ cấu Tool xuống.
    DOWN := 10,

    // Bật hút hoặc đóng kẹp.
    GRIP := 20,

    // Nâng cơ cấu Tool lên.
    UP := 30,

    // Nhả sản phẩm.
    RELEASE := 40,

    // Reset Tool.
    RESET := 100
);
END_TYPE

// Just_Motion_Control_x86_64_Linux_SM_WV/Application/ENUM/TOOL/E_ToolRuntimeState
//=============================================================================
// ENUM: TOOL RUNTIME STATE
//=============================================================================
{attribute 'qualified_only'}
{attribute 'strict'}
TYPE E_ToolRuntimeState :
(
    // Tool đang rảnh.
    IDLE := 0,

    // Tool đang hạ xuống.
    DOWNING := 10,

    // Tool đã xuống vị trí dưới.
    DOWN := 20,

    // Tool đang hút hoặc đóng kẹp.
    GRIPPING := 30,

    // Tool đang giữ sản phẩm.
    OCCUPIED := 40,

    // Tool đang nâng lên.
    UPPING := 50,

    // Tool đã ở vị trí trên.
    UP := 60,

    // Tool đang nhả sản phẩm.
    RELEASING := 70,

    // Tool báo lỗi.
    ERROR := 900
);
END_TYPE

// Just_Motion_Control_x86_64_Linux_SM_WV/Application/ENUM/TOOL/E_ToolType
//=============================================================================
// ENUM: TOOL TYPE
//=============================================================================
{attribute 'qualified_only'}
{attribute 'strict'}
TYPE E_ToolType :
(
    // Chưa cấu hình Tool.
    NONE := 0,

    // Tool hút chân không.
    VACUUM := 10,

    // Kẹp một van.
    GRIPPER_SINGLE := 20,

    // Kẹp hai van.
    GRIPPER_DOUBLE := 30,

    // Tool tùy chỉnh.
    CUSTOM := 100
);
END_TYPE

// Just_Motion_Control_x86_64_Linux_SM_WV/Application/ENUM/Vision/E_AlignState
{attribute 'qualified_only'}
{attribute 'strict'}
TYPE E_AlignState :
(
    ALIGN_IDLE := 0,               // Align Manager đang rảnh.

    ALIGN_WAIT_RESULT := 10,        // Chờ kết quả align từ vision.
    ALIGN_VALIDATE := 20,           // Kiểm tra score và giới hạn offset.
    ALIGN_TRANSFORM := 30,          // Chuyển offset từ hệ camera sang hệ robot.
    ALIGN_SET_OFFSET := 40,         // Ghi Work Offset mới.
    ALIGN_COMPLETE := 50,           // Align hoàn thành.

    ALIGN_ERROR := 900              // Kết quả align hoặc phép transform bị lỗi.
);
END_TYPE

// Just_Motion_Control_x86_64_Linux_SM_WV/Application/ENUM/Vision/E_InspectionResult
{attribute 'qualified_only'}
{attribute 'strict'}
TYPE E_InspectionResult :
(
    INS_RESULT_NONE := 0,            // Chưa có kết quả.

    INS_RESULT_PASS := 10,            // Sản phẩm đạt.
    INS_RESULT_FAIL := 20,            // Sản phẩm không đạt.
    INS_RESULT_RETRY := 30,           // Cần chụp lại.
    INS_RESULT_NOT_FOUND := 40,       // Không tìm thấy sản phẩm.
    INS_RESULT_INVALID := 50,         // Dữ liệu kiểm tra không hợp lệ.

    INS_RESULT_ERROR := 900           // Lỗi kiểm tra.
);
END_TYPE

// Just_Motion_Control_x86_64_Linux_SM_WV/Application/ENUM/Vision/E_InspectionState
{attribute 'qualified_only'}
{attribute 'strict'}
TYPE E_InspectionState :
(
    INS_IDLE := 0,                 // Inspection Manager đang rảnh.

    INS_WAIT_RESULT := 10,          // Chờ kết quả vision.
    INS_VALIDATE := 20,             // Kiểm tra cấu trúc dữ liệu trả về.
    INS_EVALUATE := 30,             // Đánh giá từng hạng mục kiểm tra.
    INS_PASS := 40,                 // Sản phẩm đạt yêu cầu.
    INS_REJECT := 50,               // Sản phẩm không đạt.
    INS_RETRY := 60,                // Yêu cầu chụp lại.
    INS_COMPLETE := 70,             // Quá trình inspection hoàn thành.

    INS_ERROR := 900                // Inspection gặp lỗi hệ thống.
);
END_TYPE

// Just_Motion_Control_x86_64_Linux_SM_WV/Application/ENUM/Vision/E_PlaceMode
{attribute 'qualified_only'}
{attribute 'strict'}
//=============================================================================
// ENUM: E_PlaceMode
//=============================================================================
TYPE E_PlaceMode :
(
    PLACE_FIXED := 0,                       // Đặt tại một điểm cố định.
    PLACE_TRAY := 1                         // Đặt vào Tray theo Master + Row/Column offset.
);
END_TYPE

// Just_Motion_Control_x86_64_Linux_SM_WV/Application/ENUM/Vision/E_VisionApplication
{attribute 'qualified_only'}
{attribute 'strict'}
TYPE E_VisionApplication :
(
    VIS_APP_NONE := 0,                    // Chưa chọn ứng dụng vision.

    VIS_APP_ALIGN := 10,                  // Tìm độ lệch X/Y/Z/A để căn chỉnh sản phẩm.
    VIS_APP_INSPECTION := 20,             // Kiểm tra ngoại quan và trả kết quả OK/NG.
    VIS_APP_SINGLE_POINT := 30,           // Tìm và trả về một tọa độ duy nhất.
    VIS_APP_POINT_LIST := 40,             // Trả về danh sách nhiều tọa độ.
    VIS_APP_GLUE_PATH := 50,              // Trả về đường chạy phục vụ bôi keo.
    VIS_APP_PICK_POSITION := 60,           // Tìm tọa độ gắp sản phẩm tĩnh.
    VIS_APP_CONVEYOR_PICK := 70,           // Tìm sản phẩm đang chạy trên conveyor để gắp.
    VIS_APP_CONVEYOR_INSPECTION := 80,     // Kiểm tra sản phẩm khi đang chạy trên conveyor.
    VIS_APP_CONVEYOR_GLUE := 90,           // Trả đường keo của sản phẩm đang chạy.
    VIS_APP_CALIBRATION := 100             // Job dùng để kiểm tra hoặc thực hiện calibration.
);
END_TYPE

// Just_Motion_Control_x86_64_Linux_SM_WV/Application/ENUM/Vision/E_VisionDataType
{attribute 'qualified_only'}
{attribute 'strict'}
TYPE E_VisionDataType :
(
    VIS_DATA_NONE := 0,               // Không có dữ liệu kết quả.

    VIS_DATA_BOOL := 10,               // Chỉ trả kết quả TRUE/FALSE hoặc OK/NG.
    VIS_DATA_VALUE := 20,              // Trả về một giá trị đo.
    VIS_DATA_POS := 30,                // Trả về một tọa độ ST_POS.
    VIS_DATA_ALIGN := 40,              // Trả về offset align X/Y/Z/A và score.
    VIS_DATA_INSPECTION := 50,         // Trả dữ liệu kiểm tra ngoại quan.
    VIS_DATA_POINT_LIST := 60,         // Trả về danh sách các điểm.
    VIS_DATA_GLUE_PATH := 70,          // Trả về dữ liệu đường bôi keo.
    VIS_DATA_TRACK_OBJECT := 80        // Trả về tọa độ object trên conveyor.
);
END_TYPE

// Just_Motion_Control_x86_64_Linux_SM_WV/Application/ENUM/Vision/E_VisionResultStatus
{attribute 'qualified_only'}
{attribute 'strict'}
TYPE E_VisionResultStatus :
(
    VIS_RESULT_NONE := 0,              // Chưa có kết quả.

    VIS_RESULT_PENDING := 10,           // Vision đang xử lý.
    VIS_RESULT_OK := 20,                // Có kết quả hợp lệ.
    VIS_RESULT_NG := 30,                // Kết quả kiểm tra là NG.
    VIS_RESULT_NOT_FOUND := 40,         // Không tìm thấy sản phẩm hoặc đặc trưng.
    VIS_RESULT_LOW_SCORE := 50,         // Score thấp hơn giới hạn.
    VIS_RESULT_OUT_OF_RANGE := 60,      // Tọa độ hoặc giá trị vượt giới hạn.
    VIS_RESULT_INCOMPLETE := 70,        // Dữ liệu nhận chưa đầy đủ.
    VIS_RESULT_INVALID := 80,           // Header hoặc payload không hợp lệ.

    VIS_RESULT_ERROR := 900             // Vision báo lỗi xử lý.
);
END_TYPE

// Just_Motion_Control_x86_64_Linux_SM_WV/Application/ENUM/Vision/E_VisionRobot
{attribute 'qualified_only'}
{attribute 'strict'}
TYPE E_VisionRobot :
(
    VIS_ROBOT_NONE := 0,    // Camera chưa được gán cho Robot.
    VIS_ROBOT_A := 1,       // Camera được gán cho Robot A.
    VIS_ROBOT_B := 2        // Camera được gán cho Robot B.
);
END_TYPE

// Just_Motion_Control_x86_64_Linux_SM_WV/Application/ENUM/Vision/E_VisionState
{attribute 'qualified_only'}
{attribute 'strict'}
TYPE E_VisionState :
(
    VIS_IDLE := 0,                 // Kênh vision đang rảnh.

    VIS_PREPARE := 10,             // Chuẩn bị JobID, TriggerID và vùng dữ liệu.
    VIS_SEND_JOB := 20,            // Gửi JobID sang phần mềm vision.
    VIS_SEND_TRIGGER := 30,        // Phát lệnh trigger camera.
    VIS_WAIT_BUSY := 40,           // Chờ vision xác nhận đang xử lý.
    VIS_WAIT_RESULT := 50,         // Chờ vision báo kết quả sẵn sàng.
    VIS_READ_HEADER := 60,         // Đọc header kết quả.
    VIS_READ_DATA := 70,           // Đọc payload kết quả.
    VIS_READ_BLOCK := 80,          // Đọc từng block khi dữ liệu có nhiều điểm.
    VIS_VALIDATE := 90,            // Kiểm tra TriggerID, số điểm và checksum.
    VIS_ACK_RESULT := 100,          // Xác nhận PLC đã nhận kết quả.
    VIS_DONE := 110,               // Yêu cầu vision hoàn thành.
    VIS_ABORTING := 120,           // Đang hủy yêu cầu vision.
    VIS_RESETTING := 130,          // Đang reset trạng thái giao tiếp.

    VIS_ERROR := 900               // Giao tiếp hoặc dữ liệu vision bị lỗi.
);
END_TYPE

// Just_Motion_Control_x86_64_Linux_SM_WV/Application/STRUCT_/Alarm/Alarm_Robot
TYPE Alarm_Robot :
STRUCT
	A_Tool_1, A_Tool_2, B_Tool_1, B_Tool_2, RB_A_Error, RB_A_A0_Error, RB_A_A1_Error, RB_A_A2_Error, RB_A_A3_Error : BOOL;
	RB_B_Error, RB_B_B0_Error, RB_B_B1_Error, RB_B_B2_Error, RB_B_B3_Error : BOOL;
	No_On_Servo_RB_A, No_On_Servo_RB_B, No_Enable_RB_A, No_Enable_RB_B : BOOL;
END_STRUCT
END_TYPE

// Just_Motion_Control_x86_64_Linux_SM_WV/Application/STRUCT_/Application/ST_APPLICATION_COMMAND
TYPE ST_APPLICATION_COMMAND :
STRUCT
	Execute : BOOL;
    Abort : BOOL;
    Reset : BOOL;
    ApplicationID : E_ApplicationID;
    RecipeID : UINT;
    RobotID : UINT;
    CommandID : UDINT;
END_STRUCT
END_TYPE

// Just_Motion_Control_x86_64_Linux_SM_WV/Application/STRUCT_/Application/ST_APPLICATION_RESPONSE
TYPE ST_APPLICATION_RESPONSE :
STRUCT
	Accepted : BOOL;
    Busy : BOOL;
    Done : BOOL;
    Error : BOOL;
    ErrorID : UDINT;
    ActiveApplication : E_ApplicationID;
    CommandID : UDINT;
    ProgressState : INT;
END_STRUCT
END_TYPE

// Just_Motion_Control_x86_64_Linux_SM_WV/Application/STRUCT_/Array/Pallets_In
TYPE Pallets_In :
STRUCT
	//in 
    ZOrder      : INT; //0:= Z trước hay 1:= Z sau
    RowFirst    : BOOL;// TRUE = Row trước, FALSE = Col trước

    RowCount    : INT;
    ColCount    : INT;
    ZCount      : INT;

    PitchRow    : REAL;
    PitchCol    : REAL;
    PitchZ      : REAL;
	
	Pos_Number	: INT; // of 50 pos teach
    StartX      : REAL;
    StartY      : REAL;
    StartZ      : REAL;
END_STRUCT
END_TYPE

// Just_Motion_Control_x86_64_Linux_SM_WV/Application/STRUCT_/Array/Pallets_Out
TYPE Pallets_Out :
STRUCT
		 // out
	PosX        : REAL;
    PosY        : REAL;
    PosZ        : REAL;
	
	CurrentID   : INT;
    RowIndex    : INT;
    ColIndex    : INT;
    ZIndex      : INT;
	Total		:INT;
END_STRUCT
END_TYPE

// Just_Motion_Control_x86_64_Linux_SM_WV/Application/STRUCT_/CAM/Calib_Cam
TYPE Calib_Cam :
STRUCT
	Enable      : BOOL;
    Start       : BOOL;
    Reset       : BOOL;
	A_Error   : BOOL;
	B_Error   : BOOL;
END_STRUCT
END_TYPE

// Just_Motion_Control_x86_64_Linux_SM_WV/Application/STRUCT_/CAM/Calib_Cam_Input_Model
TYPE Calib_Cam_Input_Model :
STRUCT
	Hand_No     : INT; // 0: Robot A; 1: Robot B
	PointNo1    : INT; // so thu tu diem calib dau tien
	Nb_Point_X  : INT; 
	Nb_Point_Y  : INT;
	Delta_X     : INT;  // khoang cach giua cac diem theo phuong X
	Delta_Y     : INT;  // Khoang cach giua cac diem theo phuong Y
	Delta_A     : INT;  // Khoang cach giua cac diem theo phuong xoay
	Position_Cam    : INT;  // 0: TOP; 1: BOT
	Use : BOOL;
	Run_By_Array_Point : BOOL;
	Delay_Trigger_Time : INT;
	Bypass_VS : BOOL;
	Nb_Trigger_VS_Max : INT;
	Run_No_Trigger : BOOL;
END_STRUCT
END_TYPE

// Just_Motion_Control_x86_64_Linux_SM_WV/Application/STRUCT_/CAM/ModbusCam
TYPE ModbusCam :
STRUCT
	
	Pos_X, Pos_Y, Pos_R : REAL;
	POS_X_OFFSET, POS_Y_OFFSET, POS_R_OFFSET : REAL;
	POS_X_RESULT, POS_Y_RESULT, POS_R_RESULT : REAL;
	
END_STRUCT
END_TYPE

// Just_Motion_Control_x86_64_Linux_SM_WV/Application/STRUCT_/CAM/VS_Control
TYPE VS_Control :
STRUCT
	Trigger_VS, Run_Calib_VS, Run_Pick_For_Calib_VS, Trigger_Done, Calib_VS_Done, Run_Pos_Calib_Done, Trigger_Again, Pass_Trigger_VS_NG : BOOL;
	Enable_FB_Trigger_VS, Start_FB_Trigger_VS : BOOL;
	RTrig_Trigger_VS_Done, RTrig_Trigger_Calib_VS_Done : R_TRIG;
END_STRUCT
END_TYPE

// Just_Motion_Control_x86_64_Linux_SM_WV/Application/STRUCT_/COMMON/ST_ERROR_INFO
TYPE ST_ERROR_INFO :
STRUCT
    Active          : BOOL;     // TRUE khi lỗi đang tồn tại.
    ErrorID         : UDINT;    // Mã lỗi.
    ModuleID        : UINT;     // ID module phát sinh lỗi.
    SubCode         : UINT;     // Mã lỗi phụ của thiết bị hoặc thư viện.
    StepNo          : UINT;     // Bước chương trình khi lỗi xảy ra.
    ObjectID        : UDINT;    // Object liên quan đến lỗi, nếu có.
    ResetRequired   : BOOL;     // TRUE khi cần thao tác reset.
END_STRUCT
END_TYPE

// Just_Motion_Control_x86_64_Linux_SM_WV/Application/STRUCT_/COMMON/ST_MODULE_REQUEST
TYPE ST_MODULE_REQUEST :
STRUCT
    Execute     : BOOL;     // Cạnh lên bắt đầu yêu cầu.
    Abort       : BOOL;     // Yêu cầu hủy tác vụ đang chạy.
    Reset       : BOOL;     // Reset lỗi và đưa module về trạng thái Idle.

    RequestID   : UDINT;    // ID duy nhất của yêu cầu.
    Command     : UINT;     // Mã lệnh nội bộ của module.

    Param1      : REAL;     // Tham số mở rộng số 1.
    Param2      : REAL;     // Tham số mở rộng số 2.
    Param3      : REAL;     // Tham số mở rộng số 3.
    Param4      : REAL;     // Tham số mở rộng số 4.
END_STRUCT
END_TYPE

// Just_Motion_Control_x86_64_Linux_SM_WV/Application/STRUCT_/COMMON/ST_MODULE_RESPONSE
TYPE ST_MODULE_RESPONSE :
STRUCT
    Accepted    : BOOL;     // Module đã tiếp nhận yêu cầu.
    Busy        : BOOL;     // Module đang thực hiện yêu cầu.
    Done        : BOOL;     // Yêu cầu đã hoàn thành thành công.
    Aborted     : BOOL;     // Yêu cầu đã bị hủy.

    Error       : BOOL;     // Module đang có lỗi.
    ErrorID     : UDINT;    // Mã lỗi chi tiết.

    RequestID   : UDINT;    // ID yêu cầu đang được phản hồi.
    State       : UINT;     // Giá trị trạng thái hiện tại để hiển thị HMI.
END_STRUCT
END_TYPE

// Just_Motion_Control_x86_64_Linux_SM_WV/Application/STRUCT_/COMMON/ST_MotionProfile
//=============================================================================
// DUT: MOTION PROFILE
//=============================================================================
TYPE ST_MotionProfile :
STRUCT

    // Tốc độ chuyển động.
    Speed : REAL;

    // Gia tốc.
    Acceleration : REAL;

    // Giảm tốc.
    Deceleration : REAL;

    // Jerk.
    Jerk : REAL;

    // Bán kính Blend.
    BlendRadius : REAL;

END_STRUCT
END_TYPE

// Just_Motion_Control_x86_64_Linux_SM_WV/Application/STRUCT_/COMMON/ST_POS
TYPE ST_POS :
STRUCT
	X : REAL;   // Tọa độ theo trục X, đơn vị mm.
    Y : REAL;   // Tọa độ theo trục Y, đơn vị mm.
    Z : REAL;   // Tọa độ theo trục Z, đơn vị mm.
    A : REAL;   // Góc quay của SCARA quanh trục Z, đơn vị độ.
END_STRUCT
END_TYPE

// Just_Motion_Control_x86_64_Linux_SM_WV/Application/STRUCT_/COMMON/ST_RANGE_REAL
TYPE ST_RANGE_REAL :
STRUCT
    MinValue    : REAL;     // Giới hạn nhỏ nhất.
    MaxValue    : REAL;     // Giới hạn lớn nhất.
    Enable      : BOOL;     // TRUE khi cần kiểm tra giới hạn này.
END_STRUCT
END_TYPE

// Just_Motion_Control_x86_64_Linux_SM_WV/Application/STRUCT_/COMMON/ST_Transform2D
TYPE ST_Transform2D :
STRUCT
	X       : REAL;  // Độ tịnh tiến của hệ tọa độ theo X, mm.
    Y       : REAL;  // Độ tịnh tiến của hệ tọa độ theo Y, mm.
    A       : REAL;  // Góc xoay của hệ tọa độ, độ.
    Valid   : BOOL;  // TRUE khi dữ liệu biến đổi hợp lệ.
END_STRUCT
END_TYPE

// Just_Motion_Control_x86_64_Linux_SM_WV/Application/STRUCT_/COMMON/ST_VECTOR_2D
TYPE ST_VECTOR_2D :
STRUCT
    X       : REAL;     // Thành phần vector theo trục X.
    Y       : REAL;     // Thành phần vector theo trục Y.
END_STRUCT
END_TYPE

// Just_Motion_Control_x86_64_Linux_SM_WV/Application/STRUCT_/ConveyorTracking/ST_CONVEYOR_CONFIG
TYPE ST_CONVEYOR_CONFIG :
STRUCT
    Enable                  : BOOL;     // Cho phép conveyor.
    SimulationMode          : BOOL;     // Mô phỏng encoder.

    ConveyorID              : UINT;     // ID conveyor.
    DirectionSign           : SINT;     // 1: thuận; -1: đảo chiều.
    ConveyorAngleDeg        : REAL;     // Góc conveyor so với X robot.

//     PickZoneStartMM         : REAL;     // Đầu vùng gắp theo trục conveyor.
//     PickZoneEndMM           : REAL;     // Cuối vùng gắp.
//     ExpirePositionMM        : REAL;     // Vị trí object hết hiệu lực.

    RunningThresholdMMs     : REAL;     // Ngưỡng xác định conveyor chạy.
    MaxVelocityMMs          : REAL;     // Tốc độ lớn nhất, mm/s.
    MaxAccelerationMMs2     : REAL;     // Gia tốc lớn nhất, mm/s².

    VelocityFilterFactor    : REAL;     // Hệ số lọc vận tốc.
    PCSNumber               : UINT;     // PCS 1 hoặc 2.
	// Mốc cuối cho phép bắt đầu thao tác gắp.
    // Vượt mốc này mà chưa hút được vật thì phải abort.
//     AbortPositionMM      : REAL;
	Origin 				 : ST_POS;

    // Có thể đặt bằng hoặc xa hơn AbortPositionMM.
    // Qua mốc này object không active sẽ bị EXPIRED.
    // Project đã có ExpirePositionMM nên giữ nguyên.
END_STRUCT
END_TYPE

// Just_Motion_Control_x86_64_Linux_SM_WV/Application/STRUCT_/ConveyorTracking/ST_CONVEYOR_RUNTIME
TYPE ST_CONVEYOR_RUNTIME :
STRUCT
    Config          : ST_CONVEYOR_CONFIG; // Cấu hình conveyor.
    Status          : ST_CONVEYOR_STATUS; // Trạng thái runtime.

    LastPositionMM  : REAL;                // Position chu kỳ trước.
    LastVelocityMMs : REAL;                // Velocity chu kỳ trước.

    CaptureRequest  : BOOL;                // Yêu cầu chốt encoder.
    CaptureDone     : BOOL;                // Đã chốt encoder.
    CapturePosition : REAL;                // Position tại thời điểm capture.
END_STRUCT
END_TYPE

// Just_Motion_Control_x86_64_Linux_SM_WV/Application/STRUCT_/ConveyorTracking/ST_CONVEYOR_STATUS
TYPE ST_CONVEYOR_STATUS :
STRUCT
    Valid                   : BOOL;     // Position và velocity hợp lệ.
    State                   : E_ConveyorState;

    RawPosition             : LREAL;    // Position gốc từ SoftMotion.
    RawVelocity             : LREAL;    // Velocity gốc từ SoftMotion.

    PositionMM              : REAL;     // Position dùng trong ứng dụng.
    VelocityMMs             : REAL;     // Vận tốc tức thời.
    FilteredVelocityMMs     : REAL;     // Vận tốc sau lọc.
    AccelerationMMs2        : REAL;     // Gia tốc ước lượng.

    Direction               : SINT;     // 1 thuận, -1 nghịch, 0 đứng yên.
    Running                 : BOOL;     // Conveyor đang chạy.
    Standstill              : BOOL;     // Conveyor đang dừng.
    TrackingActive          : BOOL;     // Có robot đang tracking.

    Error                   : BOOL;     // Lỗi conveyor axis.
    ErrorID                 : UDINT;    // Mã lỗi.
END_STRUCT
END_TYPE

// Just_Motion_Control_x86_64_Linux_SM_WV/Application/STRUCT_/ConveyorTracking/ST_HMIToolConfigEditor
//=============================================================================
// DUT: HMI TOOL CONFIG EDITOR
//-----------------------------------------------------------------------------
// Bộ dữ liệu trung gian để một trang HMI có thể chỉnh nhiều Tool.
//=============================================================================
TYPE ST_HMIToolConfigEditor :
STRUCT
    // Index Tool người vận hành đang chọn trên HMI.
    SelectedIndex : UINT;

    // Index Tool đã được nạp vào EditData.
    // Khi Save phải dùng LoadedIndex để tránh ghi nhầm Tool.
    LoadedIndex : UINT;

    // Dữ liệu đang hiển thị và chỉnh sửa trên HMI.
    EditData : ST_ToolConfig;

    // Bản dữ liệu ban đầu khi Load.
    // Dùng để Cancel hoặc kiểm tra dữ liệu thay đổi.
    OriginalData : ST_ToolConfig;

    // Lệnh từ HMI.
    LoadCommand : BOOL;
    SaveCommand : BOOL;
    CancelCommand : BOOL;

    // Phản hồi dạng xung một vòng quét.
    LoadDone : BOOL;
    SaveDone : BOOL;

    // Trạng thái xử lý.
    Busy : BOOL;
    Error : BOOL;
    ErrorID : UDINT;

    // HMI đặt TRUE khi người dùng thay đổi bất kỳ ô nhập nào.
    DataChanged : BOOL;
END_STRUCT
END_TYPE

// Just_Motion_Control_x86_64_Linux_SM_WV/Application/STRUCT_/ConveyorTracking/ST_PCS_INFO
TYPE ST_PCS_INFO :
STRUCT
    Valid               : BOOL;     // PCS đã được tạo hợp lệ.
    PCSNumber           : UINT;     // PCS 1 hoặc PCS 2.

    ObjectID            : UDINT;    // Object đang gắn với PCS.
    InitialObjectPos    : ST_POS;   // Pose object lúc tạo PCS.

    ConveyorOrigin      : ST_POS;   // Gốc conveyor trong WCS.
    ConveyorCapturePos  : REAL;     // Position axis tại lúc thiết lập.

    InUse               : BOOL;     // PCS đang được motion sử dụng.
    Error               : BOOL;     // Lỗi tạo PCS.
    ErrorID             : UDINT;    // Mã lỗi.
END_STRUCT
END_TYPE

// Just_Motion_Control_x86_64_Linux_SM_WV/Application/STRUCT_/ConveyorTracking/ST_SensorObjectSourceConfig
//=============================================================================
// DUT: SENSOR OBJECT SOURCE CONFIG
//-----------------------------------------------------------------------------
// Cấu hình nguồn Object không dùng Vision.
//=============================================================================
TYPE ST_SensorObjectSourceConfig :
STRUCT

    // Cho phép sử dụng nguồn Sensor.
    Enable : BOOL;

    // ID của nguồn Sensor.
    SensorSourceID : UINT;
	
	// Name của nguồn Sensor.
    SensorSourceName : STRING[32];

    // Số kênh DI phát hiện sản phẩm.
    DetectInputChannel : UINT;

    // Mức logic tác động của DI.
    DetectActiveLevel : BOOL;

    // Thời gian chống rung tín hiệu Sensor.
    DebounceTime : TIME;

    // Khoảng cách tối thiểu giữa hai Object.
    MinimumObjectSpacingMM : REAL;

    // Pose mặc định của Object tại đúng vị trí Sensor.
    CapturePoseInConveyor : ST_POS;

    // Product Class mặc định.
    ProductClassID : UINT;

END_STRUCT
END_TYPE

// Just_Motion_Control_x86_64_Linux_SM_WV/Application/STRUCT_/ConveyorTracking/ST_TRACKING_CONFIG
TYPE ST_TRACKING_CONFIG :
STRUCT
    // TRUE: cho phép ứng dụng Conveyor Tracking hoạt động.
    Enable : BOOL;

    // Cách chọn object trong Queue.
    //SelectMode : E_TrackingSelectMode;

    // Cấu hình toàn bộ I/O của ứng dụng.
    IO : ST_TRACKING_IO_CONFIG;

    // Cấu hình vùng làm việc trên conveyor.
    Workspace : ST_TRACKING_WORKSPACE_CONFIG;

    // Cấu hình động học cho từng pha chuyển động.
    Motion : ST_TRACKING_MOTION_CONFIG;

    // Offset TCP so với tâm object trong PCS.
    PickOffset : ST_POS;

    // Độ cao approach cộng thêm vào PickOffset.Z.
    ApproachHeight : REAL;

    // Độ cao retract cộng thêm vào PickOffset.Z.
    RetractHeight : REAL;

    // Điểm rời vùng conveyor trong hệ robot/base.
    LeavePos : ST_POS;

    // Điểm đặt sản phẩm trong hệ robot/base.
    PlacePos : ST_POS;

    // Thời gian chờ sau khi bật hút trước khi kiểm tra VacuumOK.
    PickDelay : TIME;

    // Thời gian tối đa chờ VacuumOK.
    VacuumTimeout : TIME;

    // Số lần thử hút tối đa.
    MaxPickAttempts : UINT;

    // Thời gian bật van thổi khi nhả sản phẩm.
    BlowTime : TIME;

    // TRUE: sử dụng tín hiệu mô phỏng thay cho I/O thật.
    SimulationMode : BOOL;

    // Tín hiệu VacuumOK mô phỏng.
    SimulationVacuumOK : BOOL;
	// Thuật toán Scheduler dùng để chọn object.
    SelectMode : E_TrackingSelectMode;

    // ObjectID cụ thể khi SelectMode = TRACK_SELECT_SPECIFIC_ID.
    SpecificObjectID : UDINT;

    // Priority mặc định khi Vision/Application không gán.
    DefaultObjectPriority : UINT;

    // Thời gian gắp ước tính mặc định, đơn vị giây.
    DefaultEstimatedPickTimeSec : REAL;

    // Điểm Vision tối thiểu để object được phép tham gia Scheduler.
    MinimumVisionScore : REAL;
END_STRUCT
END_TYPE

// Just_Motion_Control_x86_64_Linux_SM_WV/Application/STRUCT_/ConveyorTracking/ST_TRACKING_IO_CONFIG
TYPE ST_TRACKING_IO_CONFIG :
STRUCT
    // Chỉ số output điều khiển van hút trong mảng GVL.Y[].
    VacuumOutputIndex : UINT;

    // TRUE: output TRUE làm van hút ON.
    // FALSE: output FALSE làm van hút ON.
    VacuumOutputActiveHigh : BOOL;

    // Chỉ số output điều khiển van thổi trong mảng GVL.Y[].
    BlowOutputIndex : UINT;

    // TRUE: output TRUE làm van thổi ON.
    // FALSE: output FALSE làm van thổi ON.
    BlowOutputActiveHigh : BOOL;

    // Chỉ số output báo module tracking đang hoạt động.
    TrackingActiveOutputIndex : UINT;

    // Cực tính output báo trạng thái tracking.
    TrackingActiveOutputActiveHigh : BOOL;

    // Chỉ số input xác nhận chân không trong mảng GVL.X[].
    VacuumOKInputIndex : UINT;

    // TRUE: input TRUE nghĩa là VacuumOK.
    // FALSE: input FALSE nghĩa là VacuumOK.
    VacuumOKInputActiveHigh : BOOL;

    // Chỉ số input cảm biến phát hiện sản phẩm.
    ProductSensorInputIndex : UINT;

    // Cực tính input cảm biến sản phẩm.
    ProductSensorActiveHigh : BOOL;

    // Chỉ số input cho phép module tracking chạy.
    EnableInputIndex : UINT;

    // Cực tính input Enable.
    EnableInputActiveHigh : BOOL;

    // Chỉ số input reset module tracking.
    ResetInputIndex : UINT;

    // Cực tính input Reset.
    ResetInputActiveHigh : BOOL;
END_STRUCT
END_TYPE

// Just_Motion_Control_x86_64_Linux_SM_WV/Application/STRUCT_/ConveyorTracking/ST_TRACKING_MOTION_CONFIG
TYPE ST_TRACKING_MOTION_CONFIG :
STRUCT
	// Thông số chuyển động tới điểm phía trên vật.
    Approach : ST_TRACKING_MOTION_PHASE_CONFIG;

    // Thông số chuyển động hạ xuống điểm gắp.
    Pick : ST_TRACKING_MOTION_PHASE_CONFIG;

    // Thông số chuyển động nâng vật sau khi gắp.
    Retract : ST_TRACKING_MOTION_PHASE_CONFIG;

    // Thông số chuyển động rời vùng conveyor.
    Leave : ST_TRACKING_MOTION_PHASE_CONFIG;

    // Thông số chuyển động tới điểm đặt.
    Place : ST_TRACKING_MOTION_PHASE_CONFIG;
END_STRUCT
END_TYPE

// Just_Motion_Control_x86_64_Linux_SM_WV/Application/STRUCT_/ConveyorTracking/ST_TRACKING_MOTION_PHASE_CONFIG
TYPE ST_TRACKING_MOTION_PHASE_CONFIG  :
STRUCT
	// Tốc độ đặt cho pha chuyển động.
    Speed : REAL;

    // Gia tốc đặt cho pha chuyển động.
    Acceleration : REAL;

    // Giảm tốc đặt cho pha chuyển động.
    Deceleration : REAL;

    // Jerk đặt cho pha chuyển động.
    Jerk : REAL;

    // Bán kính blend; đặt 0 nếu cần dừng chính xác tại điểm.
    BlendRadius : REAL;
END_STRUCT
END_TYPE

// Just_Motion_Control_x86_64_Linux_SM_WV/Application/STRUCT_/ConveyorTracking/ST_TRACKING_OBJECT
//=============================================================================
// DUT: TRACKING OBJECT
//-----------------------------------------------------------------------------
// Dữ liệu chuẩn hóa của một sản phẩm trong Tracking Queue.
//=============================================================================
TYPE ST_TRACKING_OBJECT :
STRUCT

    // TRUE khi Slot đang chứa Object hợp lệ.
    Valid : BOOL;

    // ID duy nhất của Object.
    ObjectID : UDINT;

    // Mã loại sản phẩm.
    ProductClassID : UINT;

    // Nguồn tạo Object.
    SourceType : E_ObjectSourceType;
	// ID của nguồn tạo Object.
	// SENSOR -> SensorSourceID.
	// VISION -> có thể dùng VisionSourceID hoặc Camera/Job tùy kiến trúc.
	SourceID : UINT;

    // Pose của Object trong hệ Conveyor tại thời điểm Capture.
    PoseInConveyor : ST_POS;

    // Vị trí Conveyor tại thời điểm Object được Capture.
    CaptureConveyorPositionMM : LREAL;

